// TIA Portal V21 export
FUNCTION "CPEC" : Void   // FC17, LAD
{ S7_Optimized_Access := 'TRUE' }
// stored: SetENOAutomatically false
   VAR_TEMP   // added for the SCL form of the ladder/FBD networks
      _w1 : Bool;
      _w2 : Bool;
      _w3 : Bool;
      _w4 : Bool;
      _w5 : Bool;
      _w6 : Bool;
      _w7 : Bool;
      _w8 : Bool;
      _w9 : Bool;
      _w10 : Bool;
      _w11 : Bool;
      _w12 : Bool;
      _w13 : Bool;
      _w14 : Bool;
      _w15 : Bool;
      _w16 : Bool;
      _w17 : Bool;
      _w18 : Bool;
      _w19 : Bool;
      _w20 : Bool;
      _w21 : Bool;
      _w22 : Bool;
      _w23 : Bool;
      _w24 : Bool;
      _w25 : Bool;
      _w26 : Bool;
      _w27 : Bool;
      _w28 : Bool;
      _w29 : Bool;
      _w30 : Bool;
      _w31 : Bool;
      _w32 : Bool;
      _w33 : Bool;
      _w34 : Bool;
      _w35 : Bool;
      _w36 : Bool;
      _w37 : Bool;
      _w38 : Bool;
      _w39 : Bool;
      _w40 : Bool;
      _w41 : Bool;
      _w42 : Bool;
      _w43 : Bool;
      _w44 : Bool;
      _w45 : Bool;
      _w46 : Bool;
      _w47 : Bool;
      _w48 : Bool;
      _w49 : Bool;
      _w50 : Bool;
      _w51 : Bool;
      _w52 : Bool;
      _w53 : Bool;
      _w54 : Bool;
   END_VAR
BEGIN

REGION Network 1
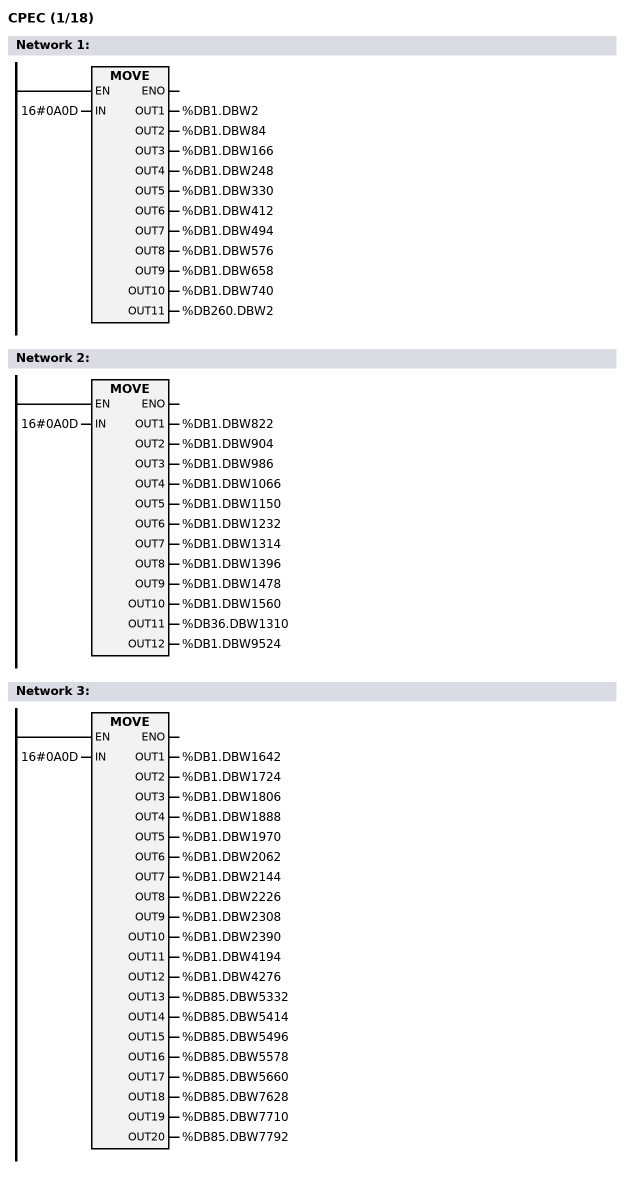
   RUNG wire#powerrail
      Move(in := 16#0A0D, out1 => %DB1.DBW2, out2 => %DB1.DBW84, out3 => %DB1.DBW166, out4 => %DB1.DBW248, out5 => %DB1.DBW330, out6 => %DB1.DBW412, out7 => %DB1.DBW494, out8 => %DB1.DBW576, out9 => %DB1.DBW658, out10 => %DB1.DBW740, out11 => %DB260.DBW2)
   END_RUNG
   // the same network as SCL:
   %DB1.DBW2 := 16#0A0D;
   %DB1.DBW84 := 16#0A0D;
   %DB1.DBW166 := 16#0A0D;
   %DB1.DBW248 := 16#0A0D;
   %DB1.DBW330 := 16#0A0D;
   %DB1.DBW412 := 16#0A0D;
   %DB1.DBW494 := 16#0A0D;
   %DB1.DBW576 := 16#0A0D;
   %DB1.DBW658 := 16#0A0D;
   %DB1.DBW740 := 16#0A0D;
   %DB260.DBW2 := 16#0A0D;
END_REGION

REGION Network 2
   RUNG wire#powerrail
      Move(in := 16#0A0D, out1 => %DB1.DBW822, out2 => %DB1.DBW904, out3 => %DB1.DBW986, out4 => %DB1.DBW1066, out5 => %DB1.DBW1150, out6 => %DB1.DBW1232, out7 => %DB1.DBW1314, out8 => %DB1.DBW1396, out9 => %DB1.DBW1478, out10 => %DB1.DBW1560, out11 => %DB36.DBW1310, out12 => %DB1.DBW9524)
   END_RUNG
   // the same network as SCL:
   %DB1.DBW822 := 16#0A0D;
   %DB1.DBW904 := 16#0A0D;
   %DB1.DBW986 := 16#0A0D;
   %DB1.DBW1066 := 16#0A0D;
   %DB1.DBW1150 := 16#0A0D;
   %DB1.DBW1232 := 16#0A0D;
   %DB1.DBW1314 := 16#0A0D;
   %DB1.DBW1396 := 16#0A0D;
   %DB1.DBW1478 := 16#0A0D;
   %DB1.DBW1560 := 16#0A0D;
   %DB36.DBW1310 := 16#0A0D;
   %DB1.DBW9524 := 16#0A0D;
END_REGION

REGION Network 3
   RUNG wire#powerrail
      Move(in := 16#0A0D, out1 => %DB1.DBW1642, out2 => %DB1.DBW1724, out3 => %DB1.DBW1806, out4 => %DB1.DBW1888, out5 => %DB1.DBW1970, out6 => %DB1.DBW2062, out7 => %DB1.DBW2144, out8 => %DB1.DBW2226, out9 => %DB1.DBW2308, out10 => %DB1.DBW2390, out11 => %DB1.DBW4194, out12 => %DB1.DBW4276, out13 => %DB85.DBW5332, out14 => %DB85.DBW5414, out15 => %DB85.DBW5496, out16 => %DB85.DBW5578, out17 => %DB85.DBW5660, out18 => %DB85.DBW7628, out19 => %DB85.DBW7710, out20 => %DB85.DBW7792)
   END_RUNG
   // the same network as SCL:
   %DB1.DBW1642 := 16#0A0D;
   %DB1.DBW1724 := 16#0A0D;
   %DB1.DBW1806 := 16#0A0D;
   %DB1.DBW1888 := 16#0A0D;
   %DB1.DBW1970 := 16#0A0D;
   %DB1.DBW2062 := 16#0A0D;
   %DB1.DBW2144 := 16#0A0D;
   %DB1.DBW2226 := 16#0A0D;
   %DB1.DBW2308 := 16#0A0D;
   %DB1.DBW2390 := 16#0A0D;
   %DB1.DBW4194 := 16#0A0D;
   %DB1.DBW4276 := 16#0A0D;
   %DB85.DBW5332 := 16#0A0D;
   %DB85.DBW5414 := 16#0A0D;
   %DB85.DBW5496 := 16#0A0D;
   %DB85.DBW5578 := 16#0A0D;
   %DB85.DBW5660 := 16#0A0D;
   %DB85.DBW7628 := 16#0A0D;
   %DB85.DBW7710 := 16#0A0D;
   %DB85.DBW7792 := 16#0A0D;
END_REGION

REGION Network 4
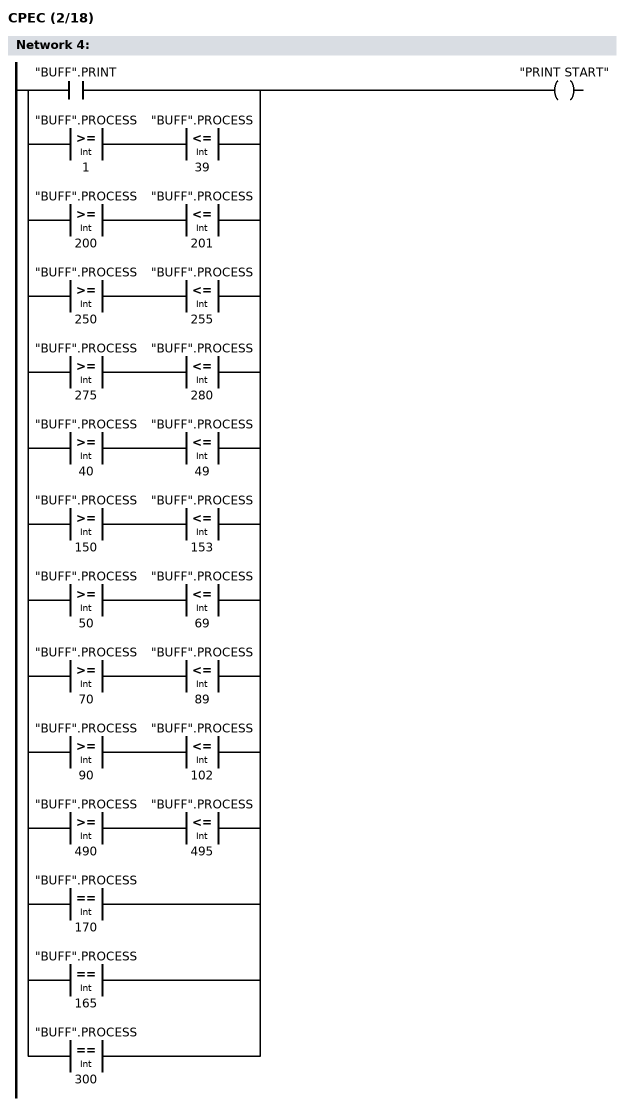
   RUNG wire#powerrail
      Contact( "BUFF".PRINT )
      wire#w1
      Coil( "PRINT START" )
   END_RUNG
   RUNG wire#powerrail
      { S7_Templates := "SrcType := Int" } GE_Contact(in1 := "BUFF".PROCESS, in2 := 1)
      { S7_Templates := "SrcType := Int" } LE_Contact(in1 := "BUFF".PROCESS, in2 := 39)
   END_RUNG wire#w1
   RUNG wire#powerrail
      { S7_Templates := "SrcType := Int" } GE_Contact(in1 := "BUFF".PROCESS, in2 := 200)
      { S7_Templates := "SrcType := Int" } LE_Contact(in1 := "BUFF".PROCESS, in2 := 201)
   END_RUNG wire#w1
   RUNG wire#powerrail
      { S7_Templates := "SrcType := Int" } GE_Contact(in1 := "BUFF".PROCESS, in2 := 250)
      { S7_Templates := "SrcType := Int" } LE_Contact(in1 := "BUFF".PROCESS, in2 := 255)
   END_RUNG wire#w1
   RUNG wire#powerrail
      { S7_Templates := "SrcType := Int" } GE_Contact(in1 := "BUFF".PROCESS, in2 := 275)
      { S7_Templates := "SrcType := Int" } LE_Contact(in1 := "BUFF".PROCESS, in2 := 280)
   END_RUNG wire#w1
   RUNG wire#powerrail
      { S7_Templates := "SrcType := Int" } GE_Contact(in1 := "BUFF".PROCESS, in2 := 40)
      { S7_Templates := "SrcType := Int" } LE_Contact(in1 := "BUFF".PROCESS, in2 := 49)
   END_RUNG wire#w1
   RUNG wire#powerrail
      { S7_Templates := "SrcType := Int" } GE_Contact(in1 := "BUFF".PROCESS, in2 := 150)
      { S7_Templates := "SrcType := Int" } LE_Contact(in1 := "BUFF".PROCESS, in2 := 153)
   END_RUNG wire#w1
   RUNG wire#powerrail
      { S7_Templates := "SrcType := Int" } GE_Contact(in1 := "BUFF".PROCESS, in2 := 50)
      { S7_Templates := "SrcType := Int" } LE_Contact(in1 := "BUFF".PROCESS, in2 := 69)
   END_RUNG wire#w1
   RUNG wire#powerrail
      { S7_Templates := "SrcType := Int" } GE_Contact(in1 := "BUFF".PROCESS, in2 := 70)
      { S7_Templates := "SrcType := Int" } LE_Contact(in1 := "BUFF".PROCESS, in2 := 89)
   END_RUNG wire#w1
   RUNG wire#powerrail
      { S7_Templates := "SrcType := Int" } GE_Contact(in1 := "BUFF".PROCESS, in2 := 90)
      { S7_Templates := "SrcType := Int" } LE_Contact(in1 := "BUFF".PROCESS, in2 := 102)
   END_RUNG wire#w1
   RUNG wire#powerrail
      { S7_Templates := "SrcType := Int" } GE_Contact(in1 := "BUFF".PROCESS, in2 := 490)
      { S7_Templates := "SrcType := Int" } LE_Contact(in1 := "BUFF".PROCESS, in2 := 495)
   END_RUNG wire#w1
   RUNG wire#powerrail
      { S7_Templates := "SrcType := Int" } EQ_Contact(in1 := "BUFF".PROCESS, in2 := 170)
   END_RUNG wire#w1
   RUNG wire#powerrail
      { S7_Templates := "SrcType := Int" } EQ_Contact(in1 := "BUFF".PROCESS, in2 := 165)
   END_RUNG wire#w1
   RUNG wire#powerrail
      { S7_Templates := "SrcType := Int" } EQ_Contact(in1 := "BUFF".PROCESS, in2 := 300)
   END_RUNG wire#w1
   // the same network as SCL:
   "PRINT START" := "BUFF".PRINT OR (("BUFF".PROCESS >= 1) AND ("BUFF".PROCESS <= 39)) OR (("BUFF".PROCESS >= 200) AND ("BUFF".PROCESS <= 201)) OR (("BUFF".PROCESS >= 250) AND ("BUFF".PROCESS <= 255)) OR (("BUFF".PROCESS >= 275) AND ("BUFF".PROCESS <= 280)) OR (("BUFF".PROCESS >= 40) AND ("BUFF".PROCESS <= 49)) OR (("BUFF".PROCESS >= 150) AND ("BUFF".PROCESS <= 153)) OR (("BUFF".PROCESS >= 50) AND ("BUFF".PROCESS <= 69)) OR (("BUFF".PROCESS >= 70) AND ("BUFF".PROCESS <= 89)) OR (("BUFF".PROCESS >= 90) AND ("BUFF".PROCESS <= 102)) OR (("BUFF".PROCESS >= 490) AND ("BUFF".PROCESS <= 495)) OR ("BUFF".PROCESS = 170) OR ("BUFF".PROCESS = 165) OR ("BUFF".PROCESS = 300);
END_REGION

REGION Network 5
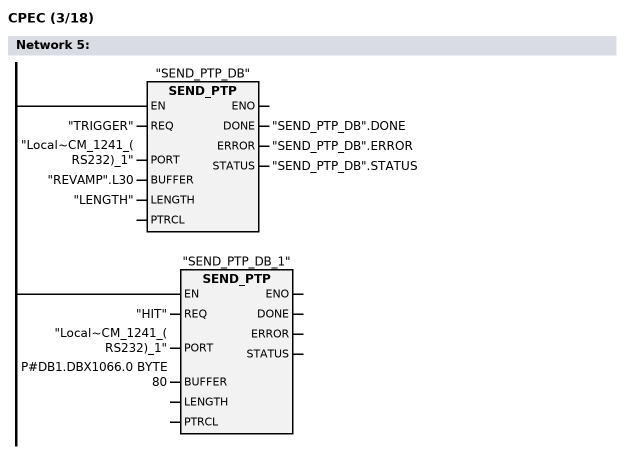
   RUNG wire#powerrail
      "SEND_PTP_DB".SEND_PTP(REQ := "TRIGGER", PORT := "Local~CM_1241_(RS232)_1", BUFFER := "REVAMP".L30, LENGTH := "LENGTH", PTRCL :=, DONE => "SEND_PTP_DB".DONE, ERROR => "SEND_PTP_DB".ERROR, STATUS => "SEND_PTP_DB".STATUS)
   END_RUNG
   RUNG wire#powerrail
      "SEND_PTP_DB_1".SEND_PTP(REQ := "HIT", PORT := "Local~CM_1241_(RS232)_1", BUFFER := P#DB1.DBX1066.0 BYTE 80, LENGTH :=, PTRCL :=, DONE =>, ERROR =>, STATUS =>)
   END_RUNG
   // the same network as SCL:
   "SEND_PTP_DB"(REQ := "TRIGGER",   // SEND_PTP
                 PORT := "Local~CM_1241_(RS232)_1",
                 BUFFER := "REVAMP".L30,
                 LENGTH := "LENGTH",
                 DONE => "SEND_PTP_DB".DONE,
                 ERROR => "SEND_PTP_DB".ERROR,
                 STATUS => "SEND_PTP_DB".STATUS);
   "SEND_PTP_DB_1"(REQ := "HIT", PORT := "Local~CM_1241_(RS232)_1", BUFFER := P#DB1.DBX1066.0 BYTE 80);   // SEND_PTP
END_REGION

REGION Network 6
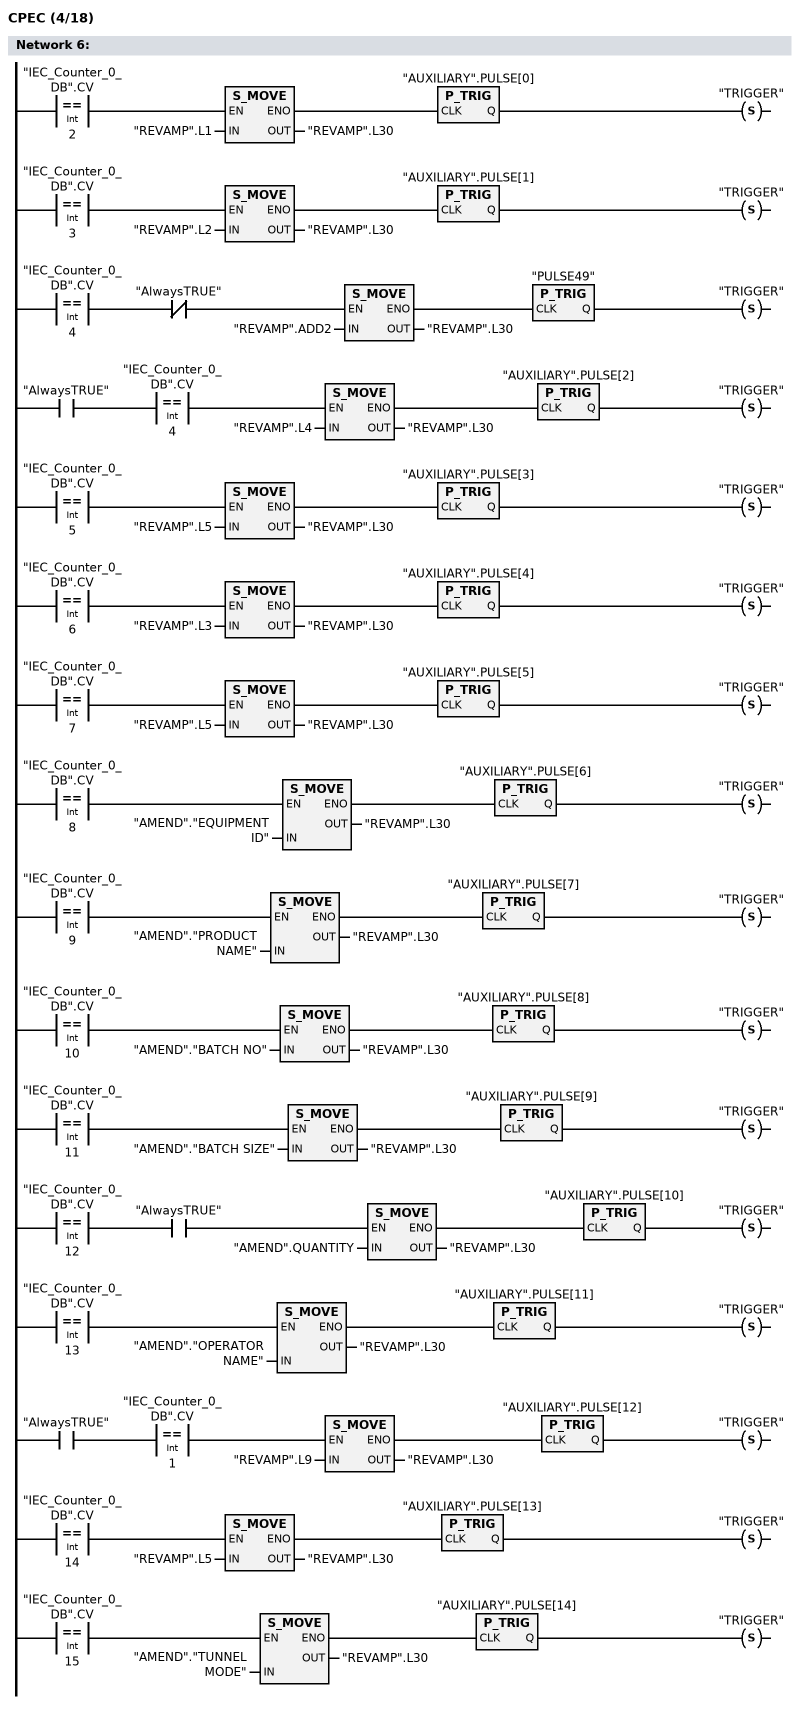
   RUNG wire#powerrail
      { S7_Templates := "SrcType := Int" } EQ_Contact(in1 := "IEC_Counter_0_DB".CV, in2 := 2)
      S_Move(in := "REVAMP".L1, out => "REVAMP".L30)
      P_Trig( "AUXILIARY".PULSE[0] )
      S_Coil( "TRIGGER" )
   END_RUNG
   RUNG wire#powerrail
      { S7_Templates := "SrcType := Int" } EQ_Contact(in1 := "IEC_Counter_0_DB".CV, in2 := 3)
      S_Move(in := "REVAMP".L2, out => "REVAMP".L30)
      P_Trig( "AUXILIARY".PULSE[1] )
      S_Coil( "TRIGGER" )
   END_RUNG
   RUNG wire#powerrail
      { S7_Templates := "SrcType := Int" } EQ_Contact(in1 := "IEC_Counter_0_DB".CV, in2 := 4)
      I_Contact( "AlwaysTRUE" )
      S_Move(in := "REVAMP".ADD2, out => "REVAMP".L30)
      P_Trig( "PULSE49" )
      S_Coil( "TRIGGER" )
   END_RUNG
   RUNG wire#powerrail
      Contact( "AlwaysTRUE" )
      { S7_Templates := "SrcType := Int" } EQ_Contact(in1 := "IEC_Counter_0_DB".CV, in2 := 4)
      S_Move(in := "REVAMP".L4, out => "REVAMP".L30)
      P_Trig( "AUXILIARY".PULSE[2] )
      S_Coil( "TRIGGER" )
   END_RUNG
   RUNG wire#powerrail
      { S7_Templates := "SrcType := Int" } EQ_Contact(in1 := "IEC_Counter_0_DB".CV, in2 := 5)
      S_Move(in := "REVAMP".L5, out => "REVAMP".L30)
      P_Trig( "AUXILIARY".PULSE[3] )
      S_Coil( "TRIGGER" )
   END_RUNG
   RUNG wire#powerrail
      { S7_Templates := "SrcType := Int" } EQ_Contact(in1 := "IEC_Counter_0_DB".CV, in2 := 6)
      S_Move(in := "REVAMP".L3, out => "REVAMP".L30)
      P_Trig( "AUXILIARY".PULSE[4] )
      S_Coil( "TRIGGER" )
   END_RUNG
   RUNG wire#powerrail
      { S7_Templates := "SrcType := Int" } EQ_Contact(in1 := "IEC_Counter_0_DB".CV, in2 := 7)
      S_Move(in := "REVAMP".L5, out => "REVAMP".L30)
      P_Trig( "AUXILIARY".PULSE[5] )
      S_Coil( "TRIGGER" )
   END_RUNG
   RUNG wire#powerrail
      { S7_Templates := "SrcType := Int" } EQ_Contact(in1 := "IEC_Counter_0_DB".CV, in2 := 8)
      S_Move(in := "AMEND"."EQUIPMENT ID", out => "REVAMP".L30)
      P_Trig( "AUXILIARY".PULSE[6] )
      S_Coil( "TRIGGER" )
   END_RUNG
   RUNG wire#powerrail
      { S7_Templates := "SrcType := Int" } EQ_Contact(in1 := "IEC_Counter_0_DB".CV, in2 := 9)
      S_Move(in := "AMEND"."PRODUCT NAME", out => "REVAMP".L30)
      P_Trig( "AUXILIARY".PULSE[7] )
      S_Coil( "TRIGGER" )
   END_RUNG
   RUNG wire#powerrail
      { S7_Templates := "SrcType := Int" } EQ_Contact(in1 := "IEC_Counter_0_DB".CV, in2 := 10)
      S_Move(in := "AMEND"."BATCH NO", out => "REVAMP".L30)
      P_Trig( "AUXILIARY".PULSE[8] )
      S_Coil( "TRIGGER" )
   END_RUNG
   RUNG wire#powerrail
      { S7_Templates := "SrcType := Int" } EQ_Contact(in1 := "IEC_Counter_0_DB".CV, in2 := 11)
      S_Move(in := "AMEND"."BATCH SIZE", out => "REVAMP".L30)
      P_Trig( "AUXILIARY".PULSE[9] )
      S_Coil( "TRIGGER" )
   END_RUNG
   RUNG wire#powerrail
      { S7_Templates := "SrcType := Int" } EQ_Contact(in1 := "IEC_Counter_0_DB".CV, in2 := 12)
      Contact( "AlwaysTRUE" )
      S_Move(in := "AMEND".QUANTITY, out => "REVAMP".L30)
      P_Trig( "AUXILIARY".PULSE[10] )
      S_Coil( "TRIGGER" )
   END_RUNG
   RUNG wire#powerrail
      { S7_Templates := "SrcType := Int" } EQ_Contact(in1 := "IEC_Counter_0_DB".CV, in2 := 13)
      S_Move(in := "AMEND"."OPERATOR NAME", out => "REVAMP".L30)
      P_Trig( "AUXILIARY".PULSE[11] )
      S_Coil( "TRIGGER" )
   END_RUNG
   RUNG wire#powerrail
      Contact( "AlwaysTRUE" )
      { S7_Templates := "SrcType := Int" } EQ_Contact(in1 := "IEC_Counter_0_DB".CV, in2 := 1)
      S_Move(in := "REVAMP".L9, out => "REVAMP".L30)
      P_Trig( "AUXILIARY".PULSE[12] )
      S_Coil( "TRIGGER" )
   END_RUNG
   RUNG wire#powerrail
      { S7_Templates := "SrcType := Int" } EQ_Contact(in1 := "IEC_Counter_0_DB".CV, in2 := 14)
      S_Move(in := "REVAMP".L5, out => "REVAMP".L30)
      P_Trig( "AUXILIARY".PULSE[13] )
      S_Coil( "TRIGGER" )
   END_RUNG
   RUNG wire#powerrail
      { S7_Templates := "SrcType := Int" } EQ_Contact(in1 := "IEC_Counter_0_DB".CV, in2 := 15)
      S_Move(in := "AMEND"."TUNNEL MODE", out => "REVAMP".L30)
      P_Trig( "AUXILIARY".PULSE[14] )
      S_Coil( "TRIGGER" )
   END_RUNG
   // the same network as SCL:
   #_w1 := "IEC_Counter_0_DB".CV = 2;
   IF #_w1 THEN "REVAMP".L30 := "REVAMP".L1; END_IF;
   #_w2 := #_w1 AND NOT "AUXILIARY".PULSE[0];   // rising edge
   "AUXILIARY".PULSE[0] := #_w1;
   IF #_w2 THEN "TRIGGER" := TRUE; END_IF;
   #_w3 := "IEC_Counter_0_DB".CV = 3;
   IF #_w3 THEN "REVAMP".L30 := "REVAMP".L2; END_IF;
   #_w4 := #_w3 AND NOT "AUXILIARY".PULSE[1];   // rising edge
   "AUXILIARY".PULSE[1] := #_w3;
   IF #_w4 THEN "TRIGGER" := TRUE; END_IF;
   #_w5 := ("IEC_Counter_0_DB".CV = 4) AND NOT "AlwaysTRUE";
   IF #_w5 THEN "REVAMP".L30 := "REVAMP".ADD2; END_IF;
   #_w6 := #_w5 AND NOT "PULSE49";   // rising edge
   "PULSE49" := #_w5;
   IF #_w6 THEN "TRIGGER" := TRUE; END_IF;
   #_w7 := "AlwaysTRUE" AND ("IEC_Counter_0_DB".CV = 4);
   IF #_w7 THEN "REVAMP".L30 := "REVAMP".L4; END_IF;
   #_w8 := #_w7 AND NOT "AUXILIARY".PULSE[2];   // rising edge
   "AUXILIARY".PULSE[2] := #_w7;
   IF #_w8 THEN "TRIGGER" := TRUE; END_IF;
   #_w9 := "IEC_Counter_0_DB".CV = 5;
   IF #_w9 THEN "REVAMP".L30 := "REVAMP".L5; END_IF;
   #_w10 := #_w9 AND NOT "AUXILIARY".PULSE[3];   // rising edge
   "AUXILIARY".PULSE[3] := #_w9;
   IF #_w10 THEN "TRIGGER" := TRUE; END_IF;
   #_w11 := "IEC_Counter_0_DB".CV = 6;
   IF #_w11 THEN "REVAMP".L30 := "REVAMP".L3; END_IF;
   #_w12 := #_w11 AND NOT "AUXILIARY".PULSE[4];   // rising edge
   "AUXILIARY".PULSE[4] := #_w11;
   IF #_w12 THEN "TRIGGER" := TRUE; END_IF;
   #_w13 := "IEC_Counter_0_DB".CV = 7;
   IF #_w13 THEN "REVAMP".L30 := "REVAMP".L5; END_IF;
   #_w14 := #_w13 AND NOT "AUXILIARY".PULSE[5];   // rising edge
   "AUXILIARY".PULSE[5] := #_w13;
   IF #_w14 THEN "TRIGGER" := TRUE; END_IF;
   #_w15 := "IEC_Counter_0_DB".CV = 8;
   IF #_w15 THEN "REVAMP".L30 := "AMEND"."EQUIPMENT ID"; END_IF;
   #_w16 := #_w15 AND NOT "AUXILIARY".PULSE[6];   // rising edge
   "AUXILIARY".PULSE[6] := #_w15;
   IF #_w16 THEN "TRIGGER" := TRUE; END_IF;
   #_w17 := "IEC_Counter_0_DB".CV = 9;
   IF #_w17 THEN "REVAMP".L30 := "AMEND"."PRODUCT NAME"; END_IF;
   #_w18 := #_w17 AND NOT "AUXILIARY".PULSE[7];   // rising edge
   "AUXILIARY".PULSE[7] := #_w17;
   IF #_w18 THEN "TRIGGER" := TRUE; END_IF;
   #_w19 := "IEC_Counter_0_DB".CV = 10;
   IF #_w19 THEN "REVAMP".L30 := "AMEND"."BATCH NO"; END_IF;
   #_w20 := #_w19 AND NOT "AUXILIARY".PULSE[8];   // rising edge
   "AUXILIARY".PULSE[8] := #_w19;
   IF #_w20 THEN "TRIGGER" := TRUE; END_IF;
   #_w21 := "IEC_Counter_0_DB".CV = 11;
   IF #_w21 THEN "REVAMP".L30 := "AMEND"."BATCH SIZE"; END_IF;
   #_w22 := #_w21 AND NOT "AUXILIARY".PULSE[9];   // rising edge
   "AUXILIARY".PULSE[9] := #_w21;
   IF #_w22 THEN "TRIGGER" := TRUE; END_IF;
   #_w23 := ("IEC_Counter_0_DB".CV = 12) AND "AlwaysTRUE";
   IF #_w23 THEN "REVAMP".L30 := "AMEND".QUANTITY; END_IF;
   #_w24 := #_w23 AND NOT "AUXILIARY".PULSE[10];   // rising edge
   "AUXILIARY".PULSE[10] := #_w23;
   IF #_w24 THEN "TRIGGER" := TRUE; END_IF;
   #_w25 := "IEC_Counter_0_DB".CV = 13;
   IF #_w25 THEN "REVAMP".L30 := "AMEND"."OPERATOR NAME"; END_IF;
   #_w26 := #_w25 AND NOT "AUXILIARY".PULSE[11];   // rising edge
   "AUXILIARY".PULSE[11] := #_w25;
   IF #_w26 THEN "TRIGGER" := TRUE; END_IF;
   #_w27 := "AlwaysTRUE" AND ("IEC_Counter_0_DB".CV = 1);
   IF #_w27 THEN "REVAMP".L30 := "REVAMP".L9; END_IF;
   #_w28 := #_w27 AND NOT "AUXILIARY".PULSE[12];   // rising edge
   "AUXILIARY".PULSE[12] := #_w27;
   IF #_w28 THEN "TRIGGER" := TRUE; END_IF;
   #_w29 := "IEC_Counter_0_DB".CV = 14;
   IF #_w29 THEN "REVAMP".L30 := "REVAMP".L5; END_IF;
   #_w30 := #_w29 AND NOT "AUXILIARY".PULSE[13];   // rising edge
   "AUXILIARY".PULSE[13] := #_w29;
   IF #_w30 THEN "TRIGGER" := TRUE; END_IF;
   #_w31 := "IEC_Counter_0_DB".CV = 15;
   IF #_w31 THEN "REVAMP".L30 := "AMEND"."TUNNEL MODE"; END_IF;
   #_w32 := #_w31 AND NOT "AUXILIARY".PULSE[14];   // rising edge
   "AUXILIARY".PULSE[14] := #_w31;
   IF #_w32 THEN "TRIGGER" := TRUE; END_IF;
END_REGION

REGION Network 7
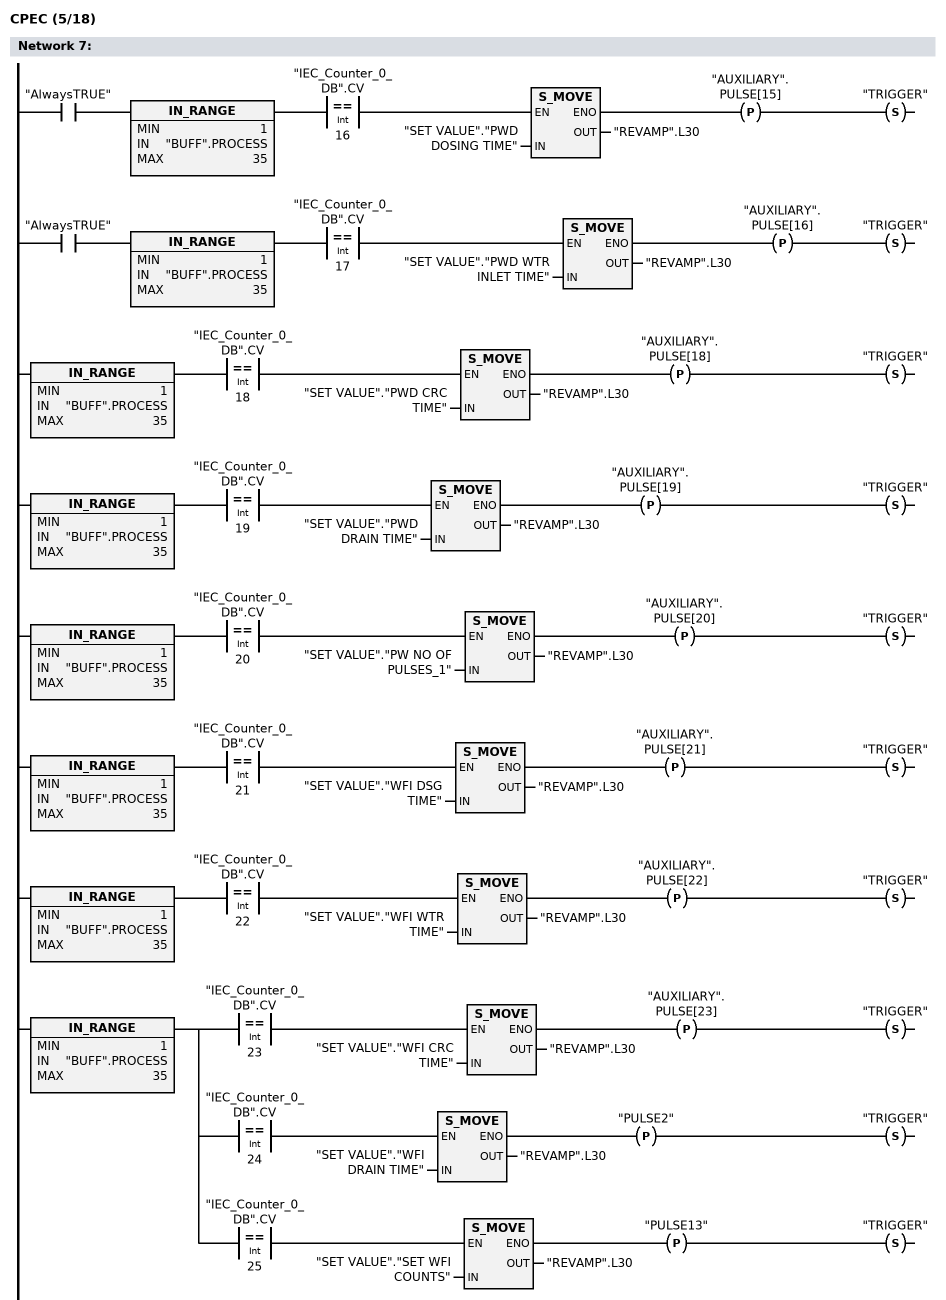
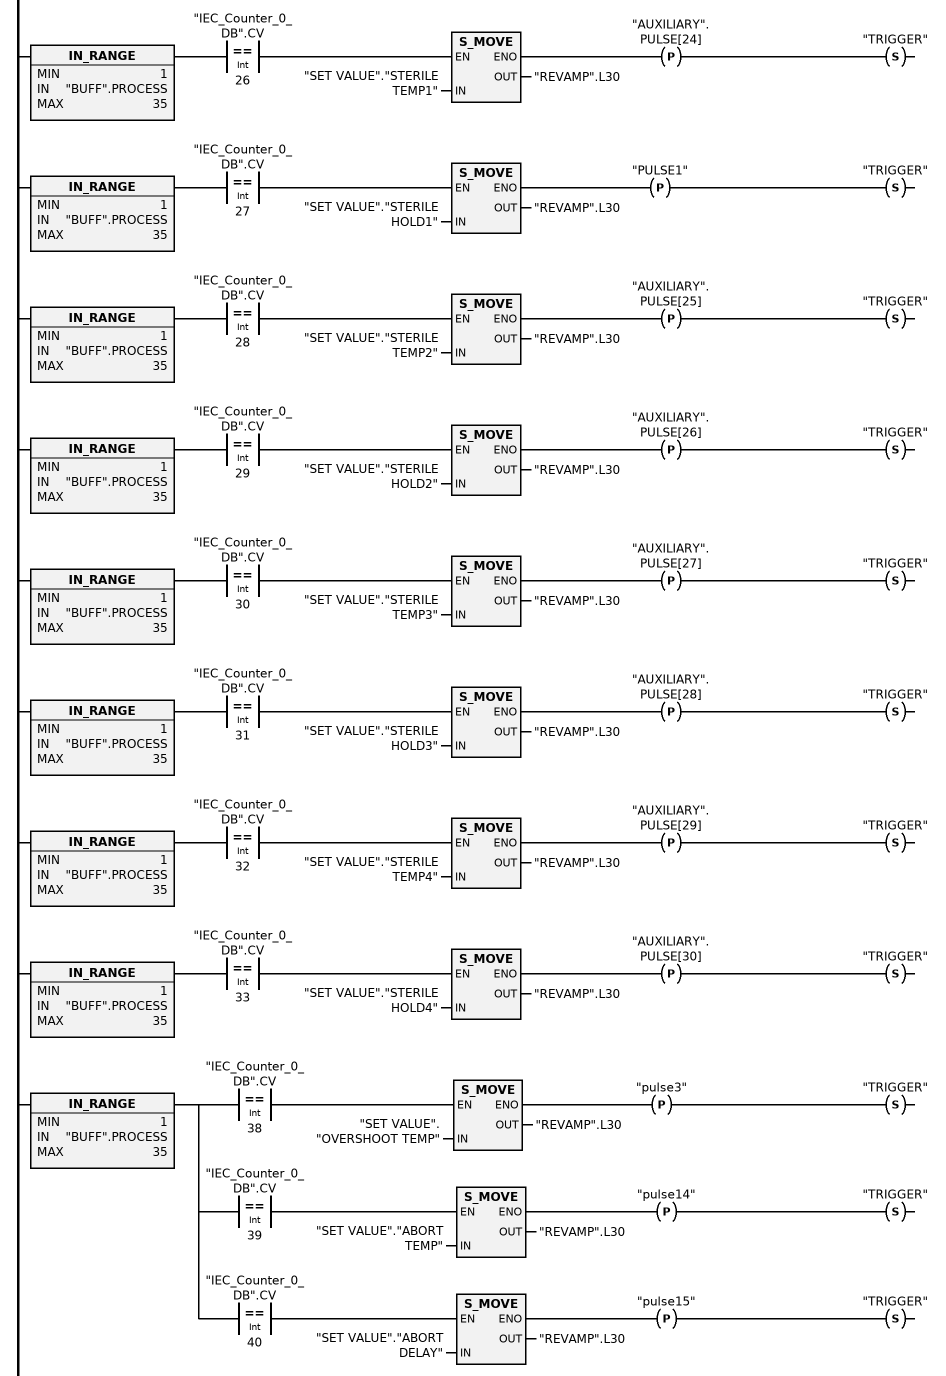
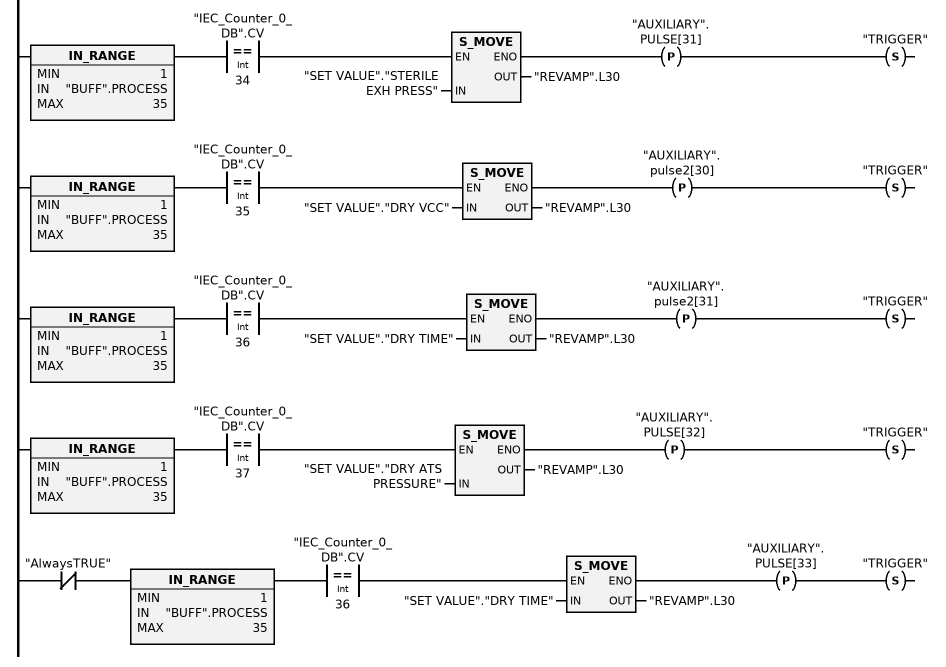
   RUNG wire#powerrail
      Contact( "AlwaysTRUE" )
      { S7_Templates := "SrcType := Int" } InRange(min := 1, in := "BUFF".PROCESS, max := 35)
      { S7_Templates := "SrcType := Int" } EQ_Contact(in1 := "IEC_Counter_0_DB".CV, in2 := 16)
      S_Move(in := "SET VALUE"."PWD DOSING TIME", out => "REVAMP".L30)
      P_Trig( "AUXILIARY".PULSE[15] )
      S_Coil( "TRIGGER" )
   END_RUNG
   RUNG wire#powerrail
      Contact( "AlwaysTRUE" )
      { S7_Templates := "SrcType := Int" } InRange(min := 1, in := "BUFF".PROCESS, max := 35)
      { S7_Templates := "SrcType := Int" } EQ_Contact(in1 := "IEC_Counter_0_DB".CV, in2 := 17)
      S_Move(in := "SET VALUE"."PWD WTR INLET TIME", out => "REVAMP".L30)
      P_Trig( "AUXILIARY".PULSE[16] )
      S_Coil( "TRIGGER" )
   END_RUNG
   RUNG wire#powerrail
      { S7_Templates := "SrcType := Int" } InRange(min := 1, in := "BUFF".PROCESS, max := 35)
      { S7_Templates := "SrcType := Int" } EQ_Contact(in1 := "IEC_Counter_0_DB".CV, in2 := 18)
      S_Move(in := "SET VALUE"."PWD CRC TIME", out => "REVAMP".L30)
      P_Trig( "AUXILIARY".PULSE[18] )
      S_Coil( "TRIGGER" )
   END_RUNG
   RUNG wire#powerrail
      { S7_Templates := "SrcType := Int" } InRange(min := 1, in := "BUFF".PROCESS, max := 35)
      { S7_Templates := "SrcType := Int" } EQ_Contact(in1 := "IEC_Counter_0_DB".CV, in2 := 19)
      S_Move(in := "SET VALUE"."PWD DRAIN TIME", out => "REVAMP".L30)
      P_Trig( "AUXILIARY".PULSE[19] )
      S_Coil( "TRIGGER" )
   END_RUNG
   RUNG wire#powerrail
      { S7_Templates := "SrcType := Int" } InRange(min := 1, in := "BUFF".PROCESS, max := 35)
      { S7_Templates := "SrcType := Int" } EQ_Contact(in1 := "IEC_Counter_0_DB".CV, in2 := 20)
      S_Move(in := "SET VALUE"."PW NO OF PULSES_1", out => "REVAMP".L30)
      P_Trig( "AUXILIARY".PULSE[20] )
      S_Coil( "TRIGGER" )
   END_RUNG
   RUNG wire#powerrail
      { S7_Templates := "SrcType := Int" } InRange(min := 1, in := "BUFF".PROCESS, max := 35)
      { S7_Templates := "SrcType := Int" } EQ_Contact(in1 := "IEC_Counter_0_DB".CV, in2 := 21)
      S_Move(in := "SET VALUE"."WFI DSG TIME", out => "REVAMP".L30)
      P_Trig( "AUXILIARY".PULSE[21] )
      S_Coil( "TRIGGER" )
   END_RUNG
   RUNG wire#powerrail
      { S7_Templates := "SrcType := Int" } InRange(min := 1, in := "BUFF".PROCESS, max := 35)
      { S7_Templates := "SrcType := Int" } EQ_Contact(in1 := "IEC_Counter_0_DB".CV, in2 := 22)
      S_Move(in := "SET VALUE"."WFI WTR TIME", out => "REVAMP".L30)
      P_Trig( "AUXILIARY".PULSE[22] )
      S_Coil( "TRIGGER" )
   END_RUNG
   RUNG wire#powerrail
      { S7_Templates := "SrcType := Int" } InRange(min := 1, in := "BUFF".PROCESS, max := 35)
      wire#w1
      { S7_Templates := "SrcType := Int" } EQ_Contact(in1 := "IEC_Counter_0_DB".CV, in2 := 23)
      S_Move(in := "SET VALUE"."WFI CRC TIME", out => "REVAMP".L30)
      P_Trig( "AUXILIARY".PULSE[23] )
      S_Coil( "TRIGGER" )
   END_RUNG
   RUNG wire#w1
      { S7_Templates := "SrcType := Int" } EQ_Contact(in1 := "IEC_Counter_0_DB".CV, in2 := 24)
      S_Move(in := "SET VALUE"."WFI DRAIN TIME", out => "REVAMP".L30)
      P_Trig( "PULSE2" )
      S_Coil( "TRIGGER" )
   END_RUNG
   RUNG wire#w1
      { S7_Templates := "SrcType := Int" } EQ_Contact(in1 := "IEC_Counter_0_DB".CV, in2 := 25)
      S_Move(in := "SET VALUE"."SET WFI COUNTS", out => "REVAMP".L30)
      P_Trig( "PULSE13" )
      S_Coil( "TRIGGER" )
   END_RUNG
   RUNG wire#powerrail
      { S7_Templates := "SrcType := Int" } InRange(min := 1, in := "BUFF".PROCESS, max := 35)
      { S7_Templates := "SrcType := Int" } EQ_Contact(in1 := "IEC_Counter_0_DB".CV, in2 := 26)
      S_Move(in := "SET VALUE"."STERILE TEMP1", out => "REVAMP".L30)
      P_Trig( "AUXILIARY".PULSE[24] )
      S_Coil( "TRIGGER" )
   END_RUNG
   RUNG wire#powerrail
      { S7_Templates := "SrcType := Int" } InRange(min := 1, in := "BUFF".PROCESS, max := 35)
      { S7_Templates := "SrcType := Int" } EQ_Contact(in1 := "IEC_Counter_0_DB".CV, in2 := 27)
      S_Move(in := "SET VALUE"."STERILE HOLD1", out => "REVAMP".L30)
      P_Trig( "PULSE1" )
      S_Coil( "TRIGGER" )
   END_RUNG
   RUNG wire#powerrail
      { S7_Templates := "SrcType := Int" } InRange(min := 1, in := "BUFF".PROCESS, max := 35)
      { S7_Templates := "SrcType := Int" } EQ_Contact(in1 := "IEC_Counter_0_DB".CV, in2 := 28)
      S_Move(in := "SET VALUE"."STERILE TEMP2", out => "REVAMP".L30)
      P_Trig( "AUXILIARY".PULSE[25] )
      S_Coil( "TRIGGER" )
   END_RUNG
   RUNG wire#powerrail
      { S7_Templates := "SrcType := Int" } InRange(min := 1, in := "BUFF".PROCESS, max := 35)
      { S7_Templates := "SrcType := Int" } EQ_Contact(in1 := "IEC_Counter_0_DB".CV, in2 := 29)
      S_Move(in := "SET VALUE"."STERILE HOLD2", out => "REVAMP".L30)
      P_Trig( "AUXILIARY".PULSE[26] )
      S_Coil( "TRIGGER" )
   END_RUNG
   RUNG wire#powerrail
      { S7_Templates := "SrcType := Int" } InRange(min := 1, in := "BUFF".PROCESS, max := 35)
      { S7_Templates := "SrcType := Int" } EQ_Contact(in1 := "IEC_Counter_0_DB".CV, in2 := 30)
      S_Move(in := "SET VALUE"."STERILE TEMP3", out => "REVAMP".L30)
      P_Trig( "AUXILIARY".PULSE[27] )
      S_Coil( "TRIGGER" )
   END_RUNG
   RUNG wire#powerrail
      { S7_Templates := "SrcType := Int" } InRange(min := 1, in := "BUFF".PROCESS, max := 35)
      { S7_Templates := "SrcType := Int" } EQ_Contact(in1 := "IEC_Counter_0_DB".CV, in2 := 31)
      S_Move(in := "SET VALUE"."STERILE HOLD3", out => "REVAMP".L30)
      P_Trig( "AUXILIARY".PULSE[28] )
      S_Coil( "TRIGGER" )
   END_RUNG
   RUNG wire#powerrail
      { S7_Templates := "SrcType := Int" } InRange(min := 1, in := "BUFF".PROCESS, max := 35)
      { S7_Templates := "SrcType := Int" } EQ_Contact(in1 := "IEC_Counter_0_DB".CV, in2 := 32)
      S_Move(in := "SET VALUE"."STERILE TEMP4", out => "REVAMP".L30)
      P_Trig( "AUXILIARY".PULSE[29] )
      S_Coil( "TRIGGER" )
   END_RUNG
   RUNG wire#powerrail
      { S7_Templates := "SrcType := Int" } InRange(min := 1, in := "BUFF".PROCESS, max := 35)
      { S7_Templates := "SrcType := Int" } EQ_Contact(in1 := "IEC_Counter_0_DB".CV, in2 := 33)
      S_Move(in := "SET VALUE"."STERILE HOLD4", out => "REVAMP".L30)
      P_Trig( "AUXILIARY".PULSE[30] )
      S_Coil( "TRIGGER" )
   END_RUNG
   RUNG wire#powerrail
      { S7_Templates := "SrcType := Int" } InRange(min := 1, in := "BUFF".PROCESS, max := 35)
      wire#w2
      { S7_Templates := "SrcType := Int" } EQ_Contact(in1 := "IEC_Counter_0_DB".CV, in2 := 38)
      S_Move(in := "SET VALUE"."OVERSHOOT TEMP", out => "REVAMP".L30)
      P_Trig( "pulse3" )
      S_Coil( "TRIGGER" )
   END_RUNG
   RUNG wire#w2
      { S7_Templates := "SrcType := Int" } EQ_Contact(in1 := "IEC_Counter_0_DB".CV, in2 := 39)
      S_Move(in := "SET VALUE"."ABORT TEMP", out => "REVAMP".L30)
      P_Trig( "pulse14" )
      S_Coil( "TRIGGER" )
   END_RUNG
   RUNG wire#w2
      { S7_Templates := "SrcType := Int" } EQ_Contact(in1 := "IEC_Counter_0_DB".CV, in2 := 40)
      S_Move(in := "SET VALUE"."ABORT DELAY", out => "REVAMP".L30)
      P_Trig( "pulse15" )
      S_Coil( "TRIGGER" )
   END_RUNG
   RUNG wire#powerrail
      { S7_Templates := "SrcType := Int" } InRange(min := 1, in := "BUFF".PROCESS, max := 35)
      { S7_Templates := "SrcType := Int" } EQ_Contact(in1 := "IEC_Counter_0_DB".CV, in2 := 34)
      S_Move(in := "SET VALUE"."STERILE EXH PRESS", out => "REVAMP".L30)
      P_Trig( "AUXILIARY".PULSE[31] )
      S_Coil( "TRIGGER" )
   END_RUNG
   RUNG wire#powerrail
      { S7_Templates := "SrcType := Int" } InRange(min := 1, in := "BUFF".PROCESS, max := 35)
      { S7_Templates := "SrcType := Int" } EQ_Contact(in1 := "IEC_Counter_0_DB".CV, in2 := 35)
      S_Move(in := "SET VALUE"."DRY VCC", out => "REVAMP".L30)
      P_Trig( "AUXILIARY".pulse2[30] )
      S_Coil( "TRIGGER" )
   END_RUNG
   RUNG wire#powerrail
      { S7_Templates := "SrcType := Int" } InRange(min := 1, in := "BUFF".PROCESS, max := 35)
      { S7_Templates := "SrcType := Int" } EQ_Contact(in1 := "IEC_Counter_0_DB".CV, in2 := 36)
      S_Move(in := "SET VALUE"."DRY TIME", out => "REVAMP".L30)
      P_Trig( "AUXILIARY".pulse2[31] )
      S_Coil( "TRIGGER" )
   END_RUNG
   RUNG wire#powerrail
      { S7_Templates := "SrcType := Int" } InRange(min := 1, in := "BUFF".PROCESS, max := 35)
      { S7_Templates := "SrcType := Int" } EQ_Contact(in1 := "IEC_Counter_0_DB".CV, in2 := 37)
      S_Move(in := "SET VALUE"."DRY ATS PRESSURE", out => "REVAMP".L30)
      P_Trig( "AUXILIARY".PULSE[32] )
      S_Coil( "TRIGGER" )
   END_RUNG
   RUNG wire#powerrail
      I_Contact( "AlwaysTRUE" )
      { S7_Templates := "SrcType := Int" } InRange(min := 1, in := "BUFF".PROCESS, max := 35)
      { S7_Templates := "SrcType := Int" } EQ_Contact(in1 := "IEC_Counter_0_DB".CV, in2 := 36)
      S_Move(in := "SET VALUE"."DRY TIME", out => "REVAMP".L30)
      P_Trig( "AUXILIARY".PULSE[33] )
      S_Coil( "TRIGGER" )
   END_RUNG
   // the same network as SCL:
   #_w1 := "AlwaysTRUE" AND (1 <= "BUFF".PROCESS) AND ("BUFF".PROCESS <= 35) AND ("IEC_Counter_0_DB".CV = 16);
   IF #_w1 THEN "REVAMP".L30 := "SET VALUE"."PWD DOSING TIME"; END_IF;
   #_w2 := #_w1 AND NOT "AUXILIARY".PULSE[15];   // rising edge
   "AUXILIARY".PULSE[15] := #_w1;
   IF #_w2 THEN "TRIGGER" := TRUE; END_IF;
   #_w3 := "AlwaysTRUE" AND (1 <= "BUFF".PROCESS) AND ("BUFF".PROCESS <= 35) AND ("IEC_Counter_0_DB".CV = 17);
   IF #_w3 THEN "REVAMP".L30 := "SET VALUE"."PWD WTR INLET TIME"; END_IF;
   #_w4 := #_w3 AND NOT "AUXILIARY".PULSE[16];   // rising edge
   "AUXILIARY".PULSE[16] := #_w3;
   IF #_w4 THEN "TRIGGER" := TRUE; END_IF;
   #_w5 := (1 <= "BUFF".PROCESS) AND ("BUFF".PROCESS <= 35) AND ("IEC_Counter_0_DB".CV = 18);
   IF #_w5 THEN "REVAMP".L30 := "SET VALUE"."PWD CRC TIME"; END_IF;
   #_w6 := #_w5 AND NOT "AUXILIARY".PULSE[18];   // rising edge
   "AUXILIARY".PULSE[18] := #_w5;
   IF #_w6 THEN "TRIGGER" := TRUE; END_IF;
   #_w7 := (1 <= "BUFF".PROCESS) AND ("BUFF".PROCESS <= 35) AND ("IEC_Counter_0_DB".CV = 19);
   IF #_w7 THEN "REVAMP".L30 := "SET VALUE"."PWD DRAIN TIME"; END_IF;
   #_w8 := #_w7 AND NOT "AUXILIARY".PULSE[19];   // rising edge
   "AUXILIARY".PULSE[19] := #_w7;
   IF #_w8 THEN "TRIGGER" := TRUE; END_IF;
   #_w9 := (1 <= "BUFF".PROCESS) AND ("BUFF".PROCESS <= 35) AND ("IEC_Counter_0_DB".CV = 20);
   IF #_w9 THEN "REVAMP".L30 := "SET VALUE"."PW NO OF PULSES_1"; END_IF;
   #_w10 := #_w9 AND NOT "AUXILIARY".PULSE[20];   // rising edge
   "AUXILIARY".PULSE[20] := #_w9;
   IF #_w10 THEN "TRIGGER" := TRUE; END_IF;
   #_w11 := (1 <= "BUFF".PROCESS) AND ("BUFF".PROCESS <= 35) AND ("IEC_Counter_0_DB".CV = 21);
   IF #_w11 THEN "REVAMP".L30 := "SET VALUE"."WFI DSG TIME"; END_IF;
   #_w12 := #_w11 AND NOT "AUXILIARY".PULSE[21];   // rising edge
   "AUXILIARY".PULSE[21] := #_w11;
   IF #_w12 THEN "TRIGGER" := TRUE; END_IF;
   #_w13 := (1 <= "BUFF".PROCESS) AND ("BUFF".PROCESS <= 35) AND ("IEC_Counter_0_DB".CV = 22);
   IF #_w13 THEN "REVAMP".L30 := "SET VALUE"."WFI WTR TIME"; END_IF;
   #_w14 := #_w13 AND NOT "AUXILIARY".PULSE[22];   // rising edge
   "AUXILIARY".PULSE[22] := #_w13;
   IF #_w14 THEN "TRIGGER" := TRUE; END_IF;
   #_w15 := (1 <= "BUFF".PROCESS) AND ("BUFF".PROCESS <= 35);
   #_w16 := #_w15 AND ("IEC_Counter_0_DB".CV = 23);
   IF #_w16 THEN "REVAMP".L30 := "SET VALUE"."WFI CRC TIME"; END_IF;
   #_w17 := #_w16 AND NOT "AUXILIARY".PULSE[23];   // rising edge
   "AUXILIARY".PULSE[23] := #_w16;
   IF #_w17 THEN "TRIGGER" := TRUE; END_IF;
   #_w18 := #_w15 AND ("IEC_Counter_0_DB".CV = 24);
   IF #_w18 THEN "REVAMP".L30 := "SET VALUE"."WFI DRAIN TIME"; END_IF;
   #_w19 := #_w18 AND NOT "PULSE2";   // rising edge
   "PULSE2" := #_w18;
   IF #_w19 THEN "TRIGGER" := TRUE; END_IF;
   #_w20 := #_w15 AND ("IEC_Counter_0_DB".CV = 25);
   IF #_w20 THEN "REVAMP".L30 := "SET VALUE"."SET WFI COUNTS"; END_IF;
   #_w21 := #_w20 AND NOT "PULSE13";   // rising edge
   "PULSE13" := #_w20;
   IF #_w21 THEN "TRIGGER" := TRUE; END_IF;
   #_w22 := (1 <= "BUFF".PROCESS) AND ("BUFF".PROCESS <= 35) AND ("IEC_Counter_0_DB".CV = 26);
   IF #_w22 THEN "REVAMP".L30 := "SET VALUE"."STERILE TEMP1"; END_IF;
   #_w23 := #_w22 AND NOT "AUXILIARY".PULSE[24];   // rising edge
   "AUXILIARY".PULSE[24] := #_w22;
   IF #_w23 THEN "TRIGGER" := TRUE; END_IF;
   #_w24 := (1 <= "BUFF".PROCESS) AND ("BUFF".PROCESS <= 35) AND ("IEC_Counter_0_DB".CV = 27);
   IF #_w24 THEN "REVAMP".L30 := "SET VALUE"."STERILE HOLD1"; END_IF;
   #_w25 := #_w24 AND NOT "PULSE1";   // rising edge
   "PULSE1" := #_w24;
   IF #_w25 THEN "TRIGGER" := TRUE; END_IF;
   #_w26 := (1 <= "BUFF".PROCESS) AND ("BUFF".PROCESS <= 35) AND ("IEC_Counter_0_DB".CV = 28);
   IF #_w26 THEN "REVAMP".L30 := "SET VALUE"."STERILE TEMP2"; END_IF;
   #_w27 := #_w26 AND NOT "AUXILIARY".PULSE[25];   // rising edge
   "AUXILIARY".PULSE[25] := #_w26;
   IF #_w27 THEN "TRIGGER" := TRUE; END_IF;
   #_w28 := (1 <= "BUFF".PROCESS) AND ("BUFF".PROCESS <= 35) AND ("IEC_Counter_0_DB".CV = 29);
   IF #_w28 THEN "REVAMP".L30 := "SET VALUE"."STERILE HOLD2"; END_IF;
   #_w29 := #_w28 AND NOT "AUXILIARY".PULSE[26];   // rising edge
   "AUXILIARY".PULSE[26] := #_w28;
   IF #_w29 THEN "TRIGGER" := TRUE; END_IF;
   #_w30 := (1 <= "BUFF".PROCESS) AND ("BUFF".PROCESS <= 35) AND ("IEC_Counter_0_DB".CV = 30);
   IF #_w30 THEN "REVAMP".L30 := "SET VALUE"."STERILE TEMP3"; END_IF;
   #_w31 := #_w30 AND NOT "AUXILIARY".PULSE[27];   // rising edge
   "AUXILIARY".PULSE[27] := #_w30;
   IF #_w31 THEN "TRIGGER" := TRUE; END_IF;
   #_w32 := (1 <= "BUFF".PROCESS) AND ("BUFF".PROCESS <= 35) AND ("IEC_Counter_0_DB".CV = 31);
   IF #_w32 THEN "REVAMP".L30 := "SET VALUE"."STERILE HOLD3"; END_IF;
   #_w33 := #_w32 AND NOT "AUXILIARY".PULSE[28];   // rising edge
   "AUXILIARY".PULSE[28] := #_w32;
   IF #_w33 THEN "TRIGGER" := TRUE; END_IF;
   #_w34 := (1 <= "BUFF".PROCESS) AND ("BUFF".PROCESS <= 35) AND ("IEC_Counter_0_DB".CV = 32);
   IF #_w34 THEN "REVAMP".L30 := "SET VALUE"."STERILE TEMP4"; END_IF;
   #_w35 := #_w34 AND NOT "AUXILIARY".PULSE[29];   // rising edge
   "AUXILIARY".PULSE[29] := #_w34;
   IF #_w35 THEN "TRIGGER" := TRUE; END_IF;
   #_w36 := (1 <= "BUFF".PROCESS) AND ("BUFF".PROCESS <= 35) AND ("IEC_Counter_0_DB".CV = 33);
   IF #_w36 THEN "REVAMP".L30 := "SET VALUE"."STERILE HOLD4"; END_IF;
   #_w37 := #_w36 AND NOT "AUXILIARY".PULSE[30];   // rising edge
   "AUXILIARY".PULSE[30] := #_w36;
   IF #_w37 THEN "TRIGGER" := TRUE; END_IF;
   #_w38 := (1 <= "BUFF".PROCESS) AND ("BUFF".PROCESS <= 35);
   #_w39 := #_w38 AND ("IEC_Counter_0_DB".CV = 38);
   IF #_w39 THEN "REVAMP".L30 := "SET VALUE"."OVERSHOOT TEMP"; END_IF;
   #_w40 := #_w39 AND NOT "pulse3";   // rising edge
   "pulse3" := #_w39;
   IF #_w40 THEN "TRIGGER" := TRUE; END_IF;
   #_w41 := #_w38 AND ("IEC_Counter_0_DB".CV = 39);
   IF #_w41 THEN "REVAMP".L30 := "SET VALUE"."ABORT TEMP"; END_IF;
   #_w42 := #_w41 AND NOT "pulse14";   // rising edge
   "pulse14" := #_w41;
   IF #_w42 THEN "TRIGGER" := TRUE; END_IF;
   #_w43 := #_w38 AND ("IEC_Counter_0_DB".CV = 40);
   IF #_w43 THEN "REVAMP".L30 := "SET VALUE"."ABORT DELAY"; END_IF;
   #_w44 := #_w43 AND NOT "pulse15";   // rising edge
   "pulse15" := #_w43;
   IF #_w44 THEN "TRIGGER" := TRUE; END_IF;
   #_w45 := (1 <= "BUFF".PROCESS) AND ("BUFF".PROCESS <= 35) AND ("IEC_Counter_0_DB".CV = 34);
   IF #_w45 THEN "REVAMP".L30 := "SET VALUE"."STERILE EXH PRESS"; END_IF;
   #_w46 := #_w45 AND NOT "AUXILIARY".PULSE[31];   // rising edge
   "AUXILIARY".PULSE[31] := #_w45;
   IF #_w46 THEN "TRIGGER" := TRUE; END_IF;
   #_w47 := (1 <= "BUFF".PROCESS) AND ("BUFF".PROCESS <= 35) AND ("IEC_Counter_0_DB".CV = 35);
   IF #_w47 THEN "REVAMP".L30 := "SET VALUE"."DRY VCC"; END_IF;
   #_w48 := #_w47 AND NOT "AUXILIARY".pulse2[30];   // rising edge
   "AUXILIARY".pulse2[30] := #_w47;
   IF #_w48 THEN "TRIGGER" := TRUE; END_IF;
   #_w49 := (1 <= "BUFF".PROCESS) AND ("BUFF".PROCESS <= 35) AND ("IEC_Counter_0_DB".CV = 36);
   IF #_w49 THEN "REVAMP".L30 := "SET VALUE"."DRY TIME"; END_IF;
   #_w50 := #_w49 AND NOT "AUXILIARY".pulse2[31];   // rising edge
   "AUXILIARY".pulse2[31] := #_w49;
   IF #_w50 THEN "TRIGGER" := TRUE; END_IF;
   #_w51 := (1 <= "BUFF".PROCESS) AND ("BUFF".PROCESS <= 35) AND ("IEC_Counter_0_DB".CV = 37);
   IF #_w51 THEN "REVAMP".L30 := "SET VALUE"."DRY ATS PRESSURE"; END_IF;
   #_w52 := #_w51 AND NOT "AUXILIARY".PULSE[32];   // rising edge
   "AUXILIARY".PULSE[32] := #_w51;
   IF #_w52 THEN "TRIGGER" := TRUE; END_IF;
   #_w53 := NOT "AlwaysTRUE" AND (1 <= "BUFF".PROCESS) AND ("BUFF".PROCESS <= 35) AND ("IEC_Counter_0_DB".CV = 36);
   IF #_w53 THEN "REVAMP".L30 := "SET VALUE"."DRY TIME"; END_IF;
   #_w54 := #_w53 AND NOT "AUXILIARY".PULSE[33];   // rising edge
   "AUXILIARY".PULSE[33] := #_w53;
   IF #_w54 THEN "TRIGGER" := TRUE; END_IF;
END_REGION

REGION Network 8
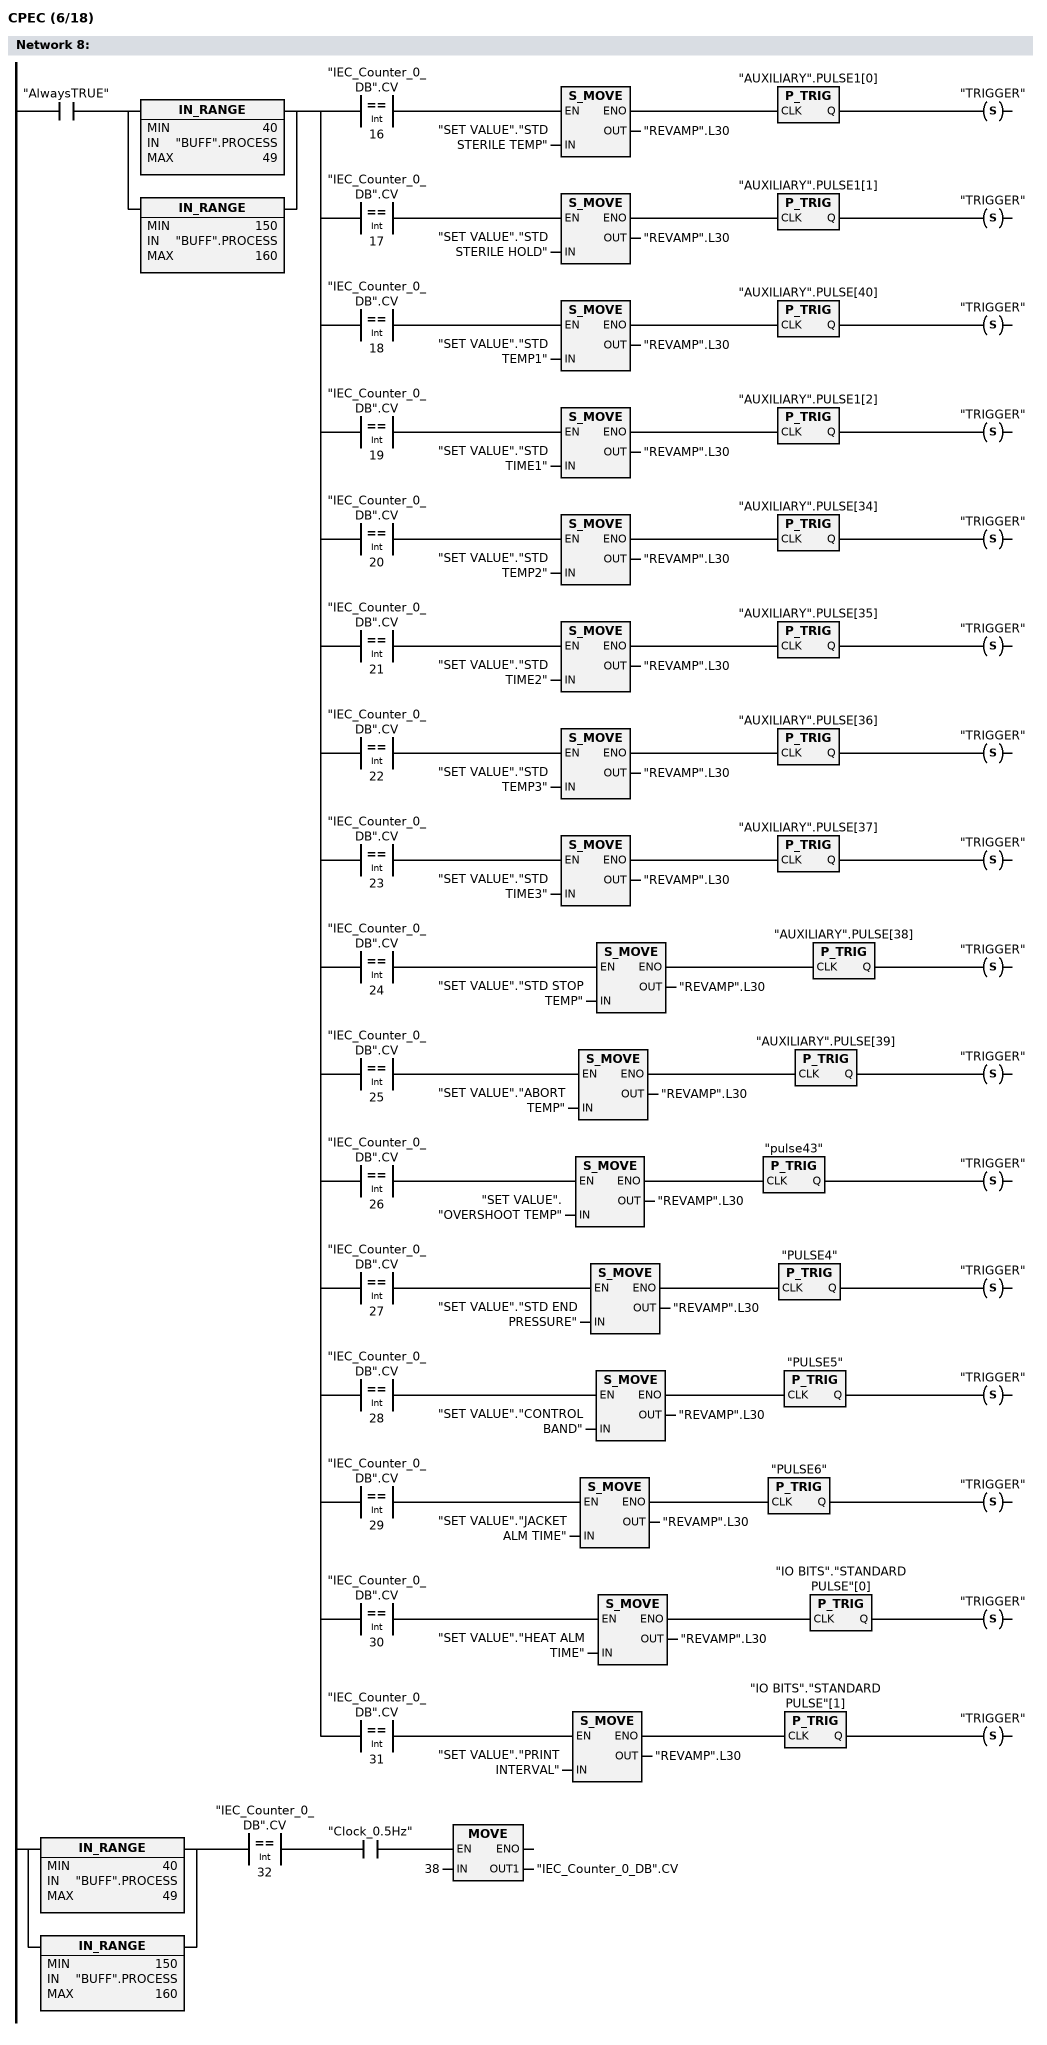
   RUNG wire#powerrail
      Contact( "AlwaysTRUE" )
      wire#w1
      { S7_Templates := "SrcType := Int" } InRange(min := 40, in := "BUFF".PROCESS, max := 49)
      wire#w2
      { S7_Templates := "SrcType := Int" } EQ_Contact(in1 := "IEC_Counter_0_DB".CV, in2 := 16)
      S_Move(in := "SET VALUE"."STD STERILE TEMP", out => "REVAMP".L30)
      P_Trig( "AUXILIARY".PULSE1[0] )
      S_Coil( "TRIGGER" )
   END_RUNG
   RUNG wire#w1
      { S7_Templates := "SrcType := Int" } InRange(min := 150, in := "BUFF".PROCESS, max := 160)
   END_RUNG wire#w2
   RUNG wire#w2
      { S7_Templates := "SrcType := Int" } EQ_Contact(in1 := "IEC_Counter_0_DB".CV, in2 := 17)
      S_Move(in := "SET VALUE"."STD STERILE HOLD", out => "REVAMP".L30)
      P_Trig( "AUXILIARY".PULSE1[1] )
      S_Coil( "TRIGGER" )
   END_RUNG
   RUNG wire#w2
      { S7_Templates := "SrcType := Int" } EQ_Contact(in1 := "IEC_Counter_0_DB".CV, in2 := 18)
      S_Move(in := "SET VALUE"."STD TEMP1", out => "REVAMP".L30)
      P_Trig( "AUXILIARY".PULSE[40] )
      S_Coil( "TRIGGER" )
   END_RUNG
   RUNG wire#w2
      { S7_Templates := "SrcType := Int" } EQ_Contact(in1 := "IEC_Counter_0_DB".CV, in2 := 19)
      S_Move(in := "SET VALUE"."STD TIME1", out => "REVAMP".L30)
      P_Trig( "AUXILIARY".PULSE1[2] )
      S_Coil( "TRIGGER" )
   END_RUNG
   RUNG wire#w2
      { S7_Templates := "SrcType := Int" } EQ_Contact(in1 := "IEC_Counter_0_DB".CV, in2 := 20)
      S_Move(in := "SET VALUE"."STD TEMP2", out => "REVAMP".L30)
      P_Trig( "AUXILIARY".PULSE[34] )
      S_Coil( "TRIGGER" )
   END_RUNG
   RUNG wire#w2
      { S7_Templates := "SrcType := Int" } EQ_Contact(in1 := "IEC_Counter_0_DB".CV, in2 := 21)
      S_Move(in := "SET VALUE"."STD TIME2", out => "REVAMP".L30)
      P_Trig( "AUXILIARY".PULSE[35] )
      S_Coil( "TRIGGER" )
   END_RUNG
   RUNG wire#w2
      { S7_Templates := "SrcType := Int" } EQ_Contact(in1 := "IEC_Counter_0_DB".CV, in2 := 22)
      S_Move(in := "SET VALUE"."STD TEMP3", out => "REVAMP".L30)
      P_Trig( "AUXILIARY".PULSE[36] )
      S_Coil( "TRIGGER" )
   END_RUNG
   RUNG wire#w2
      { S7_Templates := "SrcType := Int" } EQ_Contact(in1 := "IEC_Counter_0_DB".CV, in2 := 23)
      S_Move(in := "SET VALUE"."STD TIME3", out => "REVAMP".L30)
      P_Trig( "AUXILIARY".PULSE[37] )
      S_Coil( "TRIGGER" )
   END_RUNG
   RUNG wire#w2
      { S7_Templates := "SrcType := Int" } EQ_Contact(in1 := "IEC_Counter_0_DB".CV, in2 := 24)
      S_Move(in := "SET VALUE"."STD STOP TEMP", out => "REVAMP".L30)
      P_Trig( "AUXILIARY".PULSE[38] )
      S_Coil( "TRIGGER" )
   END_RUNG
   RUNG wire#w2
      { S7_Templates := "SrcType := Int" } EQ_Contact(in1 := "IEC_Counter_0_DB".CV, in2 := 25)
      S_Move(in := "SET VALUE"."ABORT TEMP", out => "REVAMP".L30)
      P_Trig( "AUXILIARY".PULSE[39] )
      S_Coil( "TRIGGER" )
   END_RUNG
   RUNG wire#w2
      { S7_Templates := "SrcType := Int" } EQ_Contact(in1 := "IEC_Counter_0_DB".CV, in2 := 26)
      S_Move(in := "SET VALUE"."OVERSHOOT TEMP", out => "REVAMP".L30)
      P_Trig( "pulse43" )
      S_Coil( "TRIGGER" )
   END_RUNG
   RUNG wire#w2
      { S7_Templates := "SrcType := Int" } EQ_Contact(in1 := "IEC_Counter_0_DB".CV, in2 := 27)
      S_Move(in := "SET VALUE"."STD END PRESSURE", out => "REVAMP".L30)
      P_Trig( "PULSE4" )
      S_Coil( "TRIGGER" )
   END_RUNG
   RUNG wire#w2
      { S7_Templates := "SrcType := Int" } EQ_Contact(in1 := "IEC_Counter_0_DB".CV, in2 := 28)
      S_Move(in := "SET VALUE"."CONTROL BAND", out => "REVAMP".L30)
      P_Trig( "PULSE5" )
      S_Coil( "TRIGGER" )
   END_RUNG
   RUNG wire#w2
      { S7_Templates := "SrcType := Int" } EQ_Contact(in1 := "IEC_Counter_0_DB".CV, in2 := 29)
      S_Move(in := "SET VALUE"."JACKET ALM TIME", out => "REVAMP".L30)
      P_Trig( "PULSE6" )
      S_Coil( "TRIGGER" )
   END_RUNG
   RUNG wire#w2
      { S7_Templates := "SrcType := Int" } EQ_Contact(in1 := "IEC_Counter_0_DB".CV, in2 := 30)
      S_Move(in := "SET VALUE"."HEAT ALM TIME", out => "REVAMP".L30)
      P_Trig( "IO BITS"."STANDARD PULSE"[0] )
      S_Coil( "TRIGGER" )
   END_RUNG
   RUNG wire#w2
      { S7_Templates := "SrcType := Int" } EQ_Contact(in1 := "IEC_Counter_0_DB".CV, in2 := 31)
      S_Move(in := "SET VALUE"."PRINT INTERVAL", out => "REVAMP".L30)
      P_Trig( "IO BITS"."STANDARD PULSE"[1] )
      S_Coil( "TRIGGER" )
   END_RUNG
   RUNG wire#powerrail
      { S7_Templates := "SrcType := Int" } InRange(min := 40, in := "BUFF".PROCESS, max := 49)
      wire#w3
      { S7_Templates := "SrcType := Int" } EQ_Contact(in1 := "IEC_Counter_0_DB".CV, in2 := 32)
      Contact( "Clock_0.5Hz" )
      Move(in := 38, out1 => "IEC_Counter_0_DB".CV)
   END_RUNG
   RUNG wire#powerrail
      { S7_Templates := "SrcType := Int" } InRange(min := 150, in := "BUFF".PROCESS, max := 160)
   END_RUNG wire#w3
   // the same network as SCL:
   #_w1 := "AlwaysTRUE" AND (((40 <= "BUFF".PROCESS) AND ("BUFF".PROCESS <= 49)) OR ((150 <= "BUFF".PROCESS) AND ("BUFF".PROCESS <= 160)));
   #_w2 := #_w1 AND ("IEC_Counter_0_DB".CV = 16);
   IF #_w2 THEN "REVAMP".L30 := "SET VALUE"."STD STERILE TEMP"; END_IF;
   #_w3 := #_w2 AND NOT "AUXILIARY".PULSE1[0];   // rising edge
   "AUXILIARY".PULSE1[0] := #_w2;
   IF #_w3 THEN "TRIGGER" := TRUE; END_IF;
   #_w4 := #_w1 AND ("IEC_Counter_0_DB".CV = 17);
   IF #_w4 THEN "REVAMP".L30 := "SET VALUE"."STD STERILE HOLD"; END_IF;
   #_w5 := #_w4 AND NOT "AUXILIARY".PULSE1[1];   // rising edge
   "AUXILIARY".PULSE1[1] := #_w4;
   IF #_w5 THEN "TRIGGER" := TRUE; END_IF;
   #_w6 := #_w1 AND ("IEC_Counter_0_DB".CV = 18);
   IF #_w6 THEN "REVAMP".L30 := "SET VALUE"."STD TEMP1"; END_IF;
   #_w7 := #_w6 AND NOT "AUXILIARY".PULSE[40];   // rising edge
   "AUXILIARY".PULSE[40] := #_w6;
   IF #_w7 THEN "TRIGGER" := TRUE; END_IF;
   #_w8 := #_w1 AND ("IEC_Counter_0_DB".CV = 19);
   IF #_w8 THEN "REVAMP".L30 := "SET VALUE"."STD TIME1"; END_IF;
   #_w9 := #_w8 AND NOT "AUXILIARY".PULSE1[2];   // rising edge
   "AUXILIARY".PULSE1[2] := #_w8;
   IF #_w9 THEN "TRIGGER" := TRUE; END_IF;
   #_w10 := #_w1 AND ("IEC_Counter_0_DB".CV = 20);
   IF #_w10 THEN "REVAMP".L30 := "SET VALUE"."STD TEMP2"; END_IF;
   #_w11 := #_w10 AND NOT "AUXILIARY".PULSE[34];   // rising edge
   "AUXILIARY".PULSE[34] := #_w10;
   IF #_w11 THEN "TRIGGER" := TRUE; END_IF;
   #_w12 := #_w1 AND ("IEC_Counter_0_DB".CV = 21);
   IF #_w12 THEN "REVAMP".L30 := "SET VALUE"."STD TIME2"; END_IF;
   #_w13 := #_w12 AND NOT "AUXILIARY".PULSE[35];   // rising edge
   "AUXILIARY".PULSE[35] := #_w12;
   IF #_w13 THEN "TRIGGER" := TRUE; END_IF;
   #_w14 := #_w1 AND ("IEC_Counter_0_DB".CV = 22);
   IF #_w14 THEN "REVAMP".L30 := "SET VALUE"."STD TEMP3"; END_IF;
   #_w15 := #_w14 AND NOT "AUXILIARY".PULSE[36];   // rising edge
   "AUXILIARY".PULSE[36] := #_w14;
   IF #_w15 THEN "TRIGGER" := TRUE; END_IF;
   #_w16 := #_w1 AND ("IEC_Counter_0_DB".CV = 23);
   IF #_w16 THEN "REVAMP".L30 := "SET VALUE"."STD TIME3"; END_IF;
   #_w17 := #_w16 AND NOT "AUXILIARY".PULSE[37];   // rising edge
   "AUXILIARY".PULSE[37] := #_w16;
   IF #_w17 THEN "TRIGGER" := TRUE; END_IF;
   #_w18 := #_w1 AND ("IEC_Counter_0_DB".CV = 24);
   IF #_w18 THEN "REVAMP".L30 := "SET VALUE"."STD STOP TEMP"; END_IF;
   #_w19 := #_w18 AND NOT "AUXILIARY".PULSE[38];   // rising edge
   "AUXILIARY".PULSE[38] := #_w18;
   IF #_w19 THEN "TRIGGER" := TRUE; END_IF;
   #_w20 := #_w1 AND ("IEC_Counter_0_DB".CV = 25);
   IF #_w20 THEN "REVAMP".L30 := "SET VALUE"."ABORT TEMP"; END_IF;
   #_w21 := #_w20 AND NOT "AUXILIARY".PULSE[39];   // rising edge
   "AUXILIARY".PULSE[39] := #_w20;
   IF #_w21 THEN "TRIGGER" := TRUE; END_IF;
   #_w22 := #_w1 AND ("IEC_Counter_0_DB".CV = 26);
   IF #_w22 THEN "REVAMP".L30 := "SET VALUE"."OVERSHOOT TEMP"; END_IF;
   #_w23 := #_w22 AND NOT "pulse43";   // rising edge
   "pulse43" := #_w22;
   IF #_w23 THEN "TRIGGER" := TRUE; END_IF;
   #_w24 := #_w1 AND ("IEC_Counter_0_DB".CV = 27);
   IF #_w24 THEN "REVAMP".L30 := "SET VALUE"."STD END PRESSURE"; END_IF;
   #_w25 := #_w24 AND NOT "PULSE4";   // rising edge
   "PULSE4" := #_w24;
   IF #_w25 THEN "TRIGGER" := TRUE; END_IF;
   #_w26 := #_w1 AND ("IEC_Counter_0_DB".CV = 28);
   IF #_w26 THEN "REVAMP".L30 := "SET VALUE"."CONTROL BAND"; END_IF;
   #_w27 := #_w26 AND NOT "PULSE5";   // rising edge
   "PULSE5" := #_w26;
   IF #_w27 THEN "TRIGGER" := TRUE; END_IF;
   #_w28 := #_w1 AND ("IEC_Counter_0_DB".CV = 29);
   IF #_w28 THEN "REVAMP".L30 := "SET VALUE"."JACKET ALM TIME"; END_IF;
   #_w29 := #_w28 AND NOT "PULSE6";   // rising edge
   "PULSE6" := #_w28;
   IF #_w29 THEN "TRIGGER" := TRUE; END_IF;
   #_w30 := #_w1 AND ("IEC_Counter_0_DB".CV = 30);
   IF #_w30 THEN "REVAMP".L30 := "SET VALUE"."HEAT ALM TIME"; END_IF;
   #_w31 := #_w30 AND NOT "IO BITS"."STANDARD PULSE"[0];   // rising edge
   "IO BITS"."STANDARD PULSE"[0] := #_w30;
   IF #_w31 THEN "TRIGGER" := TRUE; END_IF;
   #_w32 := #_w1 AND ("IEC_Counter_0_DB".CV = 31);
   IF #_w32 THEN "REVAMP".L30 := "SET VALUE"."PRINT INTERVAL"; END_IF;
   #_w33 := #_w32 AND NOT "IO BITS"."STANDARD PULSE"[1];   // rising edge
   "IO BITS"."STANDARD PULSE"[1] := #_w32;
   IF #_w33 THEN "TRIGGER" := TRUE; END_IF;
   IF (((40 <= "BUFF".PROCESS) AND ("BUFF".PROCESS <= 49)) OR ((150 <= "BUFF".PROCESS) AND ("BUFF".PROCESS <= 160))) AND ("IEC_Counter_0_DB".CV = 32) AND "Clock_0.5Hz" THEN
       "IEC_Counter_0_DB".CV := 38;
   END_IF;
END_REGION

REGION Network 9
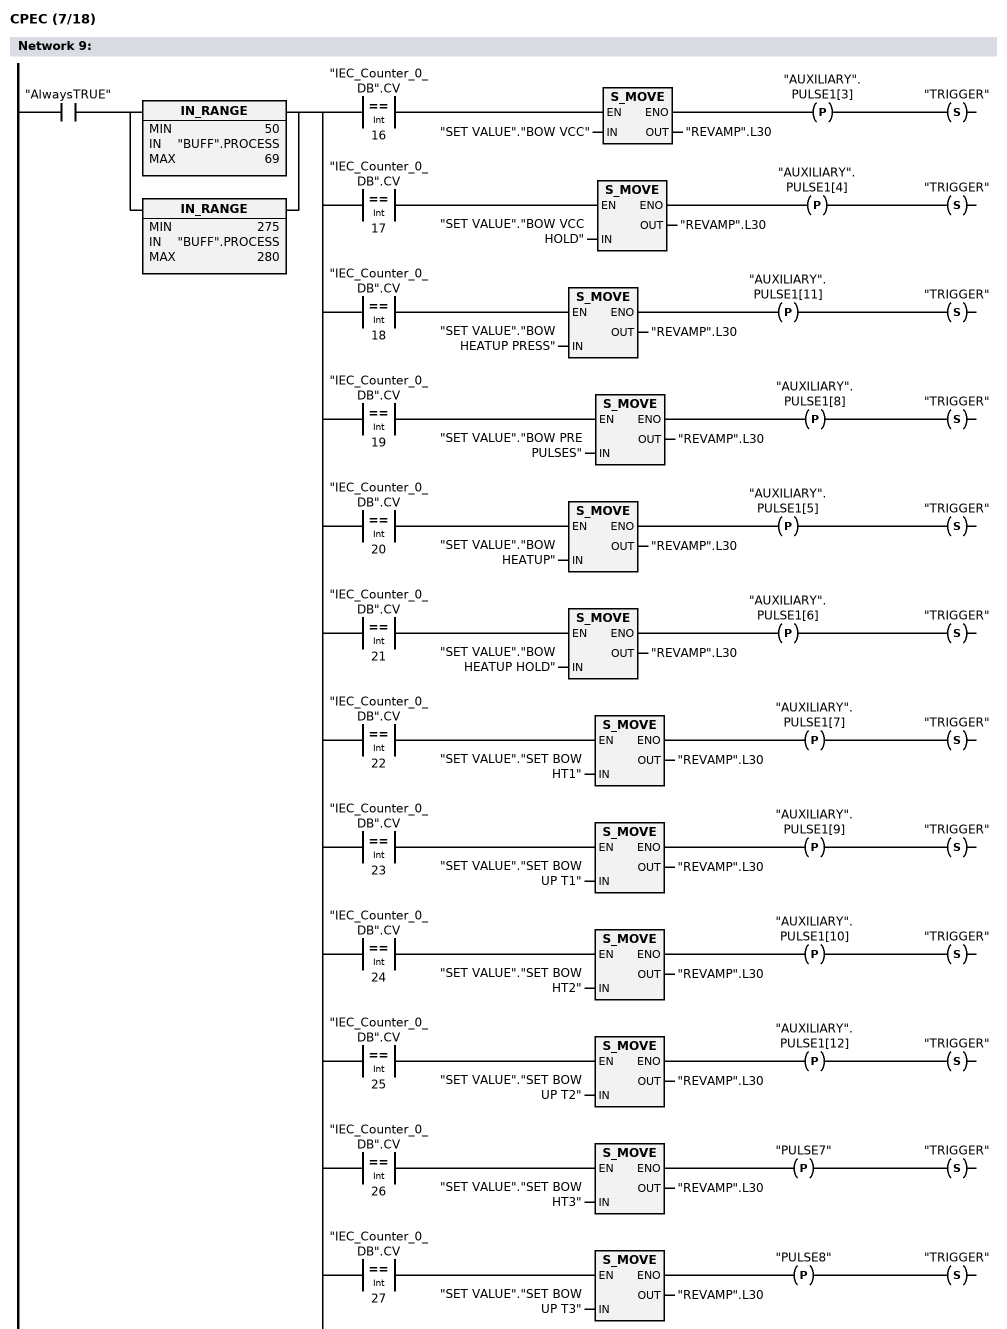
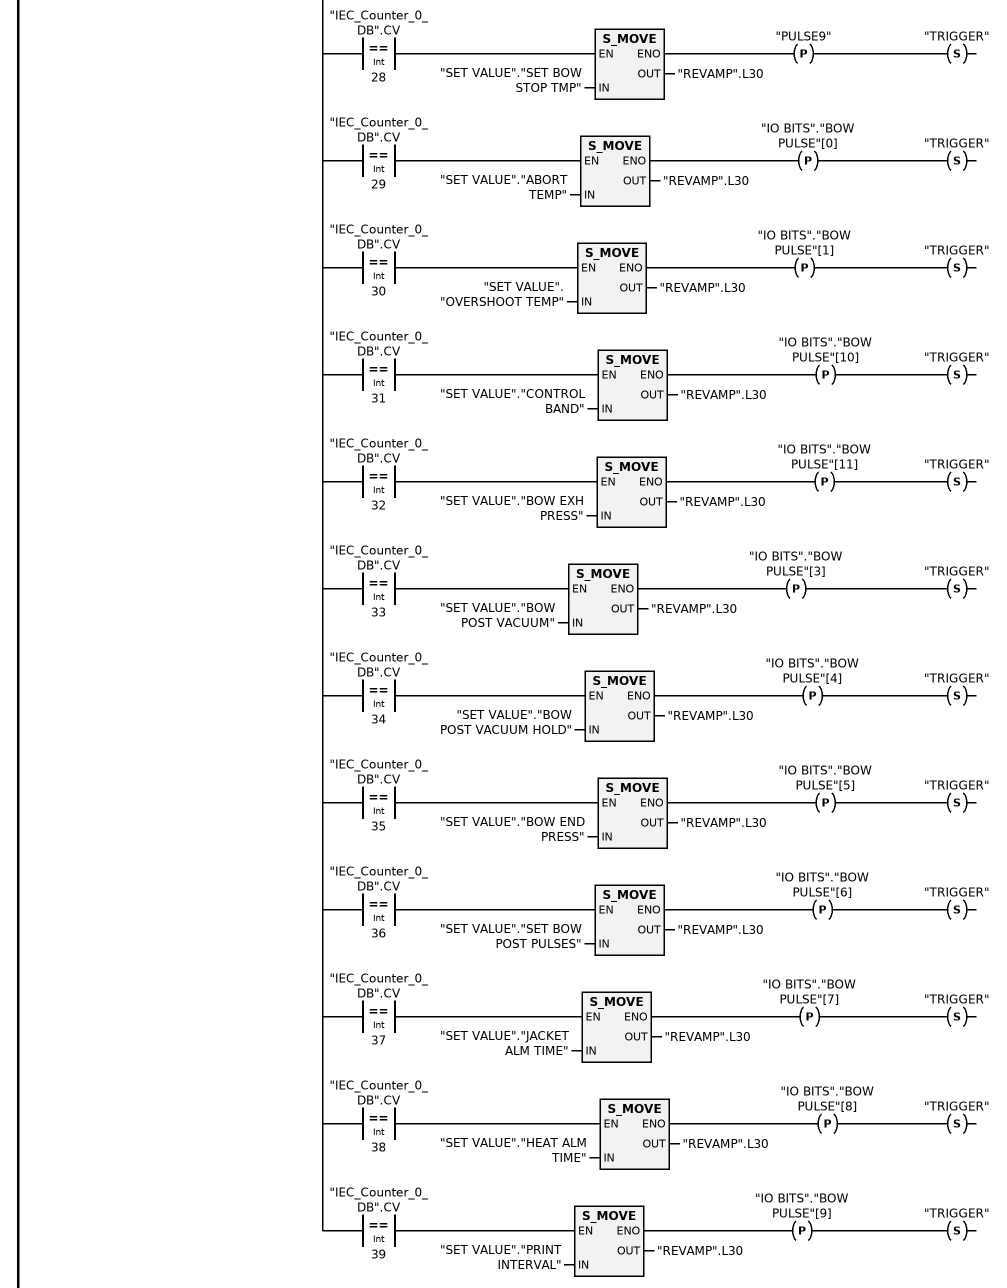
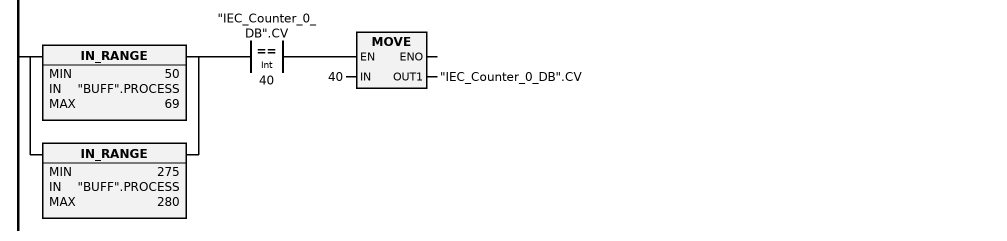
   RUNG wire#powerrail
      Contact( "AlwaysTRUE" )
      wire#w1
      { S7_Templates := "SrcType := Int" } InRange(min := 50, in := "BUFF".PROCESS, max := 69)
      wire#w2
      { S7_Templates := "SrcType := Int" } EQ_Contact(in1 := "IEC_Counter_0_DB".CV, in2 := 16)
      S_Move(in := "SET VALUE"."BOW VCC", out => "REVAMP".L30)
      P_Trig( "AUXILIARY".PULSE1[3] )
      S_Coil( "TRIGGER" )
   END_RUNG
   RUNG wire#w1
      { S7_Templates := "SrcType := Int" } InRange(min := 275, in := "BUFF".PROCESS, max := 280)
   END_RUNG wire#w2
   RUNG wire#w2
      { S7_Templates := "SrcType := Int" } EQ_Contact(in1 := "IEC_Counter_0_DB".CV, in2 := 17)
      S_Move(in := "SET VALUE"."BOW VCC HOLD", out => "REVAMP".L30)
      P_Trig( "AUXILIARY".PULSE1[4] )
      S_Coil( "TRIGGER" )
   END_RUNG
   RUNG wire#w2
      { S7_Templates := "SrcType := Int" } EQ_Contact(in1 := "IEC_Counter_0_DB".CV, in2 := 18)
      S_Move(in := "SET VALUE"."BOW HEATUP PRESS", out => "REVAMP".L30)
      P_Trig( "AUXILIARY".PULSE1[11] )
      S_Coil( "TRIGGER" )
   END_RUNG
   RUNG wire#w2
      { S7_Templates := "SrcType := Int" } EQ_Contact(in1 := "IEC_Counter_0_DB".CV, in2 := 19)
      S_Move(in := "SET VALUE"."BOW PRE PULSES", out => "REVAMP".L30)
      P_Trig( "AUXILIARY".PULSE1[8] )
      S_Coil( "TRIGGER" )
   END_RUNG
   RUNG wire#w2
      { S7_Templates := "SrcType := Int" } EQ_Contact(in1 := "IEC_Counter_0_DB".CV, in2 := 20)
      S_Move(in := "SET VALUE"."BOW HEATUP", out => "REVAMP".L30)
      P_Trig( "AUXILIARY".PULSE1[5] )
      S_Coil( "TRIGGER" )
   END_RUNG
   RUNG wire#w2
      { S7_Templates := "SrcType := Int" } EQ_Contact(in1 := "IEC_Counter_0_DB".CV, in2 := 21)
      S_Move(in := "SET VALUE"."BOW HEATUP HOLD", out => "REVAMP".L30)
      P_Trig( "AUXILIARY".PULSE1[6] )
      S_Coil( "TRIGGER" )
   END_RUNG
   RUNG wire#w2
      { S7_Templates := "SrcType := Int" } EQ_Contact(in1 := "IEC_Counter_0_DB".CV, in2 := 22)
      S_Move(in := "SET VALUE"."SET BOW HT1", out => "REVAMP".L30)
      P_Trig( "AUXILIARY".PULSE1[7] )
      S_Coil( "TRIGGER" )
   END_RUNG
   RUNG wire#w2
      { S7_Templates := "SrcType := Int" } EQ_Contact(in1 := "IEC_Counter_0_DB".CV, in2 := 23)
      S_Move(in := "SET VALUE"."SET BOW UP T1", out => "REVAMP".L30)
      P_Trig( "AUXILIARY".PULSE1[9] )
      S_Coil( "TRIGGER" )
   END_RUNG
   RUNG wire#w2
      { S7_Templates := "SrcType := Int" } EQ_Contact(in1 := "IEC_Counter_0_DB".CV, in2 := 24)
      S_Move(in := "SET VALUE"."SET BOW HT2", out => "REVAMP".L30)
      P_Trig( "AUXILIARY".PULSE1[10] )
      S_Coil( "TRIGGER" )
   END_RUNG
   RUNG wire#w2
      { S7_Templates := "SrcType := Int" } EQ_Contact(in1 := "IEC_Counter_0_DB".CV, in2 := 25)
      S_Move(in := "SET VALUE"."SET BOW UP T2", out => "REVAMP".L30)
      P_Trig( "AUXILIARY".PULSE1[12] )
      S_Coil( "TRIGGER" )
   END_RUNG
   RUNG wire#w2
      { S7_Templates := "SrcType := Int" } EQ_Contact(in1 := "IEC_Counter_0_DB".CV, in2 := 26)
      S_Move(in := "SET VALUE"."SET BOW HT3", out => "REVAMP".L30)
      P_Trig( "PULSE7" )
      S_Coil( "TRIGGER" )
   END_RUNG
   RUNG wire#w2
      { S7_Templates := "SrcType := Int" } EQ_Contact(in1 := "IEC_Counter_0_DB".CV, in2 := 27)
      S_Move(in := "SET VALUE"."SET BOW UP T3", out => "REVAMP".L30)
      P_Trig( "PULSE8" )
      S_Coil( "TRIGGER" )
   END_RUNG
   RUNG wire#w2
      { S7_Templates := "SrcType := Int" } EQ_Contact(in1 := "IEC_Counter_0_DB".CV, in2 := 28)
      S_Move(in := "SET VALUE"."SET BOW STOP TMP", out => "REVAMP".L30)
      P_Trig( "PULSE9" )
      S_Coil( "TRIGGER" )
   END_RUNG
   RUNG wire#w2
      { S7_Templates := "SrcType := Int" } EQ_Contact(in1 := "IEC_Counter_0_DB".CV, in2 := 29)
      S_Move(in := "SET VALUE"."ABORT TEMP", out => "REVAMP".L30)
      P_Trig( "IO BITS"."BOW PULSE"[0] )
      S_Coil( "TRIGGER" )
   END_RUNG
   RUNG wire#w2
      { S7_Templates := "SrcType := Int" } EQ_Contact(in1 := "IEC_Counter_0_DB".CV, in2 := 30)
      S_Move(in := "SET VALUE"."OVERSHOOT TEMP", out => "REVAMP".L30)
      P_Trig( "IO BITS"."BOW PULSE"[1] )
      S_Coil( "TRIGGER" )
   END_RUNG
   RUNG wire#w2
      { S7_Templates := "SrcType := Int" } EQ_Contact(in1 := "IEC_Counter_0_DB".CV, in2 := 31)
      S_Move(in := "SET VALUE"."CONTROL BAND", out => "REVAMP".L30)
      P_Trig( "IO BITS"."BOW PULSE"[10] )
      S_Coil( "TRIGGER" )
   END_RUNG
   RUNG wire#w2
      { S7_Templates := "SrcType := Int" } EQ_Contact(in1 := "IEC_Counter_0_DB".CV, in2 := 32)
      S_Move(in := "SET VALUE"."BOW EXH PRESS", out => "REVAMP".L30)
      P_Trig( "IO BITS"."BOW PULSE"[11] )
      S_Coil( "TRIGGER" )
   END_RUNG
   RUNG wire#w2
      { S7_Templates := "SrcType := Int" } EQ_Contact(in1 := "IEC_Counter_0_DB".CV, in2 := 33)
      S_Move(in := "SET VALUE"."BOW POST VACUUM", out => "REVAMP".L30)
      P_Trig( "IO BITS"."BOW PULSE"[3] )
      S_Coil( "TRIGGER" )
   END_RUNG
   RUNG wire#w2
      { S7_Templates := "SrcType := Int" } EQ_Contact(in1 := "IEC_Counter_0_DB".CV, in2 := 34)
      S_Move(in := "SET VALUE"."BOW POST VACUUM HOLD", out => "REVAMP".L30)
      P_Trig( "IO BITS"."BOW PULSE"[4] )
      S_Coil( "TRIGGER" )
   END_RUNG
   RUNG wire#w2
      { S7_Templates := "SrcType := Int" } EQ_Contact(in1 := "IEC_Counter_0_DB".CV, in2 := 35)
      S_Move(in := "SET VALUE"."BOW END PRESS", out => "REVAMP".L30)
      P_Trig( "IO BITS"."BOW PULSE"[5] )
      S_Coil( "TRIGGER" )
   END_RUNG
   RUNG wire#w2
      { S7_Templates := "SrcType := Int" } EQ_Contact(in1 := "IEC_Counter_0_DB".CV, in2 := 36)
      S_Move(in := "SET VALUE"."SET BOW POST PULSES", out => "REVAMP".L30)
      P_Trig( "IO BITS"."BOW PULSE"[6] )
      S_Coil( "TRIGGER" )
   END_RUNG
   RUNG wire#w2
      { S7_Templates := "SrcType := Int" } EQ_Contact(in1 := "IEC_Counter_0_DB".CV, in2 := 37)
      S_Move(in := "SET VALUE"."JACKET ALM TIME", out => "REVAMP".L30)
      P_Trig( "IO BITS"."BOW PULSE"[7] )
      S_Coil( "TRIGGER" )
   END_RUNG
   RUNG wire#w2
      { S7_Templates := "SrcType := Int" } EQ_Contact(in1 := "IEC_Counter_0_DB".CV, in2 := 38)
      S_Move(in := "SET VALUE"."HEAT ALM TIME", out => "REVAMP".L30)
      P_Trig( "IO BITS"."BOW PULSE"[8] )
      S_Coil( "TRIGGER" )
   END_RUNG
   RUNG wire#w2
      { S7_Templates := "SrcType := Int" } EQ_Contact(in1 := "IEC_Counter_0_DB".CV, in2 := 39)
      S_Move(in := "SET VALUE"."PRINT INTERVAL", out => "REVAMP".L30)
      P_Trig( "IO BITS"."BOW PULSE"[9] )
      S_Coil( "TRIGGER" )
   END_RUNG
   RUNG wire#powerrail
      { S7_Templates := "SrcType := Int" } InRange(min := 50, in := "BUFF".PROCESS, max := 69)
      wire#w3
      { S7_Templates := "SrcType := Int" } EQ_Contact(in1 := "IEC_Counter_0_DB".CV, in2 := 40)
      Move(in := 40, out1 => "IEC_Counter_0_DB".CV)
   END_RUNG
   RUNG wire#powerrail
      { S7_Templates := "SrcType := Int" } InRange(min := 275, in := "BUFF".PROCESS, max := 280)
   END_RUNG wire#w3
   // the same network as SCL:
   #_w1 := "AlwaysTRUE" AND (((50 <= "BUFF".PROCESS) AND ("BUFF".PROCESS <= 69)) OR ((275 <= "BUFF".PROCESS) AND ("BUFF".PROCESS <= 280)));
   #_w2 := #_w1 AND ("IEC_Counter_0_DB".CV = 16);
   IF #_w2 THEN "REVAMP".L30 := "SET VALUE"."BOW VCC"; END_IF;
   #_w3 := #_w2 AND NOT "AUXILIARY".PULSE1[3];   // rising edge
   "AUXILIARY".PULSE1[3] := #_w2;
   IF #_w3 THEN "TRIGGER" := TRUE; END_IF;
   #_w4 := #_w1 AND ("IEC_Counter_0_DB".CV = 17);
   IF #_w4 THEN "REVAMP".L30 := "SET VALUE"."BOW VCC HOLD"; END_IF;
   #_w5 := #_w4 AND NOT "AUXILIARY".PULSE1[4];   // rising edge
   "AUXILIARY".PULSE1[4] := #_w4;
   IF #_w5 THEN "TRIGGER" := TRUE; END_IF;
   #_w6 := #_w1 AND ("IEC_Counter_0_DB".CV = 18);
   IF #_w6 THEN "REVAMP".L30 := "SET VALUE"."BOW HEATUP PRESS"; END_IF;
   #_w7 := #_w6 AND NOT "AUXILIARY".PULSE1[11];   // rising edge
   "AUXILIARY".PULSE1[11] := #_w6;
   IF #_w7 THEN "TRIGGER" := TRUE; END_IF;
   #_w8 := #_w1 AND ("IEC_Counter_0_DB".CV = 19);
   IF #_w8 THEN "REVAMP".L30 := "SET VALUE"."BOW PRE PULSES"; END_IF;
   #_w9 := #_w8 AND NOT "AUXILIARY".PULSE1[8];   // rising edge
   "AUXILIARY".PULSE1[8] := #_w8;
   IF #_w9 THEN "TRIGGER" := TRUE; END_IF;
   #_w10 := #_w1 AND ("IEC_Counter_0_DB".CV = 20);
   IF #_w10 THEN "REVAMP".L30 := "SET VALUE"."BOW HEATUP"; END_IF;
   #_w11 := #_w10 AND NOT "AUXILIARY".PULSE1[5];   // rising edge
   "AUXILIARY".PULSE1[5] := #_w10;
   IF #_w11 THEN "TRIGGER" := TRUE; END_IF;
   #_w12 := #_w1 AND ("IEC_Counter_0_DB".CV = 21);
   IF #_w12 THEN "REVAMP".L30 := "SET VALUE"."BOW HEATUP HOLD"; END_IF;
   #_w13 := #_w12 AND NOT "AUXILIARY".PULSE1[6];   // rising edge
   "AUXILIARY".PULSE1[6] := #_w12;
   IF #_w13 THEN "TRIGGER" := TRUE; END_IF;
   #_w14 := #_w1 AND ("IEC_Counter_0_DB".CV = 22);
   IF #_w14 THEN "REVAMP".L30 := "SET VALUE"."SET BOW HT1"; END_IF;
   #_w15 := #_w14 AND NOT "AUXILIARY".PULSE1[7];   // rising edge
   "AUXILIARY".PULSE1[7] := #_w14;
   IF #_w15 THEN "TRIGGER" := TRUE; END_IF;
   #_w16 := #_w1 AND ("IEC_Counter_0_DB".CV = 23);
   IF #_w16 THEN "REVAMP".L30 := "SET VALUE"."SET BOW UP T1"; END_IF;
   #_w17 := #_w16 AND NOT "AUXILIARY".PULSE1[9];   // rising edge
   "AUXILIARY".PULSE1[9] := #_w16;
   IF #_w17 THEN "TRIGGER" := TRUE; END_IF;
   #_w18 := #_w1 AND ("IEC_Counter_0_DB".CV = 24);
   IF #_w18 THEN "REVAMP".L30 := "SET VALUE"."SET BOW HT2"; END_IF;
   #_w19 := #_w18 AND NOT "AUXILIARY".PULSE1[10];   // rising edge
   "AUXILIARY".PULSE1[10] := #_w18;
   IF #_w19 THEN "TRIGGER" := TRUE; END_IF;
   #_w20 := #_w1 AND ("IEC_Counter_0_DB".CV = 25);
   IF #_w20 THEN "REVAMP".L30 := "SET VALUE"."SET BOW UP T2"; END_IF;
   #_w21 := #_w20 AND NOT "AUXILIARY".PULSE1[12];   // rising edge
   "AUXILIARY".PULSE1[12] := #_w20;
   IF #_w21 THEN "TRIGGER" := TRUE; END_IF;
   #_w22 := #_w1 AND ("IEC_Counter_0_DB".CV = 26);
   IF #_w22 THEN "REVAMP".L30 := "SET VALUE"."SET BOW HT3"; END_IF;
   #_w23 := #_w22 AND NOT "PULSE7";   // rising edge
   "PULSE7" := #_w22;
   IF #_w23 THEN "TRIGGER" := TRUE; END_IF;
   #_w24 := #_w1 AND ("IEC_Counter_0_DB".CV = 27);
   IF #_w24 THEN "REVAMP".L30 := "SET VALUE"."SET BOW UP T3"; END_IF;
   #_w25 := #_w24 AND NOT "PULSE8";   // rising edge
   "PULSE8" := #_w24;
   IF #_w25 THEN "TRIGGER" := TRUE; END_IF;
   #_w26 := #_w1 AND ("IEC_Counter_0_DB".CV = 28);
   IF #_w26 THEN "REVAMP".L30 := "SET VALUE"."SET BOW STOP TMP"; END_IF;
   #_w27 := #_w26 AND NOT "PULSE9";   // rising edge
   "PULSE9" := #_w26;
   IF #_w27 THEN "TRIGGER" := TRUE; END_IF;
   #_w28 := #_w1 AND ("IEC_Counter_0_DB".CV = 29);
   IF #_w28 THEN "REVAMP".L30 := "SET VALUE"."ABORT TEMP"; END_IF;
   #_w29 := #_w28 AND NOT "IO BITS"."BOW PULSE"[0];   // rising edge
   "IO BITS"."BOW PULSE"[0] := #_w28;
   IF #_w29 THEN "TRIGGER" := TRUE; END_IF;
   #_w30 := #_w1 AND ("IEC_Counter_0_DB".CV = 30);
   IF #_w30 THEN "REVAMP".L30 := "SET VALUE"."OVERSHOOT TEMP"; END_IF;
   #_w31 := #_w30 AND NOT "IO BITS"."BOW PULSE"[1];   // rising edge
   "IO BITS"."BOW PULSE"[1] := #_w30;
   IF #_w31 THEN "TRIGGER" := TRUE; END_IF;
   #_w32 := #_w1 AND ("IEC_Counter_0_DB".CV = 31);
   IF #_w32 THEN "REVAMP".L30 := "SET VALUE"."CONTROL BAND"; END_IF;
   #_w33 := #_w32 AND NOT "IO BITS"."BOW PULSE"[10];   // rising edge
   "IO BITS"."BOW PULSE"[10] := #_w32;
   IF #_w33 THEN "TRIGGER" := TRUE; END_IF;
   #_w34 := #_w1 AND ("IEC_Counter_0_DB".CV = 32);
   IF #_w34 THEN "REVAMP".L30 := "SET VALUE"."BOW EXH PRESS"; END_IF;
   #_w35 := #_w34 AND NOT "IO BITS"."BOW PULSE"[11];   // rising edge
   "IO BITS"."BOW PULSE"[11] := #_w34;
   IF #_w35 THEN "TRIGGER" := TRUE; END_IF;
   #_w36 := #_w1 AND ("IEC_Counter_0_DB".CV = 33);
   IF #_w36 THEN "REVAMP".L30 := "SET VALUE"."BOW POST VACUUM"; END_IF;
   #_w37 := #_w36 AND NOT "IO BITS"."BOW PULSE"[3];   // rising edge
   "IO BITS"."BOW PULSE"[3] := #_w36;
   IF #_w37 THEN "TRIGGER" := TRUE; END_IF;
   #_w38 := #_w1 AND ("IEC_Counter_0_DB".CV = 34);
   IF #_w38 THEN "REVAMP".L30 := "SET VALUE"."BOW POST VACUUM HOLD"; END_IF;
   #_w39 := #_w38 AND NOT "IO BITS"."BOW PULSE"[4];   // rising edge
   "IO BITS"."BOW PULSE"[4] := #_w38;
   IF #_w39 THEN "TRIGGER" := TRUE; END_IF;
   #_w40 := #_w1 AND ("IEC_Counter_0_DB".CV = 35);
   IF #_w40 THEN "REVAMP".L30 := "SET VALUE"."BOW END PRESS"; END_IF;
   #_w41 := #_w40 AND NOT "IO BITS"."BOW PULSE"[5];   // rising edge
   "IO BITS"."BOW PULSE"[5] := #_w40;
   IF #_w41 THEN "TRIGGER" := TRUE; END_IF;
   #_w42 := #_w1 AND ("IEC_Counter_0_DB".CV = 36);
   IF #_w42 THEN "REVAMP".L30 := "SET VALUE"."SET BOW POST PULSES"; END_IF;
   #_w43 := #_w42 AND NOT "IO BITS"."BOW PULSE"[6];   // rising edge
   "IO BITS"."BOW PULSE"[6] := #_w42;
   IF #_w43 THEN "TRIGGER" := TRUE; END_IF;
   #_w44 := #_w1 AND ("IEC_Counter_0_DB".CV = 37);
   IF #_w44 THEN "REVAMP".L30 := "SET VALUE"."JACKET ALM TIME"; END_IF;
   #_w45 := #_w44 AND NOT "IO BITS"."BOW PULSE"[7];   // rising edge
   "IO BITS"."BOW PULSE"[7] := #_w44;
   IF #_w45 THEN "TRIGGER" := TRUE; END_IF;
   #_w46 := #_w1 AND ("IEC_Counter_0_DB".CV = 38);
   IF #_w46 THEN "REVAMP".L30 := "SET VALUE"."HEAT ALM TIME"; END_IF;
   #_w47 := #_w46 AND NOT "IO BITS"."BOW PULSE"[8];   // rising edge
   "IO BITS"."BOW PULSE"[8] := #_w46;
   IF #_w47 THEN "TRIGGER" := TRUE; END_IF;
   #_w48 := #_w1 AND ("IEC_Counter_0_DB".CV = 39);
   IF #_w48 THEN "REVAMP".L30 := "SET VALUE"."PRINT INTERVAL"; END_IF;
   #_w49 := #_w48 AND NOT "IO BITS"."BOW PULSE"[9];   // rising edge
   "IO BITS"."BOW PULSE"[9] := #_w48;
   IF #_w49 THEN "TRIGGER" := TRUE; END_IF;
   IF (((50 <= "BUFF".PROCESS) AND ("BUFF".PROCESS <= 69)) OR ((275 <= "BUFF".PROCESS) AND ("BUFF".PROCESS <= 280))) AND ("IEC_Counter_0_DB".CV = 40) THEN
       "IEC_Counter_0_DB".CV := 40;
   END_IF;
END_REGION

REGION Network 10
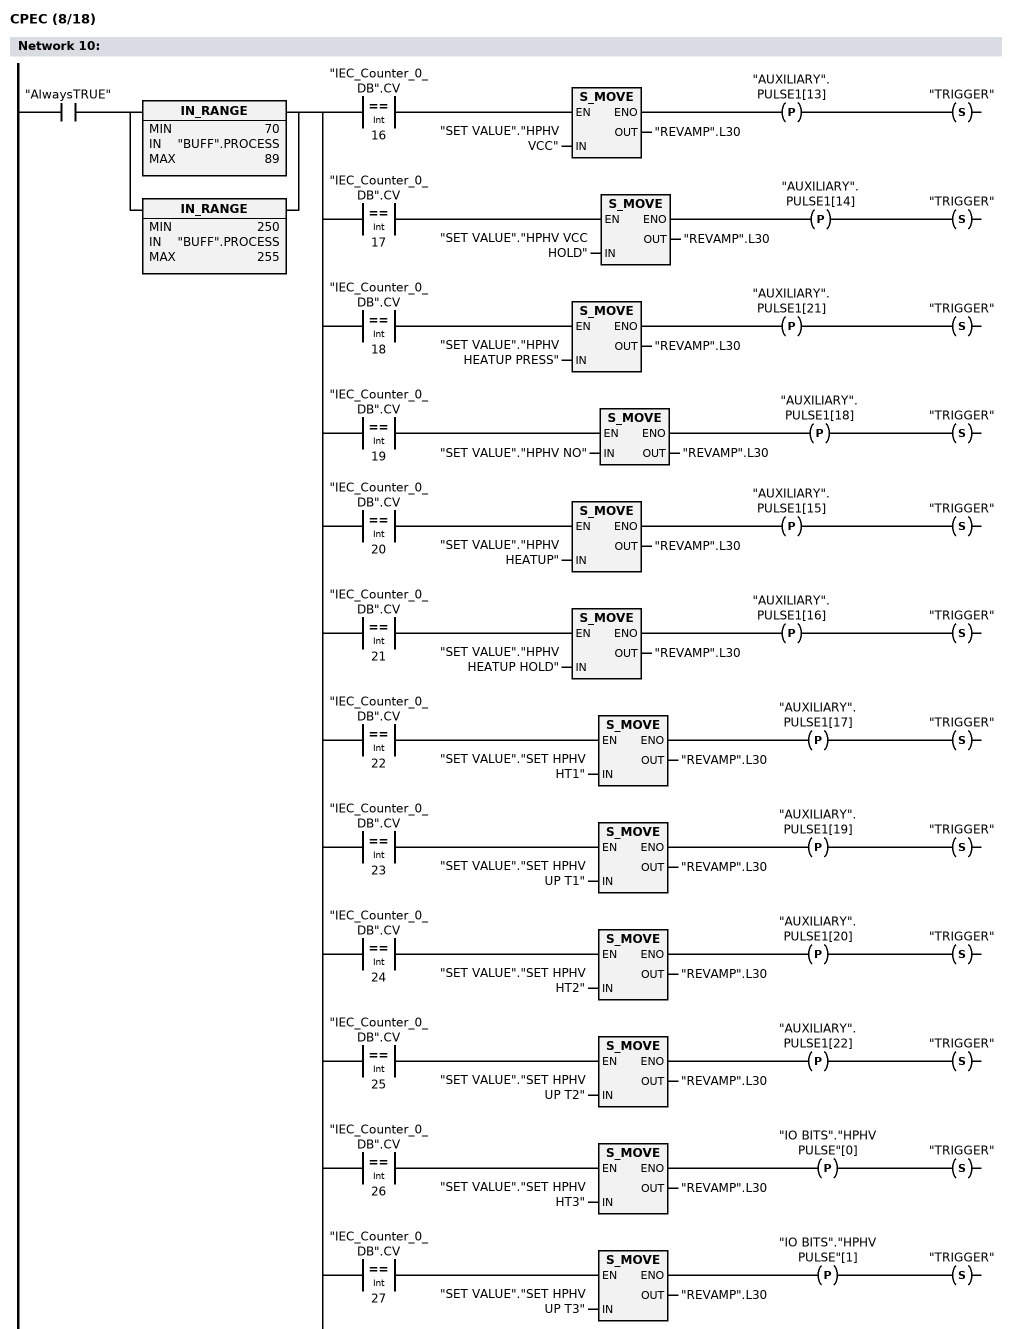
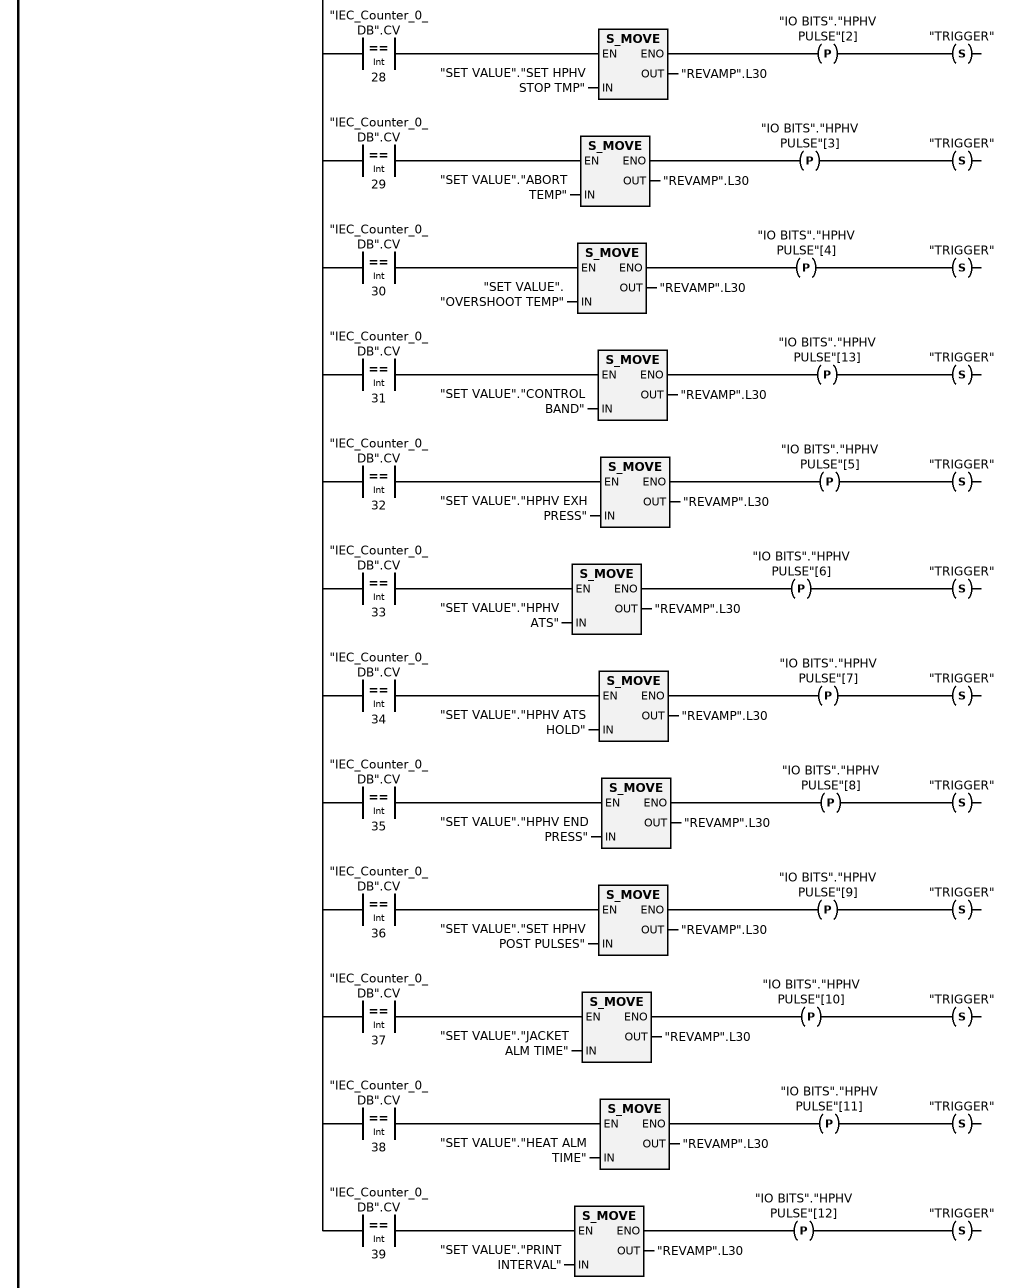
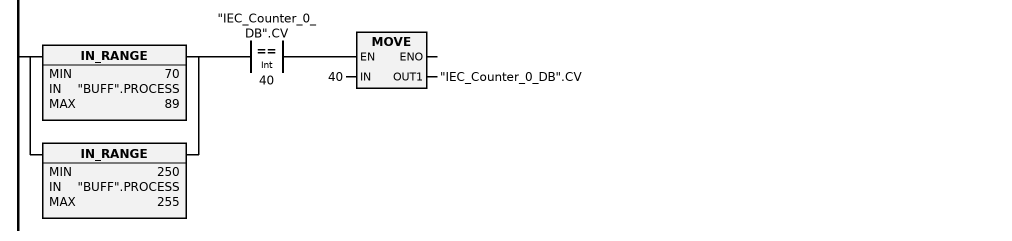
   RUNG wire#powerrail
      Contact( "AlwaysTRUE" )
      wire#w1
      { S7_Templates := "SrcType := Int" } InRange(min := 70, in := "BUFF".PROCESS, max := 89)
      wire#w2
      { S7_Templates := "SrcType := Int" } EQ_Contact(in1 := "IEC_Counter_0_DB".CV, in2 := 16)
      S_Move(in := "SET VALUE"."HPHV VCC", out => "REVAMP".L30)
      P_Trig( "AUXILIARY".PULSE1[13] )
      S_Coil( "TRIGGER" )
   END_RUNG
   RUNG wire#w1
      { S7_Templates := "SrcType := Int" } InRange(min := 250, in := "BUFF".PROCESS, max := 255)
   END_RUNG wire#w2
   RUNG wire#w2
      { S7_Templates := "SrcType := Int" } EQ_Contact(in1 := "IEC_Counter_0_DB".CV, in2 := 17)
      S_Move(in := "SET VALUE"."HPHV VCC HOLD", out => "REVAMP".L30)
      P_Trig( "AUXILIARY".PULSE1[14] )
      S_Coil( "TRIGGER" )
   END_RUNG
   RUNG wire#w2
      { S7_Templates := "SrcType := Int" } EQ_Contact(in1 := "IEC_Counter_0_DB".CV, in2 := 18)
      S_Move(in := "SET VALUE"."HPHV HEATUP PRESS", out => "REVAMP".L30)
      P_Trig( "AUXILIARY".PULSE1[21] )
      S_Coil( "TRIGGER" )
   END_RUNG
   RUNG wire#w2
      { S7_Templates := "SrcType := Int" } EQ_Contact(in1 := "IEC_Counter_0_DB".CV, in2 := 19)
      S_Move(in := "SET VALUE"."HPHV NO", out => "REVAMP".L30)
      P_Trig( "AUXILIARY".PULSE1[18] )
      S_Coil( "TRIGGER" )
   END_RUNG
   RUNG wire#w2
      { S7_Templates := "SrcType := Int" } EQ_Contact(in1 := "IEC_Counter_0_DB".CV, in2 := 20)
      S_Move(in := "SET VALUE"."HPHV HEATUP", out => "REVAMP".L30)
      P_Trig( "AUXILIARY".PULSE1[15] )
      S_Coil( "TRIGGER" )
   END_RUNG
   RUNG wire#w2
      { S7_Templates := "SrcType := Int" } EQ_Contact(in1 := "IEC_Counter_0_DB".CV, in2 := 21)
      S_Move(in := "SET VALUE"."HPHV HEATUP HOLD", out => "REVAMP".L30)
      P_Trig( "AUXILIARY".PULSE1[16] )
      S_Coil( "TRIGGER" )
   END_RUNG
   RUNG wire#w2
      { S7_Templates := "SrcType := Int" } EQ_Contact(in1 := "IEC_Counter_0_DB".CV, in2 := 22)
      S_Move(in := "SET VALUE"."SET HPHV HT1", out => "REVAMP".L30)
      P_Trig( "AUXILIARY".PULSE1[17] )
      S_Coil( "TRIGGER" )
   END_RUNG
   RUNG wire#w2
      { S7_Templates := "SrcType := Int" } EQ_Contact(in1 := "IEC_Counter_0_DB".CV, in2 := 23)
      S_Move(in := "SET VALUE"."SET HPHV UP T1", out => "REVAMP".L30)
      P_Trig( "AUXILIARY".PULSE1[19] )
      S_Coil( "TRIGGER" )
   END_RUNG
   RUNG wire#w2
      { S7_Templates := "SrcType := Int" } EQ_Contact(in1 := "IEC_Counter_0_DB".CV, in2 := 24)
      S_Move(in := "SET VALUE"."SET HPHV HT2", out => "REVAMP".L30)
      P_Trig( "AUXILIARY".PULSE1[20] )
      S_Coil( "TRIGGER" )
   END_RUNG
   RUNG wire#w2
      { S7_Templates := "SrcType := Int" } EQ_Contact(in1 := "IEC_Counter_0_DB".CV, in2 := 25)
      S_Move(in := "SET VALUE"."SET HPHV UP T2", out => "REVAMP".L30)
      P_Trig( "AUXILIARY".PULSE1[22] )
      S_Coil( "TRIGGER" )
   END_RUNG
   RUNG wire#w2
      { S7_Templates := "SrcType := Int" } EQ_Contact(in1 := "IEC_Counter_0_DB".CV, in2 := 26)
      S_Move(in := "SET VALUE"."SET HPHV HT3", out => "REVAMP".L30)
      P_Trig( "IO BITS"."HPHV PULSE"[0] )
      S_Coil( "TRIGGER" )
   END_RUNG
   RUNG wire#w2
      { S7_Templates := "SrcType := Int" } EQ_Contact(in1 := "IEC_Counter_0_DB".CV, in2 := 27)
      S_Move(in := "SET VALUE"."SET HPHV UP T3", out => "REVAMP".L30)
      P_Trig( "IO BITS"."HPHV PULSE"[1] )
      S_Coil( "TRIGGER" )
   END_RUNG
   RUNG wire#w2
      { S7_Templates := "SrcType := Int" } EQ_Contact(in1 := "IEC_Counter_0_DB".CV, in2 := 28)
      S_Move(in := "SET VALUE"."SET HPHV STOP TMP", out => "REVAMP".L30)
      P_Trig( "IO BITS"."HPHV PULSE"[2] )
      S_Coil( "TRIGGER" )
   END_RUNG
   RUNG wire#w2
      { S7_Templates := "SrcType := Int" } EQ_Contact(in1 := "IEC_Counter_0_DB".CV, in2 := 29)
      S_Move(in := "SET VALUE"."ABORT TEMP", out => "REVAMP".L30)
      P_Trig( "IO BITS"."HPHV PULSE"[3] )
      S_Coil( "TRIGGER" )
   END_RUNG
   RUNG wire#w2
      { S7_Templates := "SrcType := Int" } EQ_Contact(in1 := "IEC_Counter_0_DB".CV, in2 := 30)
      S_Move(in := "SET VALUE"."OVERSHOOT TEMP", out => "REVAMP".L30)
      P_Trig( "IO BITS"."HPHV PULSE"[4] )
      S_Coil( "TRIGGER" )
   END_RUNG
   RUNG wire#w2
      { S7_Templates := "SrcType := Int" } EQ_Contact(in1 := "IEC_Counter_0_DB".CV, in2 := 31)
      S_Move(in := "SET VALUE"."CONTROL BAND", out => "REVAMP".L30)
      P_Trig( "IO BITS"."HPHV PULSE"[13] )
      S_Coil( "TRIGGER" )
   END_RUNG
   RUNG wire#w2
      { S7_Templates := "SrcType := Int" } EQ_Contact(in1 := "IEC_Counter_0_DB".CV, in2 := 32)
      S_Move(in := "SET VALUE"."HPHV EXH PRESS", out => "REVAMP".L30)
      P_Trig( "IO BITS"."HPHV PULSE"[5] )
      S_Coil( "TRIGGER" )
   END_RUNG
   RUNG wire#w2
      { S7_Templates := "SrcType := Int" } EQ_Contact(in1 := "IEC_Counter_0_DB".CV, in2 := 33)
      S_Move(in := "SET VALUE"."HPHV ATS", out => "REVAMP".L30)
      P_Trig( "IO BITS"."HPHV PULSE"[6] )
      S_Coil( "TRIGGER" )
   END_RUNG
   RUNG wire#w2
      { S7_Templates := "SrcType := Int" } EQ_Contact(in1 := "IEC_Counter_0_DB".CV, in2 := 34)
      S_Move(in := "SET VALUE"."HPHV ATS HOLD", out => "REVAMP".L30)
      P_Trig( "IO BITS"."HPHV PULSE"[7] )
      S_Coil( "TRIGGER" )
   END_RUNG
   RUNG wire#w2
      { S7_Templates := "SrcType := Int" } EQ_Contact(in1 := "IEC_Counter_0_DB".CV, in2 := 35)
      S_Move(in := "SET VALUE"."HPHV END PRESS", out => "REVAMP".L30)
      P_Trig( "IO BITS"."HPHV PULSE"[8] )
      S_Coil( "TRIGGER" )
   END_RUNG
   RUNG wire#w2
      { S7_Templates := "SrcType := Int" } EQ_Contact(in1 := "IEC_Counter_0_DB".CV, in2 := 36)
      S_Move(in := "SET VALUE"."SET HPHV POST PULSES", out => "REVAMP".L30)
      P_Trig( "IO BITS"."HPHV PULSE"[9] )
      S_Coil( "TRIGGER" )
   END_RUNG
   RUNG wire#w2
      { S7_Templates := "SrcType := Int" } EQ_Contact(in1 := "IEC_Counter_0_DB".CV, in2 := 37)
      S_Move(in := "SET VALUE"."JACKET ALM TIME", out => "REVAMP".L30)
      P_Trig( "IO BITS"."HPHV PULSE"[10] )
      S_Coil( "TRIGGER" )
   END_RUNG
   RUNG wire#w2
      { S7_Templates := "SrcType := Int" } EQ_Contact(in1 := "IEC_Counter_0_DB".CV, in2 := 38)
      S_Move(in := "SET VALUE"."HEAT ALM TIME", out => "REVAMP".L30)
      P_Trig( "IO BITS"."HPHV PULSE"[11] )
      S_Coil( "TRIGGER" )
   END_RUNG
   RUNG wire#w2
      { S7_Templates := "SrcType := Int" } EQ_Contact(in1 := "IEC_Counter_0_DB".CV, in2 := 39)
      S_Move(in := "SET VALUE"."PRINT INTERVAL", out => "REVAMP".L30)
      P_Trig( "IO BITS"."HPHV PULSE"[12] )
      S_Coil( "TRIGGER" )
   END_RUNG
   RUNG wire#powerrail
      { S7_Templates := "SrcType := Int" } InRange(min := 70, in := "BUFF".PROCESS, max := 89)
      wire#w3
      { S7_Templates := "SrcType := Int" } EQ_Contact(in1 := "IEC_Counter_0_DB".CV, in2 := 40)
      Move(in := 40, out1 => "IEC_Counter_0_DB".CV)
   END_RUNG
   RUNG wire#powerrail
      { S7_Templates := "SrcType := Int" } InRange(min := 250, in := "BUFF".PROCESS, max := 255)
   END_RUNG wire#w3
   // the same network as SCL:
   #_w1 := "AlwaysTRUE" AND (((70 <= "BUFF".PROCESS) AND ("BUFF".PROCESS <= 89)) OR ((250 <= "BUFF".PROCESS) AND ("BUFF".PROCESS <= 255)));
   #_w2 := #_w1 AND ("IEC_Counter_0_DB".CV = 16);
   IF #_w2 THEN "REVAMP".L30 := "SET VALUE"."HPHV VCC"; END_IF;
   #_w3 := #_w2 AND NOT "AUXILIARY".PULSE1[13];   // rising edge
   "AUXILIARY".PULSE1[13] := #_w2;
   IF #_w3 THEN "TRIGGER" := TRUE; END_IF;
   #_w4 := #_w1 AND ("IEC_Counter_0_DB".CV = 17);
   IF #_w4 THEN "REVAMP".L30 := "SET VALUE"."HPHV VCC HOLD"; END_IF;
   #_w5 := #_w4 AND NOT "AUXILIARY".PULSE1[14];   // rising edge
   "AUXILIARY".PULSE1[14] := #_w4;
   IF #_w5 THEN "TRIGGER" := TRUE; END_IF;
   #_w6 := #_w1 AND ("IEC_Counter_0_DB".CV = 18);
   IF #_w6 THEN "REVAMP".L30 := "SET VALUE"."HPHV HEATUP PRESS"; END_IF;
   #_w7 := #_w6 AND NOT "AUXILIARY".PULSE1[21];   // rising edge
   "AUXILIARY".PULSE1[21] := #_w6;
   IF #_w7 THEN "TRIGGER" := TRUE; END_IF;
   #_w8 := #_w1 AND ("IEC_Counter_0_DB".CV = 19);
   IF #_w8 THEN "REVAMP".L30 := "SET VALUE"."HPHV NO"; END_IF;
   #_w9 := #_w8 AND NOT "AUXILIARY".PULSE1[18];   // rising edge
   "AUXILIARY".PULSE1[18] := #_w8;
   IF #_w9 THEN "TRIGGER" := TRUE; END_IF;
   #_w10 := #_w1 AND ("IEC_Counter_0_DB".CV = 20);
   IF #_w10 THEN "REVAMP".L30 := "SET VALUE"."HPHV HEATUP"; END_IF;
   #_w11 := #_w10 AND NOT "AUXILIARY".PULSE1[15];   // rising edge
   "AUXILIARY".PULSE1[15] := #_w10;
   IF #_w11 THEN "TRIGGER" := TRUE; END_IF;
   #_w12 := #_w1 AND ("IEC_Counter_0_DB".CV = 21);
   IF #_w12 THEN "REVAMP".L30 := "SET VALUE"."HPHV HEATUP HOLD"; END_IF;
   #_w13 := #_w12 AND NOT "AUXILIARY".PULSE1[16];   // rising edge
   "AUXILIARY".PULSE1[16] := #_w12;
   IF #_w13 THEN "TRIGGER" := TRUE; END_IF;
   #_w14 := #_w1 AND ("IEC_Counter_0_DB".CV = 22);
   IF #_w14 THEN "REVAMP".L30 := "SET VALUE"."SET HPHV HT1"; END_IF;
   #_w15 := #_w14 AND NOT "AUXILIARY".PULSE1[17];   // rising edge
   "AUXILIARY".PULSE1[17] := #_w14;
   IF #_w15 THEN "TRIGGER" := TRUE; END_IF;
   #_w16 := #_w1 AND ("IEC_Counter_0_DB".CV = 23);
   IF #_w16 THEN "REVAMP".L30 := "SET VALUE"."SET HPHV UP T1"; END_IF;
   #_w17 := #_w16 AND NOT "AUXILIARY".PULSE1[19];   // rising edge
   "AUXILIARY".PULSE1[19] := #_w16;
   IF #_w17 THEN "TRIGGER" := TRUE; END_IF;
   #_w18 := #_w1 AND ("IEC_Counter_0_DB".CV = 24);
   IF #_w18 THEN "REVAMP".L30 := "SET VALUE"."SET HPHV HT2"; END_IF;
   #_w19 := #_w18 AND NOT "AUXILIARY".PULSE1[20];   // rising edge
   "AUXILIARY".PULSE1[20] := #_w18;
   IF #_w19 THEN "TRIGGER" := TRUE; END_IF;
   #_w20 := #_w1 AND ("IEC_Counter_0_DB".CV = 25);
   IF #_w20 THEN "REVAMP".L30 := "SET VALUE"."SET HPHV UP T2"; END_IF;
   #_w21 := #_w20 AND NOT "AUXILIARY".PULSE1[22];   // rising edge
   "AUXILIARY".PULSE1[22] := #_w20;
   IF #_w21 THEN "TRIGGER" := TRUE; END_IF;
   #_w22 := #_w1 AND ("IEC_Counter_0_DB".CV = 26);
   IF #_w22 THEN "REVAMP".L30 := "SET VALUE"."SET HPHV HT3"; END_IF;
   #_w23 := #_w22 AND NOT "IO BITS"."HPHV PULSE"[0];   // rising edge
   "IO BITS"."HPHV PULSE"[0] := #_w22;
   IF #_w23 THEN "TRIGGER" := TRUE; END_IF;
   #_w24 := #_w1 AND ("IEC_Counter_0_DB".CV = 27);
   IF #_w24 THEN "REVAMP".L30 := "SET VALUE"."SET HPHV UP T3"; END_IF;
   #_w25 := #_w24 AND NOT "IO BITS"."HPHV PULSE"[1];   // rising edge
   "IO BITS"."HPHV PULSE"[1] := #_w24;
   IF #_w25 THEN "TRIGGER" := TRUE; END_IF;
   #_w26 := #_w1 AND ("IEC_Counter_0_DB".CV = 28);
   IF #_w26 THEN "REVAMP".L30 := "SET VALUE"."SET HPHV STOP TMP"; END_IF;
   #_w27 := #_w26 AND NOT "IO BITS"."HPHV PULSE"[2];   // rising edge
   "IO BITS"."HPHV PULSE"[2] := #_w26;
   IF #_w27 THEN "TRIGGER" := TRUE; END_IF;
   #_w28 := #_w1 AND ("IEC_Counter_0_DB".CV = 29);
   IF #_w28 THEN "REVAMP".L30 := "SET VALUE"."ABORT TEMP"; END_IF;
   #_w29 := #_w28 AND NOT "IO BITS"."HPHV PULSE"[3];   // rising edge
   "IO BITS"."HPHV PULSE"[3] := #_w28;
   IF #_w29 THEN "TRIGGER" := TRUE; END_IF;
   #_w30 := #_w1 AND ("IEC_Counter_0_DB".CV = 30);
   IF #_w30 THEN "REVAMP".L30 := "SET VALUE"."OVERSHOOT TEMP"; END_IF;
   #_w31 := #_w30 AND NOT "IO BITS"."HPHV PULSE"[4];   // rising edge
   "IO BITS"."HPHV PULSE"[4] := #_w30;
   IF #_w31 THEN "TRIGGER" := TRUE; END_IF;
   #_w32 := #_w1 AND ("IEC_Counter_0_DB".CV = 31);
   IF #_w32 THEN "REVAMP".L30 := "SET VALUE"."CONTROL BAND"; END_IF;
   #_w33 := #_w32 AND NOT "IO BITS"."HPHV PULSE"[13];   // rising edge
   "IO BITS"."HPHV PULSE"[13] := #_w32;
   IF #_w33 THEN "TRIGGER" := TRUE; END_IF;
   #_w34 := #_w1 AND ("IEC_Counter_0_DB".CV = 32);
   IF #_w34 THEN "REVAMP".L30 := "SET VALUE"."HPHV EXH PRESS"; END_IF;
   #_w35 := #_w34 AND NOT "IO BITS"."HPHV PULSE"[5];   // rising edge
   "IO BITS"."HPHV PULSE"[5] := #_w34;
   IF #_w35 THEN "TRIGGER" := TRUE; END_IF;
   #_w36 := #_w1 AND ("IEC_Counter_0_DB".CV = 33);
   IF #_w36 THEN "REVAMP".L30 := "SET VALUE"."HPHV ATS"; END_IF;
   #_w37 := #_w36 AND NOT "IO BITS"."HPHV PULSE"[6];   // rising edge
   "IO BITS"."HPHV PULSE"[6] := #_w36;
   IF #_w37 THEN "TRIGGER" := TRUE; END_IF;
   #_w38 := #_w1 AND ("IEC_Counter_0_DB".CV = 34);
   IF #_w38 THEN "REVAMP".L30 := "SET VALUE"."HPHV ATS HOLD"; END_IF;
   #_w39 := #_w38 AND NOT "IO BITS"."HPHV PULSE"[7];   // rising edge
   "IO BITS"."HPHV PULSE"[7] := #_w38;
   IF #_w39 THEN "TRIGGER" := TRUE; END_IF;
   #_w40 := #_w1 AND ("IEC_Counter_0_DB".CV = 35);
   IF #_w40 THEN "REVAMP".L30 := "SET VALUE"."HPHV END PRESS"; END_IF;
   #_w41 := #_w40 AND NOT "IO BITS"."HPHV PULSE"[8];   // rising edge
   "IO BITS"."HPHV PULSE"[8] := #_w40;
   IF #_w41 THEN "TRIGGER" := TRUE; END_IF;
   #_w42 := #_w1 AND ("IEC_Counter_0_DB".CV = 36);
   IF #_w42 THEN "REVAMP".L30 := "SET VALUE"."SET HPHV POST PULSES"; END_IF;
   #_w43 := #_w42 AND NOT "IO BITS"."HPHV PULSE"[9];   // rising edge
   "IO BITS"."HPHV PULSE"[9] := #_w42;
   IF #_w43 THEN "TRIGGER" := TRUE; END_IF;
   #_w44 := #_w1 AND ("IEC_Counter_0_DB".CV = 37);
   IF #_w44 THEN "REVAMP".L30 := "SET VALUE"."JACKET ALM TIME"; END_IF;
   #_w45 := #_w44 AND NOT "IO BITS"."HPHV PULSE"[10];   // rising edge
   "IO BITS"."HPHV PULSE"[10] := #_w44;
   IF #_w45 THEN "TRIGGER" := TRUE; END_IF;
   #_w46 := #_w1 AND ("IEC_Counter_0_DB".CV = 38);
   IF #_w46 THEN "REVAMP".L30 := "SET VALUE"."HEAT ALM TIME"; END_IF;
   #_w47 := #_w46 AND NOT "IO BITS"."HPHV PULSE"[11];   // rising edge
   "IO BITS"."HPHV PULSE"[11] := #_w46;
   IF #_w47 THEN "TRIGGER" := TRUE; END_IF;
   #_w48 := #_w1 AND ("IEC_Counter_0_DB".CV = 39);
   IF #_w48 THEN "REVAMP".L30 := "SET VALUE"."PRINT INTERVAL"; END_IF;
   #_w49 := #_w48 AND NOT "IO BITS"."HPHV PULSE"[12];   // rising edge
   "IO BITS"."HPHV PULSE"[12] := #_w48;
   IF #_w49 THEN "TRIGGER" := TRUE; END_IF;
   IF (((70 <= "BUFF".PROCESS) AND ("BUFF".PROCESS <= 89)) OR ((250 <= "BUFF".PROCESS) AND ("BUFF".PROCESS <= 255))) AND ("IEC_Counter_0_DB".CV = 40) THEN
       "IEC_Counter_0_DB".CV := 40;
   END_IF;
END_REGION

REGION Network 11
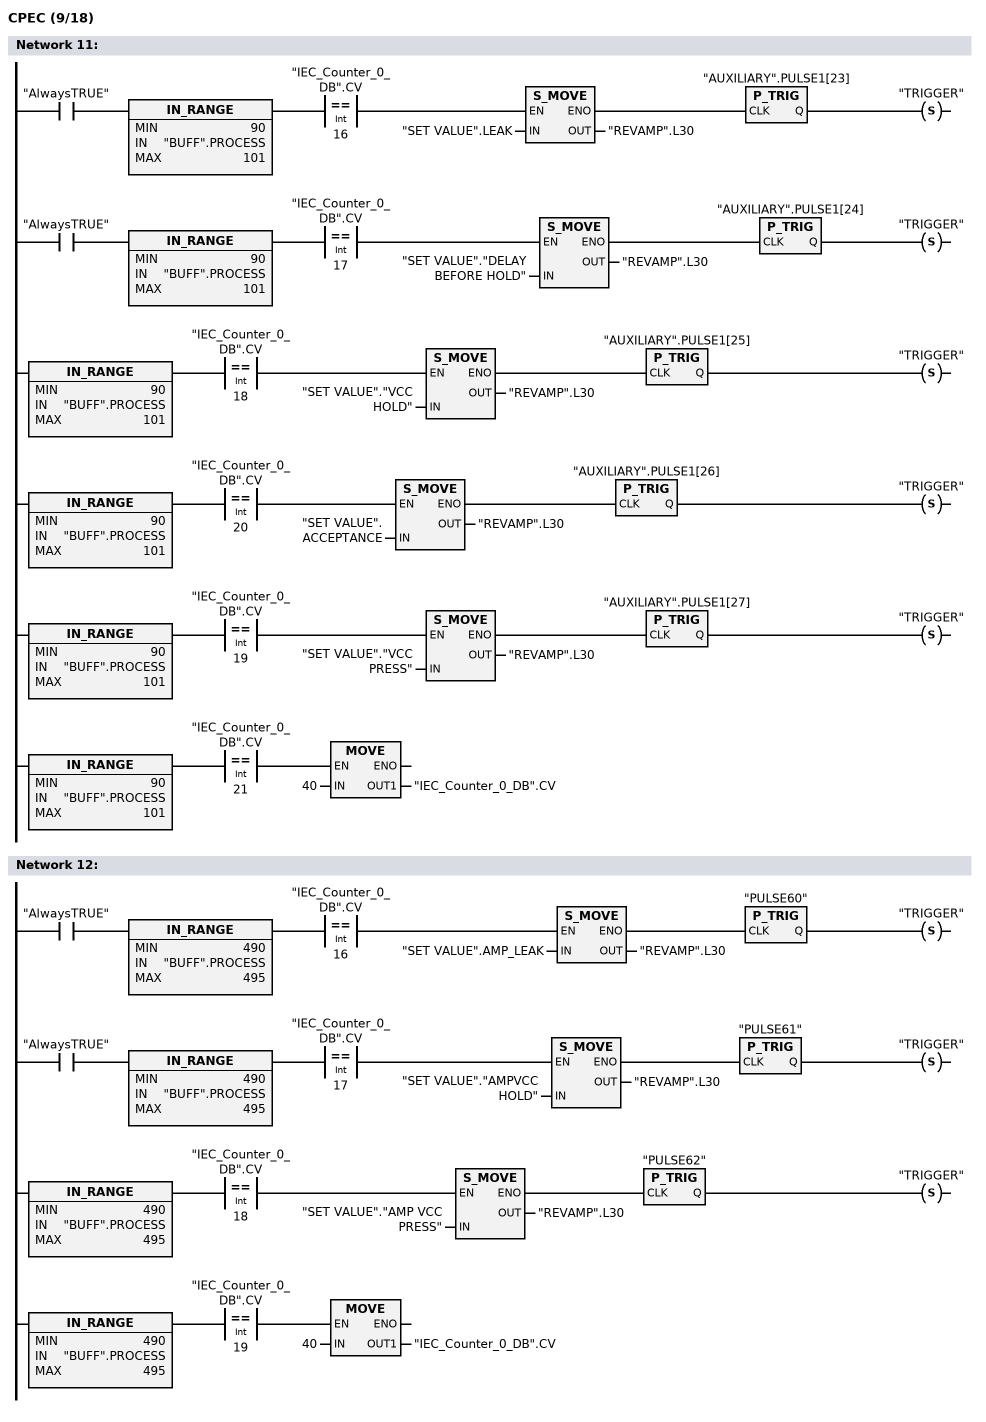
   RUNG wire#powerrail
      Contact( "AlwaysTRUE" )
      { S7_Templates := "SrcType := Int" } InRange(min := 90, in := "BUFF".PROCESS, max := 101)
      { S7_Templates := "SrcType := Int" } EQ_Contact(in1 := "IEC_Counter_0_DB".CV, in2 := 16)
      S_Move(in := "SET VALUE".LEAK, out => "REVAMP".L30)
      P_Trig( "AUXILIARY".PULSE1[23] )
      S_Coil( "TRIGGER" )
   END_RUNG
   RUNG wire#powerrail
      Contact( "AlwaysTRUE" )
      { S7_Templates := "SrcType := Int" } InRange(min := 90, in := "BUFF".PROCESS, max := 101)
      { S7_Templates := "SrcType := Int" } EQ_Contact(in1 := "IEC_Counter_0_DB".CV, in2 := 17)
      S_Move(in := "SET VALUE"."DELAY BEFORE HOLD", out => "REVAMP".L30)
      P_Trig( "AUXILIARY".PULSE1[24] )
      S_Coil( "TRIGGER" )
   END_RUNG
   RUNG wire#powerrail
      { S7_Templates := "SrcType := Int" } InRange(min := 90, in := "BUFF".PROCESS, max := 101)
      { S7_Templates := "SrcType := Int" } EQ_Contact(in1 := "IEC_Counter_0_DB".CV, in2 := 18)
      S_Move(in := "SET VALUE"."VCC HOLD", out => "REVAMP".L30)
      P_Trig( "AUXILIARY".PULSE1[25] )
      S_Coil( "TRIGGER" )
   END_RUNG
   RUNG wire#powerrail
      { S7_Templates := "SrcType := Int" } InRange(min := 90, in := "BUFF".PROCESS, max := 101)
      { S7_Templates := "SrcType := Int" } EQ_Contact(in1 := "IEC_Counter_0_DB".CV, in2 := 20)
      S_Move(in := "SET VALUE".ACCEPTANCE, out => "REVAMP".L30)
      P_Trig( "AUXILIARY".PULSE1[26] )
      S_Coil( "TRIGGER" )
   END_RUNG
   RUNG wire#powerrail
      { S7_Templates := "SrcType := Int" } InRange(min := 90, in := "BUFF".PROCESS, max := 101)
      { S7_Templates := "SrcType := Int" } EQ_Contact(in1 := "IEC_Counter_0_DB".CV, in2 := 19)
      S_Move(in := "SET VALUE"."VCC PRESS", out => "REVAMP".L30)
      P_Trig( "AUXILIARY".PULSE1[27] )
      S_Coil( "TRIGGER" )
   END_RUNG
   RUNG wire#powerrail
      { S7_Templates := "SrcType := Int" } InRange(min := 90, in := "BUFF".PROCESS, max := 101)
      { S7_Templates := "SrcType := Int" } EQ_Contact(in1 := "IEC_Counter_0_DB".CV, in2 := 21)
      Move(in := 40, out1 => "IEC_Counter_0_DB".CV)
   END_RUNG
   // the same network as SCL:
   #_w1 := "AlwaysTRUE" AND (90 <= "BUFF".PROCESS) AND ("BUFF".PROCESS <= 101) AND ("IEC_Counter_0_DB".CV = 16);
   IF #_w1 THEN "REVAMP".L30 := "SET VALUE".LEAK; END_IF;
   #_w2 := #_w1 AND NOT "AUXILIARY".PULSE1[23];   // rising edge
   "AUXILIARY".PULSE1[23] := #_w1;
   IF #_w2 THEN "TRIGGER" := TRUE; END_IF;
   #_w3 := "AlwaysTRUE" AND (90 <= "BUFF".PROCESS) AND ("BUFF".PROCESS <= 101) AND ("IEC_Counter_0_DB".CV = 17);
   IF #_w3 THEN "REVAMP".L30 := "SET VALUE"."DELAY BEFORE HOLD"; END_IF;
   #_w4 := #_w3 AND NOT "AUXILIARY".PULSE1[24];   // rising edge
   "AUXILIARY".PULSE1[24] := #_w3;
   IF #_w4 THEN "TRIGGER" := TRUE; END_IF;
   #_w5 := (90 <= "BUFF".PROCESS) AND ("BUFF".PROCESS <= 101) AND ("IEC_Counter_0_DB".CV = 18);
   IF #_w5 THEN "REVAMP".L30 := "SET VALUE"."VCC HOLD"; END_IF;
   #_w6 := #_w5 AND NOT "AUXILIARY".PULSE1[25];   // rising edge
   "AUXILIARY".PULSE1[25] := #_w5;
   IF #_w6 THEN "TRIGGER" := TRUE; END_IF;
   #_w7 := (90 <= "BUFF".PROCESS) AND ("BUFF".PROCESS <= 101) AND ("IEC_Counter_0_DB".CV = 20);
   IF #_w7 THEN "REVAMP".L30 := "SET VALUE".ACCEPTANCE; END_IF;
   #_w8 := #_w7 AND NOT "AUXILIARY".PULSE1[26];   // rising edge
   "AUXILIARY".PULSE1[26] := #_w7;
   IF #_w8 THEN "TRIGGER" := TRUE; END_IF;
   #_w9 := (90 <= "BUFF".PROCESS) AND ("BUFF".PROCESS <= 101) AND ("IEC_Counter_0_DB".CV = 19);
   IF #_w9 THEN "REVAMP".L30 := "SET VALUE"."VCC PRESS"; END_IF;
   #_w10 := #_w9 AND NOT "AUXILIARY".PULSE1[27];   // rising edge
   "AUXILIARY".PULSE1[27] := #_w9;
   IF #_w10 THEN "TRIGGER" := TRUE; END_IF;
   IF (90 <= "BUFF".PROCESS) AND ("BUFF".PROCESS <= 101) AND ("IEC_Counter_0_DB".CV = 21) THEN
       "IEC_Counter_0_DB".CV := 40;
   END_IF;
END_REGION

REGION Network 12
   RUNG wire#powerrail
      Contact( "AlwaysTRUE" )
      { S7_Templates := "SrcType := Int" } InRange(min := 490, in := "BUFF".PROCESS, max := 495)
      { S7_Templates := "SrcType := Int" } EQ_Contact(in1 := "IEC_Counter_0_DB".CV, in2 := 16)
      S_Move(in := "SET VALUE".AMP_LEAK, out => "REVAMP".L30)
      P_Trig( "PULSE60" )
      S_Coil( "TRIGGER" )
   END_RUNG
   RUNG wire#powerrail
      Contact( "AlwaysTRUE" )
      { S7_Templates := "SrcType := Int" } InRange(min := 490, in := "BUFF".PROCESS, max := 495)
      { S7_Templates := "SrcType := Int" } EQ_Contact(in1 := "IEC_Counter_0_DB".CV, in2 := 17)
      S_Move(in := "SET VALUE"."AMPVCC HOLD", out => "REVAMP".L30)
      P_Trig( "PULSE61" )
      S_Coil( "TRIGGER" )
   END_RUNG
   RUNG wire#powerrail
      { S7_Templates := "SrcType := Int" } InRange(min := 490, in := "BUFF".PROCESS, max := 495)
      { S7_Templates := "SrcType := Int" } EQ_Contact(in1 := "IEC_Counter_0_DB".CV, in2 := 18)
      S_Move(in := "SET VALUE"."AMP VCC PRESS", out => "REVAMP".L30)
      P_Trig( "PULSE62" )
      S_Coil( "TRIGGER" )
   END_RUNG
   RUNG wire#powerrail
      { S7_Templates := "SrcType := Int" } InRange(min := 490, in := "BUFF".PROCESS, max := 495)
      { S7_Templates := "SrcType := Int" } EQ_Contact(in1 := "IEC_Counter_0_DB".CV, in2 := 19)
      Move(in := 40, out1 => "IEC_Counter_0_DB".CV)
   END_RUNG
   // the same network as SCL:
   #_w1 := "AlwaysTRUE" AND (490 <= "BUFF".PROCESS) AND ("BUFF".PROCESS <= 495) AND ("IEC_Counter_0_DB".CV = 16);
   IF #_w1 THEN "REVAMP".L30 := "SET VALUE".AMP_LEAK; END_IF;
   #_w2 := #_w1 AND NOT "PULSE60";   // rising edge
   "PULSE60" := #_w1;
   IF #_w2 THEN "TRIGGER" := TRUE; END_IF;
   #_w3 := "AlwaysTRUE" AND (490 <= "BUFF".PROCESS) AND ("BUFF".PROCESS <= 495) AND ("IEC_Counter_0_DB".CV = 17);
   IF #_w3 THEN "REVAMP".L30 := "SET VALUE"."AMPVCC HOLD"; END_IF;
   #_w4 := #_w3 AND NOT "PULSE61";   // rising edge
   "PULSE61" := #_w3;
   IF #_w4 THEN "TRIGGER" := TRUE; END_IF;
   #_w5 := (490 <= "BUFF".PROCESS) AND ("BUFF".PROCESS <= 495) AND ("IEC_Counter_0_DB".CV = 18);
   IF #_w5 THEN "REVAMP".L30 := "SET VALUE"."AMP VCC PRESS"; END_IF;
   #_w6 := #_w5 AND NOT "PULSE62";   // rising edge
   "PULSE62" := #_w5;
   IF #_w6 THEN "TRIGGER" := TRUE; END_IF;
   IF (490 <= "BUFF".PROCESS) AND ("BUFF".PROCESS <= 495) AND ("IEC_Counter_0_DB".CV = 19) THEN
       "IEC_Counter_0_DB".CV := 40;
   END_IF;
END_REGION

REGION Network 13
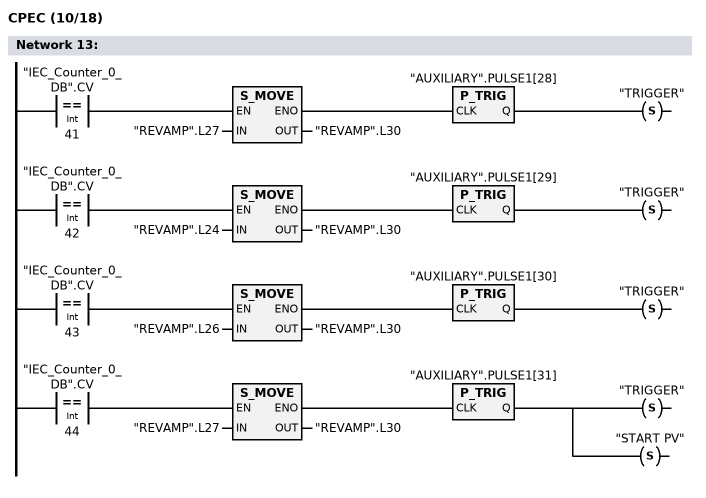
   RUNG wire#powerrail
      { S7_Templates := "SrcType := Int" } EQ_Contact(in1 := "IEC_Counter_0_DB".CV, in2 := 41)
      S_Move(in := "REVAMP".L27, out => "REVAMP".L30)
      P_Trig( "AUXILIARY".PULSE1[28] )
      S_Coil( "TRIGGER" )
   END_RUNG
   RUNG wire#powerrail
      { S7_Templates := "SrcType := Int" } EQ_Contact(in1 := "IEC_Counter_0_DB".CV, in2 := 42)
      S_Move(in := "REVAMP".L24, out => "REVAMP".L30)
      P_Trig( "AUXILIARY".PULSE1[29] )
      S_Coil( "TRIGGER" )
   END_RUNG
   RUNG wire#powerrail
      { S7_Templates := "SrcType := Int" } EQ_Contact(in1 := "IEC_Counter_0_DB".CV, in2 := 43)
      S_Move(in := "REVAMP".L26, out => "REVAMP".L30)
      P_Trig( "AUXILIARY".PULSE1[30] )
      S_Coil( "TRIGGER" )
   END_RUNG
   RUNG wire#powerrail
      { S7_Templates := "SrcType := Int" } EQ_Contact(in1 := "IEC_Counter_0_DB".CV, in2 := 44)
      S_Move(in := "REVAMP".L27, out => "REVAMP".L30)
      P_Trig( "AUXILIARY".PULSE1[31] )
      wire#w1
      S_Coil( "TRIGGER" )
   END_RUNG
   RUNG wire#w1
      S_Coil( "START PV" )
   END_RUNG
   // the same network as SCL:
   #_w1 := "IEC_Counter_0_DB".CV = 41;
   IF #_w1 THEN "REVAMP".L30 := "REVAMP".L27; END_IF;
   #_w2 := #_w1 AND NOT "AUXILIARY".PULSE1[28];   // rising edge
   "AUXILIARY".PULSE1[28] := #_w1;
   IF #_w2 THEN "TRIGGER" := TRUE; END_IF;
   #_w3 := "IEC_Counter_0_DB".CV = 42;
   IF #_w3 THEN "REVAMP".L30 := "REVAMP".L24; END_IF;
   #_w4 := #_w3 AND NOT "AUXILIARY".PULSE1[29];   // rising edge
   "AUXILIARY".PULSE1[29] := #_w3;
   IF #_w4 THEN "TRIGGER" := TRUE; END_IF;
   #_w5 := "IEC_Counter_0_DB".CV = 43;
   IF #_w5 THEN "REVAMP".L30 := "REVAMP".L26; END_IF;
   #_w6 := #_w5 AND NOT "AUXILIARY".PULSE1[30];   // rising edge
   "AUXILIARY".PULSE1[30] := #_w5;
   IF #_w6 THEN "TRIGGER" := TRUE; END_IF;
   #_w7 := "IEC_Counter_0_DB".CV = 44;
   IF #_w7 THEN "REVAMP".L30 := "REVAMP".L27; END_IF;
   #_w8 := #_w7 AND NOT "AUXILIARY".PULSE1[31];   // rising edge
   "AUXILIARY".PULSE1[31] := #_w7;
   IF #_w8 THEN
       "TRIGGER" := TRUE;
       "START PV" := TRUE;
   END_IF;
END_REGION

REGION Network 15
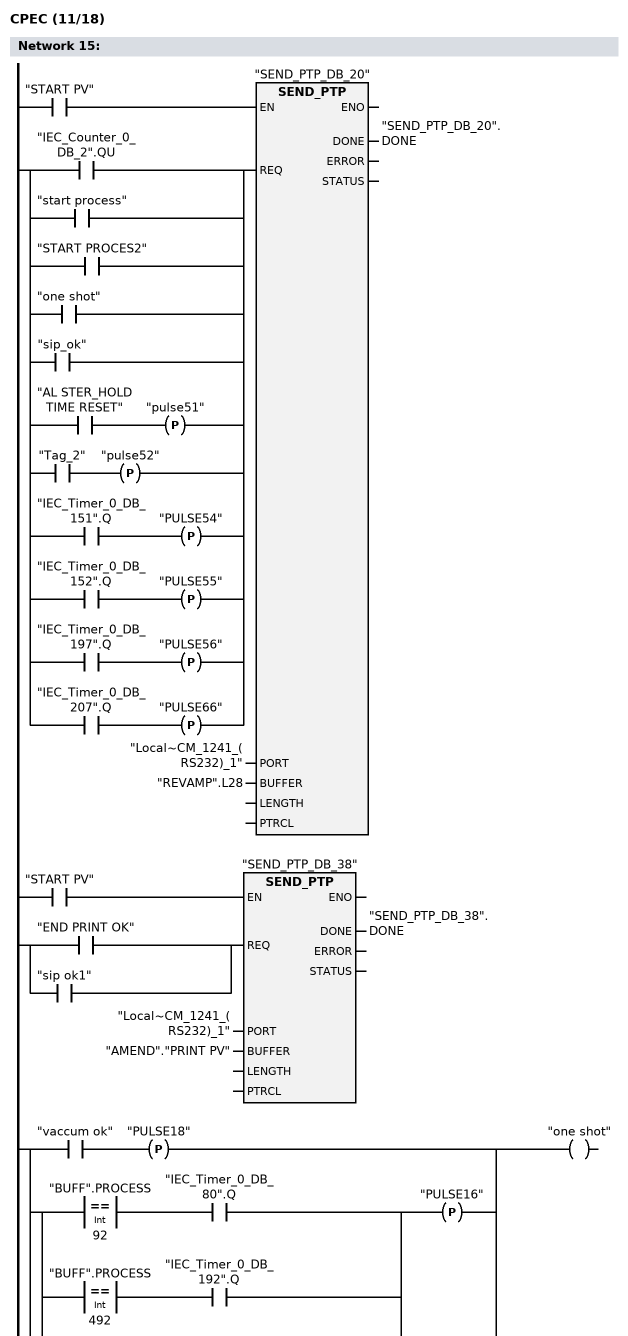
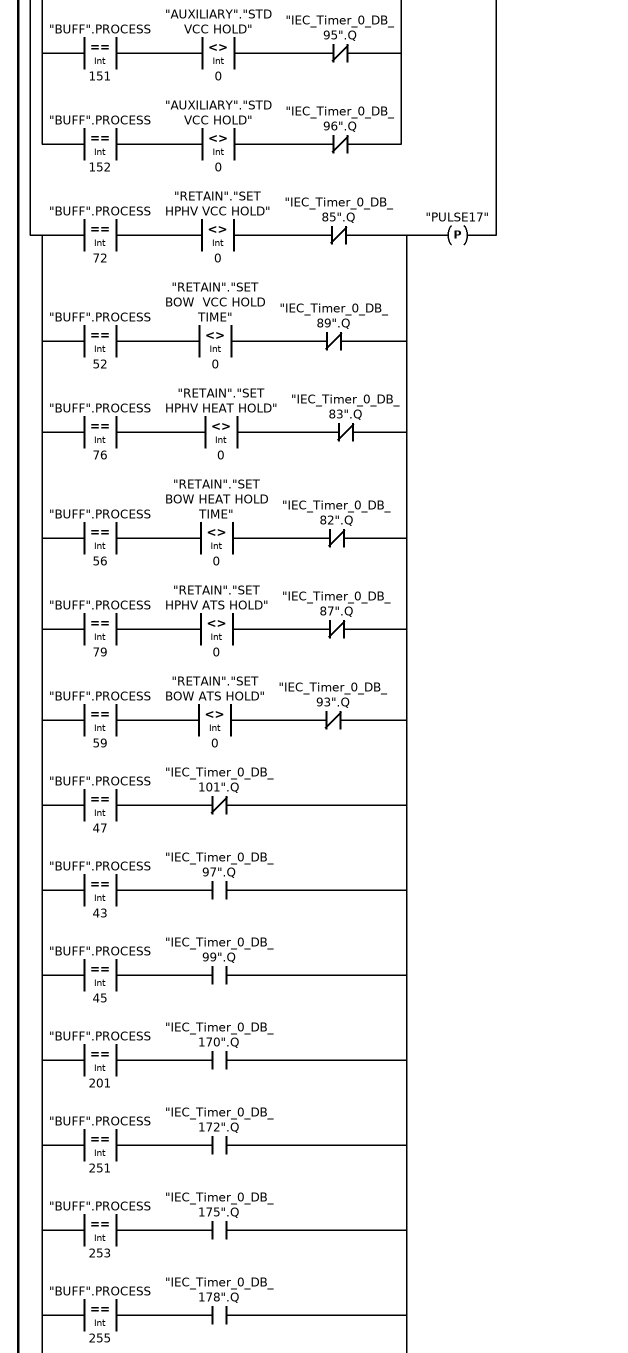
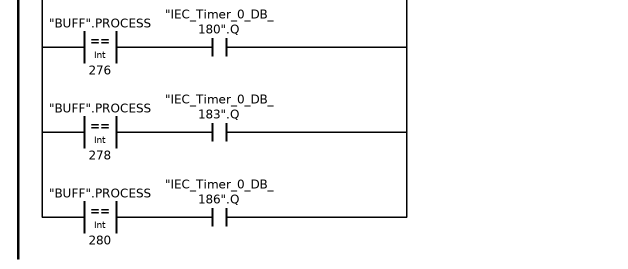
   RUNG wire#powerrail
      Contact( "START PV" )
      "SEND_PTP_DB_20".SEND_PTP(REQ := wire#w1, PORT := "Local~CM_1241_(RS232)_1", BUFFER := "REVAMP".L28, LENGTH :=, PTRCL :=, DONE => "SEND_PTP_DB_20".DONE, ERROR =>, STATUS =>)
   END_RUNG
   RUNG wire#powerrail
      Contact( "IEC_Counter_0_DB_2".QU )
   END_RUNG wire#w1
   RUNG wire#powerrail
      Contact( "start process" )
   END_RUNG wire#w1
   RUNG wire#powerrail
      Contact( "START PROCES2" )
   END_RUNG wire#w1
   RUNG wire#powerrail
      Contact( "one shot" )
   END_RUNG wire#w1
   RUNG wire#powerrail
      Contact( "sip_ok" )
   END_RUNG wire#w1
   RUNG wire#powerrail
      Contact( "AL STER_HOLD TIME RESET" )
      P_Trig( "pulse51" )
   END_RUNG wire#w1
   RUNG wire#powerrail
      Contact( "Tag_2" )
      P_Trig( "pulse52" )
   END_RUNG wire#w1
   RUNG wire#powerrail
      Contact( "IEC_Timer_0_DB_151".Q )
      P_Trig( "PULSE54" )
   END_RUNG wire#w1
   RUNG wire#powerrail
      Contact( "IEC_Timer_0_DB_152".Q )
      P_Trig( "PULSE55" )
   END_RUNG wire#w1
   RUNG wire#powerrail
      Contact( "IEC_Timer_0_DB_197".Q )
      P_Trig( "PULSE56" )
   END_RUNG wire#w1
   RUNG wire#powerrail
      Contact( "IEC_Timer_0_DB_207".Q )
      P_Trig( "PULSE66" )
   END_RUNG wire#w1
   RUNG wire#powerrail
      Contact( "START PV" )
      "SEND_PTP_DB_38".SEND_PTP(REQ := wire#w2, PORT := "Local~CM_1241_(RS232)_1", BUFFER := "AMEND"."PRINT PV", LENGTH :=, PTRCL :=, DONE => "SEND_PTP_DB_38".DONE, ERROR =>, STATUS =>)
   END_RUNG
   RUNG wire#powerrail
      Contact( "END PRINT OK" )
   END_RUNG wire#w2
   RUNG wire#powerrail
      Contact( "sip ok1" )
   END_RUNG wire#w2
   RUNG wire#powerrail
      Contact( "vaccum ok" )
      P_Trig( "PULSE18" )
      wire#w3
      Coil( "one shot" )
   END_RUNG
   RUNG wire#powerrail
      { S7_Templates := "SrcType := Int" } EQ_Contact(in1 := "BUFF".PROCESS, in2 := 92)
      Contact( "IEC_Timer_0_DB_80".Q )
      wire#w4
      P_Trig( "PULSE16" )
   END_RUNG wire#w3
   RUNG wire#powerrail
      { S7_Templates := "SrcType := Int" } EQ_Contact(in1 := "BUFF".PROCESS, in2 := 492)
      Contact( "IEC_Timer_0_DB_192".Q )
   END_RUNG wire#w4
   RUNG wire#powerrail
      { S7_Templates := "SrcType := Int" } EQ_Contact(in1 := "BUFF".PROCESS, in2 := 151)
      { S7_Templates := "SrcType := Int" } NE_Contact(in1 := "AUXILIARY"."STD VCC HOLD", in2 := 0)
      I_Contact( "IEC_Timer_0_DB_95".Q )
   END_RUNG wire#w4
   RUNG wire#powerrail
      { S7_Templates := "SrcType := Int" } EQ_Contact(in1 := "BUFF".PROCESS, in2 := 152)
      { S7_Templates := "SrcType := Int" } NE_Contact(in1 := "AUXILIARY"."STD VCC HOLD", in2 := 0)
      I_Contact( "IEC_Timer_0_DB_96".Q )
   END_RUNG wire#w4
   RUNG wire#powerrail
      { S7_Templates := "SrcType := Int" } EQ_Contact(in1 := "BUFF".PROCESS, in2 := 72)
      { S7_Templates := "SrcType := Int" } NE_Contact(in1 := "RETAIN"."SET HPHV VCC HOLD", in2 := 0)
      I_Contact( "IEC_Timer_0_DB_85".Q )
      wire#w5
      P_Trig( "PULSE17" )
   END_RUNG wire#w3
   RUNG wire#powerrail
      { S7_Templates := "SrcType := Int" } EQ_Contact(in1 := "BUFF".PROCESS, in2 := 52)
      { S7_Templates := "SrcType := Int" } NE_Contact(in1 := "RETAIN"."SET BOW  VCC HOLD TIME", in2 := 0)
      I_Contact( "IEC_Timer_0_DB_89".Q )
   END_RUNG wire#w5
   RUNG wire#powerrail
      { S7_Templates := "SrcType := Int" } EQ_Contact(in1 := "BUFF".PROCESS, in2 := 76)
      { S7_Templates := "SrcType := Int" } NE_Contact(in1 := "RETAIN"."SET HPHV HEAT HOLD", in2 := 0)
      I_Contact( "IEC_Timer_0_DB_83".Q )
   END_RUNG wire#w5
   RUNG wire#powerrail
      { S7_Templates := "SrcType := Int" } EQ_Contact(in1 := "BUFF".PROCESS, in2 := 56)
      { S7_Templates := "SrcType := Int" } NE_Contact(in1 := "RETAIN"."SET BOW HEAT HOLD TIME", in2 := 0)
      I_Contact( "IEC_Timer_0_DB_82".Q )
   END_RUNG wire#w5
   RUNG wire#powerrail
      { S7_Templates := "SrcType := Int" } EQ_Contact(in1 := "BUFF".PROCESS, in2 := 79)
      { S7_Templates := "SrcType := Int" } NE_Contact(in1 := "RETAIN"."SET HPHV ATS HOLD", in2 := 0)
      I_Contact( "IEC_Timer_0_DB_87".Q )
   END_RUNG wire#w5
   RUNG wire#powerrail
      { S7_Templates := "SrcType := Int" } EQ_Contact(in1 := "BUFF".PROCESS, in2 := 59)
      { S7_Templates := "SrcType := Int" } NE_Contact(in1 := "RETAIN"."SET BOW ATS HOLD", in2 := 0)
      I_Contact( "IEC_Timer_0_DB_93".Q )
   END_RUNG wire#w5
   RUNG wire#powerrail
      { S7_Templates := "SrcType := Int" } EQ_Contact(in1 := "BUFF".PROCESS, in2 := 47)
      I_Contact( "IEC_Timer_0_DB_101".Q )
   END_RUNG wire#w5
   RUNG wire#powerrail
      { S7_Templates := "SrcType := Int" } EQ_Contact(in1 := "BUFF".PROCESS, in2 := 43)
      Contact( "IEC_Timer_0_DB_97".Q )
   END_RUNG wire#w5
   RUNG wire#powerrail
      { S7_Templates := "SrcType := Int" } EQ_Contact(in1 := "BUFF".PROCESS, in2 := 45)
      Contact( "IEC_Timer_0_DB_99".Q )
   END_RUNG wire#w5
   RUNG wire#powerrail
      { S7_Templates := "SrcType := Int" } EQ_Contact(in1 := "BUFF".PROCESS, in2 := 201)
      Contact( "IEC_Timer_0_DB_170".Q )
   END_RUNG wire#w5
   RUNG wire#powerrail
      { S7_Templates := "SrcType := Int" } EQ_Contact(in1 := "BUFF".PROCESS, in2 := 251)
      Contact( "IEC_Timer_0_DB_172".Q )
   END_RUNG wire#w5
   RUNG wire#powerrail
      { S7_Templates := "SrcType := Int" } EQ_Contact(in1 := "BUFF".PROCESS, in2 := 253)
      Contact( "IEC_Timer_0_DB_175".Q )
   END_RUNG wire#w5
   RUNG wire#powerrail
      { S7_Templates := "SrcType := Int" } EQ_Contact(in1 := "BUFF".PROCESS, in2 := 255)
      Contact( "IEC_Timer_0_DB_178".Q )
   END_RUNG wire#w5
   RUNG wire#powerrail
      { S7_Templates := "SrcType := Int" } EQ_Contact(in1 := "BUFF".PROCESS, in2 := 276)
      Contact( "IEC_Timer_0_DB_180".Q )
   END_RUNG wire#w5
   RUNG wire#powerrail
      { S7_Templates := "SrcType := Int" } EQ_Contact(in1 := "BUFF".PROCESS, in2 := 278)
      Contact( "IEC_Timer_0_DB_183".Q )
   END_RUNG wire#w5
   RUNG wire#powerrail
      { S7_Templates := "SrcType := Int" } EQ_Contact(in1 := "BUFF".PROCESS, in2 := 280)
      Contact( "IEC_Timer_0_DB_186".Q )
   END_RUNG wire#w5
   // the same network as SCL:
   #_w1 := "AL STER_HOLD TIME RESET" AND NOT "pulse51";   // rising edge
   "pulse51" := "AL STER_HOLD TIME RESET";
   #_w2 := "Tag_2" AND NOT "pulse52";   // rising edge
   "pulse52" := "Tag_2";
   #_w3 := "IEC_Timer_0_DB_151".Q AND NOT "PULSE54";   // rising edge
   "PULSE54" := "IEC_Timer_0_DB_151".Q;
   #_w4 := "IEC_Timer_0_DB_152".Q AND NOT "PULSE55";   // rising edge
   "PULSE55" := "IEC_Timer_0_DB_152".Q;
   #_w5 := "IEC_Timer_0_DB_197".Q AND NOT "PULSE56";   // rising edge
   "PULSE56" := "IEC_Timer_0_DB_197".Q;
   #_w6 := "IEC_Timer_0_DB_207".Q AND NOT "PULSE66";   // rising edge
   "PULSE66" := "IEC_Timer_0_DB_207".Q;
   IF "START PV" THEN
       "SEND_PTP_DB_20"(REQ := "IEC_Counter_0_DB_2".QU OR "start process" OR "START PROCES2" OR "one shot" OR "sip_ok" OR #_w1 OR #_w2 OR #_w3 OR #_w4 OR #_w5 OR #_w6,   // SEND_PTP
                        PORT := "Local~CM_1241_(RS232)_1",
                        BUFFER := "REVAMP".L28,
                        DONE => "SEND_PTP_DB_20".DONE);
   END_IF;
   IF "START PV" THEN
       "SEND_PTP_DB_38"(REQ := "END PRINT OK" OR "sip ok1",   // SEND_PTP
                        PORT := "Local~CM_1241_(RS232)_1",
                        BUFFER := "AMEND"."PRINT PV",
                        DONE => "SEND_PTP_DB_38".DONE);
   END_IF;
   #_w7 := "vaccum ok" AND NOT "PULSE18";   // rising edge
   "PULSE18" := "vaccum ok";
   #_w8 := (("BUFF".PROCESS = 92) AND "IEC_Timer_0_DB_80".Q) OR (("BUFF".PROCESS = 492) AND "IEC_Timer_0_DB_192".Q) OR (("BUFF".PROCESS = 151) AND ("AUXILIARY"."STD VCC HOLD" <> 0) AND NOT "IEC_Timer_0_DB_95".Q) OR (("BUFF".PROCESS = 152) AND ("AUXILIARY"."STD VCC HOLD" <> 0) AND NOT "IEC_Timer_0_DB_96".Q);
   #_w9 := #_w8 AND NOT "PULSE16";   // rising edge
   "PULSE16" := #_w8;
   #_w10 := (("BUFF".PROCESS = 72) AND ("RETAIN"."SET HPHV VCC HOLD" <> 0) AND NOT "IEC_Timer_0_DB_85".Q) OR (("BUFF".PROCESS = 52) AND ("RETAIN"."SET BOW  VCC HOLD TIME" <> 0) AND NOT "IEC_Timer_0_DB_89".Q) OR (("BUFF".PROCESS = 76) AND ("RETAIN"."SET HPHV HEAT HOLD" <> 0) AND NOT "IEC_Timer_0_DB_83".Q) OR (("BUFF".PROCESS = 56) AND ("RETAIN"."SET BOW HEAT HOLD TIME" <> 0) AND NOT "IEC_Timer_0_DB_82".Q) OR (("BUFF".PROCESS = 79) AND ("RETAIN"."SET HPHV ATS HOLD" <> 0) AND NOT "IEC_Timer_0_DB_87".Q) OR (("BUFF".PROCESS = 59) AND ("RETAIN"."SET BOW ATS HOLD" <> 0) AND NOT "IEC_Timer_0_DB_93".Q) OR (("BUFF".PROCESS = 47) AND NOT "IEC_Timer_0_DB_101".Q) OR (("BUFF".PROCESS = 43) AND "IEC_Timer_0_DB_97".Q) OR (("BUFF".PROCESS = 45) AND "IEC_Timer_0_DB_99".Q) OR (("BUFF".PROCESS = 201) AND "IEC_Timer_0_DB_170".Q) OR (("BUFF".PROCESS = 251) AND "IEC_Timer_0_DB_172".Q) OR (("BUFF".PROCESS = 253) AND "IEC_Timer_0_DB_175".Q) OR (("BUFF".PROCESS = 255) AND "IEC_Timer_0_DB_178".Q) OR (("BUFF".PROCESS = 276) AND "IEC_Timer_0_DB_180".Q) OR (("BUFF".PROCESS = 278) AND "IEC_Timer_0_DB_183".Q) OR (("BUFF".PROCESS = 280) AND "IEC_Timer_0_DB_186".Q);
   #_w11 := #_w10 AND NOT "PULSE17";   // rising edge
   "PULSE17" := #_w10;
   "one shot" := #_w7 OR #_w9 OR #_w11;
END_REGION

REGION Network 16
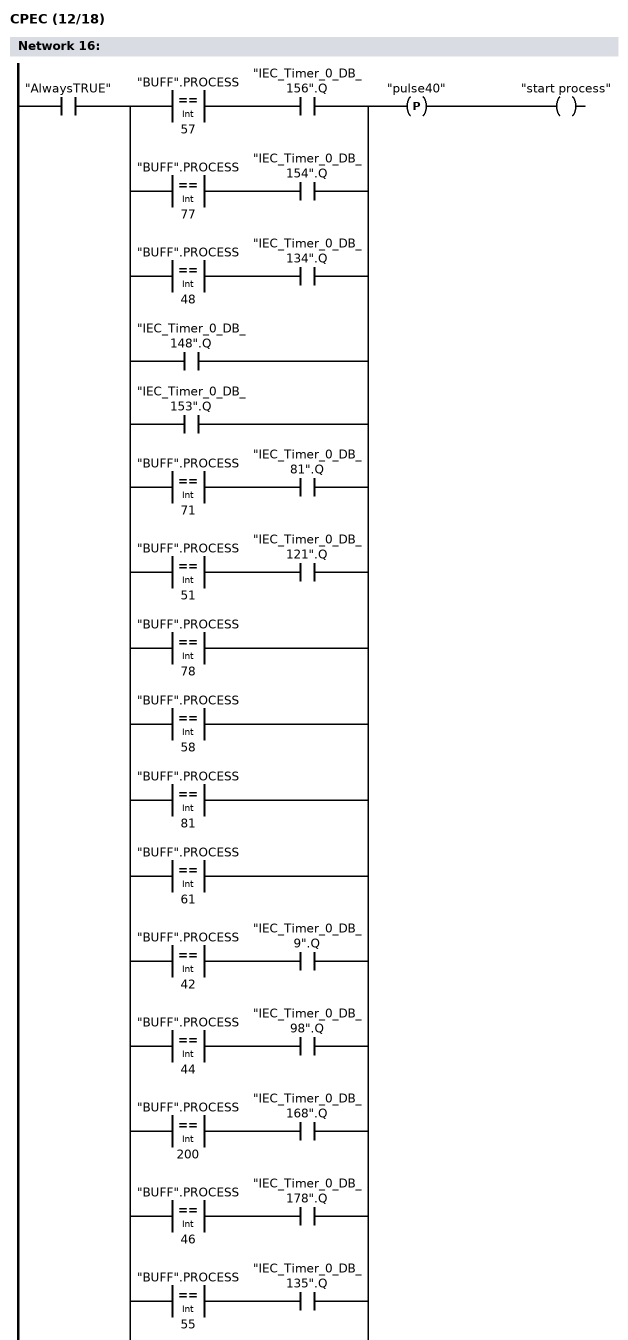
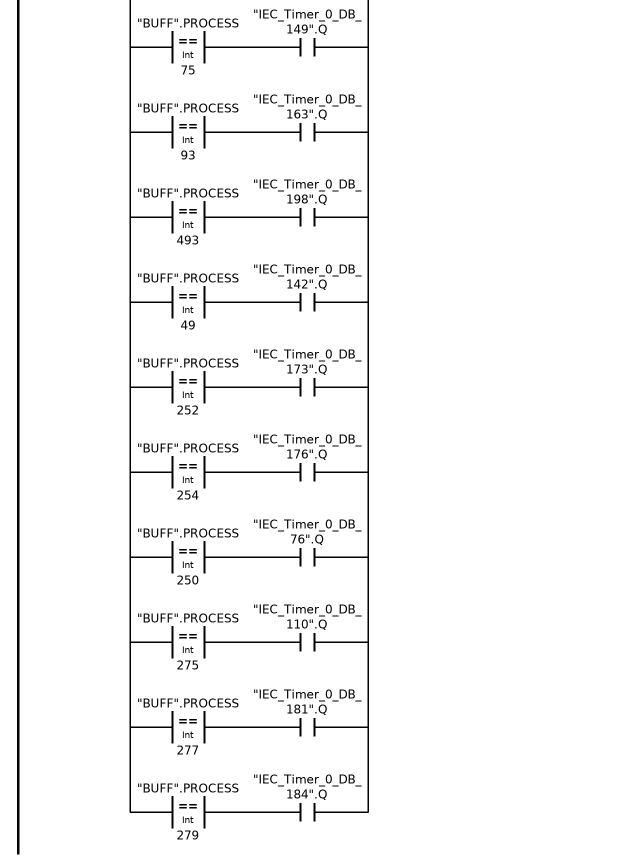
   RUNG wire#powerrail
      Contact( "AlwaysTRUE" )
      wire#w1
      { S7_Templates := "SrcType := Int" } EQ_Contact(in1 := "BUFF".PROCESS, in2 := 57)
      Contact( "IEC_Timer_0_DB_156".Q )
      wire#w2
      P_Trig( "pulse40" )
      Coil( "start process" )
   END_RUNG
   RUNG wire#w1
      { S7_Templates := "SrcType := Int" } EQ_Contact(in1 := "BUFF".PROCESS, in2 := 77)
      Contact( "IEC_Timer_0_DB_154".Q )
   END_RUNG wire#w2
   RUNG wire#w1
      { S7_Templates := "SrcType := Int" } EQ_Contact(in1 := "BUFF".PROCESS, in2 := 48)
      Contact( "IEC_Timer_0_DB_134".Q )
   END_RUNG wire#w2
   RUNG wire#w1
      Contact( "IEC_Timer_0_DB_148".Q )
   END_RUNG wire#w2
   RUNG wire#w1
      Contact( "IEC_Timer_0_DB_153".Q )
   END_RUNG wire#w2
   RUNG wire#w1
      { S7_Templates := "SrcType := Int" } EQ_Contact(in1 := "BUFF".PROCESS, in2 := 71)
      Contact( "IEC_Timer_0_DB_81".Q )
   END_RUNG wire#w2
   RUNG wire#w1
      { S7_Templates := "SrcType := Int" } EQ_Contact(in1 := "BUFF".PROCESS, in2 := 51)
      Contact( "IEC_Timer_0_DB_121".Q )
   END_RUNG wire#w2
   RUNG wire#w1
      { S7_Templates := "SrcType := Int" } EQ_Contact(in1 := "BUFF".PROCESS, in2 := 78)
   END_RUNG wire#w2
   RUNG wire#w1
      { S7_Templates := "SrcType := Int" } EQ_Contact(in1 := "BUFF".PROCESS, in2 := 58)
   END_RUNG wire#w2
   RUNG wire#w1
      { S7_Templates := "SrcType := Int" } EQ_Contact(in1 := "BUFF".PROCESS, in2 := 81)
   END_RUNG wire#w2
   RUNG wire#w1
      { S7_Templates := "SrcType := Int" } EQ_Contact(in1 := "BUFF".PROCESS, in2 := 61)
   END_RUNG wire#w2
   RUNG wire#w1
      { S7_Templates := "SrcType := Int" } EQ_Contact(in1 := "BUFF".PROCESS, in2 := 42)
      Contact( "IEC_Timer_0_DB_9".Q )
   END_RUNG wire#w2
   RUNG wire#w1
      { S7_Templates := "SrcType := Int" } EQ_Contact(in1 := "BUFF".PROCESS, in2 := 44)
      Contact( "IEC_Timer_0_DB_98".Q )
   END_RUNG wire#w2
   RUNG wire#w1
      { S7_Templates := "SrcType := Int" } EQ_Contact(in1 := "BUFF".PROCESS, in2 := 200)
      Contact( "IEC_Timer_0_DB_168".Q )
   END_RUNG wire#w2
   RUNG wire#w1
      { S7_Templates := "SrcType := Int" } EQ_Contact(in1 := "BUFF".PROCESS, in2 := 46)
      Contact( "IEC_Timer_0_DB_178".Q )
   END_RUNG wire#w2
   RUNG wire#w1
      { S7_Templates := "SrcType := Int" } EQ_Contact(in1 := "BUFF".PROCESS, in2 := 55)
      Contact( "IEC_Timer_0_DB_135".Q )
   END_RUNG wire#w2
   RUNG wire#w1
      { S7_Templates := "SrcType := Int" } EQ_Contact(in1 := "BUFF".PROCESS, in2 := 75)
      Contact( "IEC_Timer_0_DB_149".Q )
   END_RUNG wire#w2
   RUNG wire#w1
      { S7_Templates := "SrcType := Int" } EQ_Contact(in1 := "BUFF".PROCESS, in2 := 93)
      Contact( "IEC_Timer_0_DB_163".Q )
   END_RUNG wire#w2
   RUNG wire#w1
      { S7_Templates := "SrcType := Int" } EQ_Contact(in1 := "BUFF".PROCESS, in2 := 493)
      Contact( "IEC_Timer_0_DB_198".Q )
   END_RUNG wire#w2
   RUNG wire#w1
      { S7_Templates := "SrcType := Int" } EQ_Contact(in1 := "BUFF".PROCESS, in2 := 49)
      Contact( "IEC_Timer_0_DB_142".Q )
   END_RUNG wire#w2
   RUNG wire#w1
      { S7_Templates := "SrcType := Int" } EQ_Contact(in1 := "BUFF".PROCESS, in2 := 252)
      Contact( "IEC_Timer_0_DB_173".Q )
   END_RUNG wire#w2
   RUNG wire#w1
      { S7_Templates := "SrcType := Int" } EQ_Contact(in1 := "BUFF".PROCESS, in2 := 254)
      Contact( "IEC_Timer_0_DB_176".Q )
   END_RUNG wire#w2
   RUNG wire#w1
      { S7_Templates := "SrcType := Int" } EQ_Contact(in1 := "BUFF".PROCESS, in2 := 250)
      Contact( "IEC_Timer_0_DB_76".Q )
   END_RUNG wire#w2
   RUNG wire#w1
      { S7_Templates := "SrcType := Int" } EQ_Contact(in1 := "BUFF".PROCESS, in2 := 275)
      Contact( "IEC_Timer_0_DB_110".Q )
   END_RUNG wire#w2
   RUNG wire#w1
      { S7_Templates := "SrcType := Int" } EQ_Contact(in1 := "BUFF".PROCESS, in2 := 277)
      Contact( "IEC_Timer_0_DB_181".Q )
   END_RUNG wire#w2
   RUNG wire#w1
      { S7_Templates := "SrcType := Int" } EQ_Contact(in1 := "BUFF".PROCESS, in2 := 279)
      Contact( "IEC_Timer_0_DB_184".Q )
   END_RUNG wire#w2
   // the same network as SCL:
   #_w1 := "AlwaysTRUE" AND ((("BUFF".PROCESS = 57) AND "IEC_Timer_0_DB_156".Q) OR (("BUFF".PROCESS = 77) AND "IEC_Timer_0_DB_154".Q) OR (("BUFF".PROCESS = 48) AND "IEC_Timer_0_DB_134".Q) OR "IEC_Timer_0_DB_148".Q OR "IEC_Timer_0_DB_153".Q OR (("BUFF".PROCESS = 71) AND "IEC_Timer_0_DB_81".Q) OR (("BUFF".PROCESS = 51) AND "IEC_Timer_0_DB_121".Q) OR ("BUFF".PROCESS = 78) OR ("BUFF".PROCESS = 58) OR ("BUFF".PROCESS = 81) OR ("BUFF".PROCESS = 61) OR (("BUFF".PROCESS = 42) AND "IEC_Timer_0_DB_9".Q) OR (("BUFF".PROCESS = 44) AND "IEC_Timer_0_DB_98".Q) OR (("BUFF".PROCESS = 200) AND "IEC_Timer_0_DB_168".Q) OR (("BUFF".PROCESS = 46) AND "IEC_Timer_0_DB_178".Q) OR (("BUFF".PROCESS = 55) AND "IEC_Timer_0_DB_135".Q) OR (("BUFF".PROCESS = 75) AND "IEC_Timer_0_DB_149".Q) OR (("BUFF".PROCESS = 93) AND "IEC_Timer_0_DB_163".Q) OR (("BUFF".PROCESS = 493) AND "IEC_Timer_0_DB_198".Q) OR (("BUFF".PROCESS = 49) AND "IEC_Timer_0_DB_142".Q) OR (("BUFF".PROCESS = 252) AND "IEC_Timer_0_DB_173".Q) OR (("BUFF".PROCESS = 254) AND "IEC_Timer_0_DB_176".Q) OR (("BUFF".PROCESS = 250) AND "IEC_Timer_0_DB_76".Q) OR (("BUFF".PROCESS = 275) AND "IEC_Timer_0_DB_110".Q) OR (("BUFF".PROCESS = 277) AND "IEC_Timer_0_DB_181".Q) OR (("BUFF".PROCESS = 279) AND "IEC_Timer_0_DB_184".Q));
   #_w2 := #_w1 AND NOT "pulse40";   // rising edge
   "pulse40" := #_w1;
   "start process" := #_w2;
END_REGION

REGION Network 17
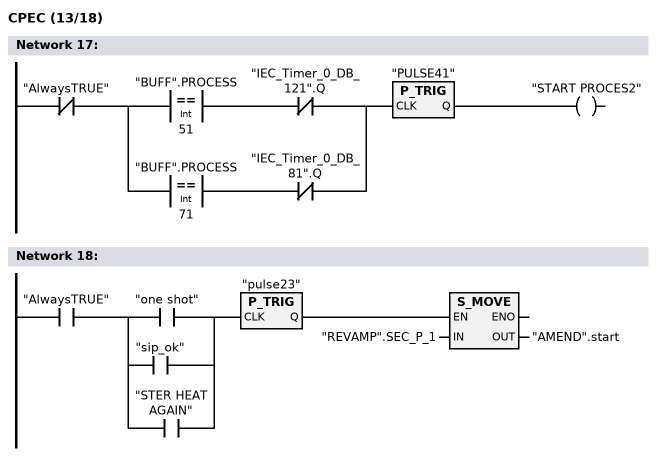
   RUNG wire#powerrail
      I_Contact( "AlwaysTRUE" )
      wire#w1
      { S7_Templates := "SrcType := Int" } EQ_Contact(in1 := "BUFF".PROCESS, in2 := 51)
      I_Contact( "IEC_Timer_0_DB_121".Q )
      wire#w2
      P_Trig( "PULSE41" )
      Coil( "START PROCES2" )
   END_RUNG
   RUNG wire#w1
      { S7_Templates := "SrcType := Int" } EQ_Contact(in1 := "BUFF".PROCESS, in2 := 71)
      I_Contact( "IEC_Timer_0_DB_81".Q )
   END_RUNG wire#w2
   // the same network as SCL:
   #_w1 := NOT "AlwaysTRUE" AND ((("BUFF".PROCESS = 51) AND NOT "IEC_Timer_0_DB_121".Q) OR (("BUFF".PROCESS = 71) AND NOT "IEC_Timer_0_DB_81".Q));
   #_w2 := #_w1 AND NOT "PULSE41";   // rising edge
   "PULSE41" := #_w1;
   "START PROCES2" := #_w2;
END_REGION

REGION Network 18
   RUNG wire#powerrail
      Contact( "AlwaysTRUE" )
      wire#w1
      Contact( "one shot" )
      wire#w2
      P_Trig( "pulse23" )
      S_Move(in := "REVAMP".SEC_P_1, out => "AMEND".start)
   END_RUNG
   RUNG wire#w1
      Contact( "sip_ok" )
   END_RUNG wire#w2
   RUNG wire#w1
      Contact( "STER HEAT AGAIN" )
   END_RUNG wire#w2
   // the same network as SCL:
   #_w1 := "AlwaysTRUE" AND ("one shot" OR "sip_ok" OR "STER HEAT AGAIN");
   #_w2 := #_w1 AND NOT "pulse23";   // rising edge
   "pulse23" := #_w1;
   IF #_w2 THEN "AMEND".start := "REVAMP".SEC_P_1; END_IF;
END_REGION

REGION Network 19
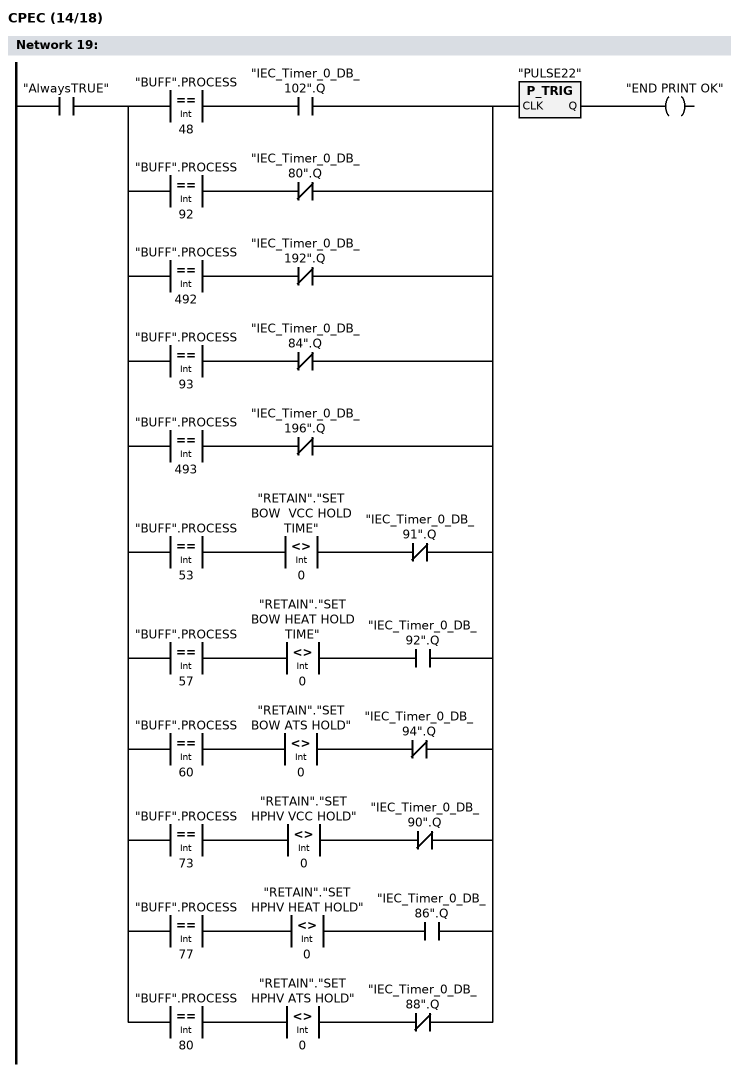
   RUNG wire#powerrail
      Contact( "AlwaysTRUE" )
      wire#w1
      { S7_Templates := "SrcType := Int" } EQ_Contact(in1 := "BUFF".PROCESS, in2 := 48)
      Contact( "IEC_Timer_0_DB_102".Q )
      wire#w2
      P_Trig( "PULSE22" )
      Coil( "END PRINT OK" )
   END_RUNG
   RUNG wire#w1
      { S7_Templates := "SrcType := Int" } EQ_Contact(in1 := "BUFF".PROCESS, in2 := 92)
      I_Contact( "IEC_Timer_0_DB_80".Q )
   END_RUNG wire#w2
   RUNG wire#w1
      { S7_Templates := "SrcType := Int" } EQ_Contact(in1 := "BUFF".PROCESS, in2 := 492)
      I_Contact( "IEC_Timer_0_DB_192".Q )
   END_RUNG wire#w2
   RUNG wire#w1
      { S7_Templates := "SrcType := Int" } EQ_Contact(in1 := "BUFF".PROCESS, in2 := 93)
      I_Contact( "IEC_Timer_0_DB_84".Q )
   END_RUNG wire#w2
   RUNG wire#w1
      { S7_Templates := "SrcType := Int" } EQ_Contact(in1 := "BUFF".PROCESS, in2 := 493)
      I_Contact( "IEC_Timer_0_DB_196".Q )
   END_RUNG wire#w2
   RUNG wire#w1
      { S7_Templates := "SrcType := Int" } EQ_Contact(in1 := "BUFF".PROCESS, in2 := 53)
      { S7_Templates := "SrcType := Int" } NE_Contact(in1 := "RETAIN"."SET BOW  VCC HOLD TIME", in2 := 0)
      I_Contact( "IEC_Timer_0_DB_91".Q )
   END_RUNG wire#w2
   RUNG wire#w1
      { S7_Templates := "SrcType := Int" } EQ_Contact(in1 := "BUFF".PROCESS, in2 := 57)
      { S7_Templates := "SrcType := Int" } NE_Contact(in1 := "RETAIN"."SET BOW HEAT HOLD TIME", in2 := 0)
      Contact( "IEC_Timer_0_DB_92".Q )
   END_RUNG wire#w2
   RUNG wire#w1
      { S7_Templates := "SrcType := Int" } EQ_Contact(in1 := "BUFF".PROCESS, in2 := 60)
      { S7_Templates := "SrcType := Int" } NE_Contact(in1 := "RETAIN"."SET BOW ATS HOLD", in2 := 0)
      I_Contact( "IEC_Timer_0_DB_94".Q )
   END_RUNG wire#w2
   RUNG wire#w1
      { S7_Templates := "SrcType := Int" } EQ_Contact(in1 := "BUFF".PROCESS, in2 := 73)
      { S7_Templates := "SrcType := Int" } NE_Contact(in1 := "RETAIN"."SET HPHV VCC HOLD", in2 := 0)
      I_Contact( "IEC_Timer_0_DB_90".Q )
   END_RUNG wire#w2
   RUNG wire#w1
      { S7_Templates := "SrcType := Int" } EQ_Contact(in1 := "BUFF".PROCESS, in2 := 77)
      { S7_Templates := "SrcType := Int" } NE_Contact(in1 := "RETAIN"."SET HPHV HEAT HOLD", in2 := 0)
      Contact( "IEC_Timer_0_DB_86".Q )
   END_RUNG wire#w2
   RUNG wire#w1
      { S7_Templates := "SrcType := Int" } EQ_Contact(in1 := "BUFF".PROCESS, in2 := 80)
      { S7_Templates := "SrcType := Int" } NE_Contact(in1 := "RETAIN"."SET HPHV ATS HOLD", in2 := 0)
      I_Contact( "IEC_Timer_0_DB_88".Q )
   END_RUNG wire#w2
   // the same network as SCL:
   #_w1 := "AlwaysTRUE" AND ((("BUFF".PROCESS = 48) AND "IEC_Timer_0_DB_102".Q) OR (("BUFF".PROCESS = 92) AND NOT "IEC_Timer_0_DB_80".Q) OR (("BUFF".PROCESS = 492) AND NOT "IEC_Timer_0_DB_192".Q) OR (("BUFF".PROCESS = 93) AND NOT "IEC_Timer_0_DB_84".Q) OR (("BUFF".PROCESS = 493) AND NOT "IEC_Timer_0_DB_196".Q) OR (("BUFF".PROCESS = 53) AND ("RETAIN"."SET BOW  VCC HOLD TIME" <> 0) AND NOT "IEC_Timer_0_DB_91".Q) OR (("BUFF".PROCESS = 57) AND ("RETAIN"."SET BOW HEAT HOLD TIME" <> 0) AND "IEC_Timer_0_DB_92".Q) OR (("BUFF".PROCESS = 60) AND ("RETAIN"."SET BOW ATS HOLD" <> 0) AND NOT "IEC_Timer_0_DB_94".Q) OR (("BUFF".PROCESS = 73) AND ("RETAIN"."SET HPHV VCC HOLD" <> 0) AND NOT "IEC_Timer_0_DB_90".Q) OR (("BUFF".PROCESS = 77) AND ("RETAIN"."SET HPHV HEAT HOLD" <> 0) AND "IEC_Timer_0_DB_86".Q) OR (("BUFF".PROCESS = 80) AND ("RETAIN"."SET HPHV ATS HOLD" <> 0) AND NOT "IEC_Timer_0_DB_88".Q));
   #_w2 := #_w1 AND NOT "PULSE22";   // rising edge
   "PULSE22" := #_w1;
   "END PRINT OK" := #_w2;
END_REGION

